Omron CX-Programmer project 新工程 (CX-Programmer 9.62)

# PLC 新PLC1: CJ2M CPU34
I/O table (CPU CJ2M-CPU34): rack 0 slot 0 CJ1W-ETN21(ETN21Mode); rack 0 slot 1 CJ1W-ID261; rack 0 slot 2 CJ1W-ID261; rack 0 slot 3 CJ1W-OD261; rack 0 slot 4 CJ1W-OD231; rack 0 slot 5 CJ1W-NC433; rack 0 slot 6 CJ1W-AD081-V1; rack 0 slot 7 CJ1W-DA08V; rack 0 slot 8 CJ1W-SCU21-V1; rack 0 slot 11 CJ2M-EIP21

## Global symbols (name address type ; comment)
0.00 BOOL  ; 手/自动选择
0.01 BOOL  ; 启动按钮
0.02 BOOL  ; 停止按钮
0.03 BOOL  ; 复位按钮
0.04 BOOL  ; 前门磁
0.05 BOOL  ; 后门磁
0.06 BOOL  ; 左门磁
0.07 BOOL  ; 右门磁
0.08 BOOL  ; 气源压力开关
0.09 BOOL  ; 主急停按钮
0.10 BOOL  ; 移动屏急停
0.11 BOOL  ; 移动屏使用中
0.12 BOOL  ; 备用1
0.13 BOOL  ; 备用2
0.14 BOOL  ; 备用3
0.15 BOOL  ; 备用4
100.00 BOOL  ; 进料定位上层前后松开输出
100.01 BOOL  ; 进料定位上层前后夹紧输出
100.02 BOOL  ; 进料定位下层前后松开输出
100.03 BOOL  ; 进料定位下层前后夹紧输出
100.04 BOOL  ; 进料定位上层左右松开输出
100.05 BOOL  ; 进料定位上层左右夹紧输出
100.06 BOOL  ; 进料定位下层左右松开输出
100.07 BOOL  ; 进料定位下层左右夹紧输出
100.08 BOOL  ; 进料定位上层平台待料输出
100.09 BOOL  ; 进料定位上层平台出料输出
100.10 BOOL  ; 进料定位下层平台待料输出
100.11 BOOL  ; 进料定位下层平台出料输出
100.12 BOOL  ; 输出
100.13 BOOL  ; 输出
100.14 BOOL  ; 输出
100.15 BOOL  ; 输出
101.00 BOOL  ; 输出
101.01 BOOL  ; 输出
101.02 BOOL  ; 输出
101.03 BOOL  ; 输出
101.04 BOOL  ; 输出
101.05 BOOL  ; 输出
101.06 BOOL  ; 输出
101.07 BOOL  ; 输出
101.08 BOOL  ; 输出
101.09 BOOL  ; 输出
101.10 BOOL  ; 输出
101.11 BOOL  ; 输出
101.12 BOOL  ; 输出
101.13 BOOL  ; 输出
101.14 BOOL  ; 输出
101.15 BOOL  ; 输出
102.00 BOOL  ; 输出
102.14 BOOL  ; 输出
102.15 BOOL  ; 输出
103.00 BOOL  ; 出料定位上层前后松开输出
103.01 BOOL  ; 出料定位上层前后夹紧输出
103.02 BOOL  ; 出料定位下层前后松开输出
103.03 BOOL  ; 出料定位下层前后夹紧输出
103.04 BOOL  ; 出料定位上层左右松开输出
103.05 BOOL  ; 出料定位上层左右夹紧输出
103.06 BOOL  ; 出料定位下层左右松开输出
103.07 BOOL  ; 出料定位下层左右夹紧输出
103.08 BOOL  ; 出料定位上层平台接料输出
103.09 BOOL  ; 出料定位上层平台出料输出
103.10 BOOL  ; 出料定位下层平台接料输出
103.11 BOOL  ; 出料定位下层平台出料输出
103.12 BOOL  ; 上下层吹气输出
103.13 BOOL  ; 输出
103.14 BOOL  ; 输出
103.15 BOOL  ; 输出
104.00 BOOL  ; 输出
104.01 BOOL  ; 输出
104.02 BOOL  ; 输出
104.03 BOOL  ; 输出
104.04 BOOL  ; 输出
104.05 BOOL  ; 输出
104.06 BOOL  ; 输出
104.07 BOOL  ; 输出
104.08 BOOL  ; 输出
104.09 BOOL  ; 输出
104.10 BOOL  ; 输出
105.14 BOOL  ; 输出
105.15 BOOL  ; 输出
106.00 BOOL  ; 进料夹爪张开输出
106.01 BOOL  ; 进料夹爪夹紧输出
106.02 BOOL  ; 进料爪上下层左右压紧上升输出
106.03 BOOL  ; 进料爪上下层左右压紧下降输出
106.04 BOOL  ; 进料爪上下层中间压紧上升输出
106.05 BOOL  ; 进料爪上下层中间压紧下降输出
106.06 BOOL  ; 进料夹爪上升输出
106.07 BOOL  ; 进料夹爪下降输出
106.08 BOOL  ; 输出
106.09 BOOL  ; 输出
106.10 BOOL  ; 输出
106.11 BOOL  ; 输出
106.12 BOOL  ; 输出
107.00 BOOL  ; 出料夹爪张开输出
107.01 BOOL  ; 出料夹爪夹紧输出
107.02 BOOL  ; 出料爪上下层左右压紧上升输出
107.03 BOOL  ; 出料爪上下层左右压紧下降输出
107.04 BOOL  ; 出料夹爪上升输出
107.05 BOOL  ; 出料夹爪下降输出
108.04 BOOL  ; 输出
108.05 BOOL  ; 输出
108.06 BOOL  ; 输出
108.07 BOOL  ; 输出
108.08 BOOL  ; 输出
108.09 BOOL  ; 输出
108.10 BOOL  ; 输出
108.11 BOOL  ; 输出
108.12 BOOL  ; 输出
108.13 BOOL  ; 输出
108.14 BOOL  ; 输出
108.15 BOOL  ; 输出
109.00 BOOL  ; 输出
109.01 BOOL  ; 输出
109.02 BOOL  ; 输出
109.03 BOOL  ; 输出
109.04 BOOL  ; 输出
109.05 BOOL  ; 输出
109.06 BOOL  ; 输出
109.07 BOOL  ; 输出
109.08 BOOL  ; 输出
109.09 BOOL  ; 输出
109.10 BOOL  ; 输出
109.11 BOOL  ; 输出
109.12 BOOL  ; 输出
109.13 BOOL  ; 输出
109.14 BOOL  ; 输出
109.15 BOOL  ; 输出
10.00 BOOL  ; 进料定位上层前后松开
10.01 BOOL  ; 进料定位上层前后夹紧
10.02 BOOL  ; 进料定位下层前后松开
10.03 BOOL  ; 进料定位下层前后夹紧
10.04 BOOL  ; 进料定位上层左右松开
10.05 BOOL  ; 进料定位上层左右夹紧
10.06 BOOL  ; 进料定位下层左右松开
10.07 BOOL  ; 进料定位下层左右夹紧
10.08 BOOL  ; 进料定位上层平台待料
10.09 BOOL  ; 进料定位上层平台出料
10.10 BOOL  ; 进料定位下层平台待料
10.11 BOOL  ; 进料定位下层平台出料
10.12 BOOL  ; 出料定位上层前后松开
10.13 BOOL  ; 出料定位上层前后夹紧
10.14 BOOL  ; 出料定位下层前后松开
10.15 BOOL  ; 出料定位下层前后夹紧
110.00 BOOL  ; 热压A增压缸上升输出
110.01 BOOL  ; 热压A增压缸下降输出
110.02 BOOL  ; 热压A上层顶升气缸上升输出
110.03 BOOL  ; 热压A上层顶升气缸下降输出
110.04 BOOL  ; 热压A下层顶升气缸上升输出
110.05 BOOL  ; 热压A下层顶升气缸下降输出
110.06 BOOL  ; 热压A垫高气缸移出输出
110.07 BOOL  ; 热压A垫高气缸热压输出
110.08 BOOL  ; 热压AHip测试气缸上升输出
110.09 BOOL  ; 热压AHip测试气缸下降输出
110.10 BOOL  ; 热压A上下层吹气输出
110.11 BOOL  ; 热压A上层HIP测试选择输出
110.12 BOOL  ; 热压A下层HIP测试选择输出
110.13 BOOL  ; 热压A极耳测试输出
110.14 BOOL  ; 热压A压力清零输出
110.15 BOOL  ; 热压B极耳测试输出
111.00 BOOL  ; 热压B压力清零输出
111.01 BOOL  ; 输出
111.02 BOOL  ; 输出
111.03 BOOL  ; 输出
111.04 BOOL  ; 输出
111.05 BOOL  ; 输出
111.06 BOOL  ; 输出
111.07 BOOL  ; 输出
111.08 BOOL  ; 输出
111.09 BOOL  ; 输出
111.10 BOOL  ; 输出
111.11 BOOL  ; 输出
111.12 BOOL  ; 输出
111.13 BOOL  ; 输出
111.14 BOOL  ; 输出
112 CHANNEL  ; 顶升伸出状态
112.14 BOOL  ; 输出
112.15 BOOL  ; 输出
113.00 BOOL  ; 热压B增压缸上升输出
113.01 BOOL  ; 热压B增压缸下降输出
113.02 BOOL  ; 热压B上层顶升气缸上升输出
113.03 BOOL  ; 热压B上层顶升气缸下降输出
113.04 BOOL  ; 热压B下层顶升气缸上升输出
113.05 BOOL  ; 热压B下层顶升气缸下降输出
113.06 BOOL  ; 热压B垫高气缸移出输出
113.07 BOOL  ; 热压B垫高气缸热压输出
113.08 BOOL  ; 热压BHip测试气缸上升输出
113.09 BOOL  ; 热压BHip测试气缸下降输出
113.10 BOOL  ; 热压B上下层吹气输出
113.11 BOOL  ; 热压B上层HIP测试选择输出
113.12 BOOL  ; 热压B下层HIP测试选择输出
113.13 BOOL  ; 热压B极耳测试输出
113.14 BOOL  ; 热压B压力清零输出
113.15 BOOL  ; 输出
114.00 BOOL  ; 输出
114.01 BOOL  ; 输出
114.02 BOOL  ; 输出
114.03 BOOL  ; 输出
114.04 BOOL  ; 输出
114.05 BOOL  ; 输出
114.06 BOOL  ; 输出
114.07 BOOL  ; 输出
114.08 BOOL  ; 输出
114.09 BOOL  ; 输出
114.10 BOOL  ; 输出
114.11 BOOL  ; 输出
114.12 BOOL  ; 输出
114.13 BOOL  ; 输出
114.14 BOOL  ; 输出
114.15 BOOL  ; 输出
115.00 BOOL  ; 输出
115.01 BOOL  ; 输出
116.00 BOOL  ; 热压C增压缸上升输出
116.01 BOOL  ; 热压C增压缸下降输出
116.02 BOOL  ; 热压C上层顶升气缸上升输出
116.03 BOOL  ; 热压C上层顶升气缸下降输出
116.04 BOOL  ; 热压C下层顶升气缸上升输出
116.05 BOOL  ; 热压C下层顶升气缸下降输出
116.06 BOOL  ; 热压C垫高气缸移出输出
116.07 BOOL  ; 热压C垫高气缸热压输出
116.08 BOOL  ; 热压CHip测试气缸上升输出
116.09 BOOL  ; 热压CHip测试气缸下降输出
116.10 BOOL  ; 热压C上下层吹气输出
116.11 BOOL  ; 热压C上层HIP测试选择输出
116.12 BOOL  ; 热压C下层HIP测试选择输出
116.13 BOOL  ; 热压C极耳测试输出
116.14 BOOL  ; 热压C压力清零输出
119.01 BOOL  ; 热压A正压伺服转矩模式输出
119.02 BOOL  ; 热压A1左右伺服转矩模式输出
119.07 BOOL  ; 热压B正压伺服转矩模式输出
119.08 BOOL  ; 热压B1左右伺服转矩模式输出
11.00 BOOL  ; 出料定位上层左右松开
11.01 BOOL  ; 出料定位上层左右夹紧
11.02 BOOL  ; 出料定位下层左右松开
11.03 BOOL  ; 出料定位下层左右夹紧
11.04 BOOL  ; 出料定位上层平台接料
11.05 BOOL  ; 出料定位上层平台出料
11.06 BOOL  ; 出料定位下层平台接料
11.07 BOOL  ; 出料定位下层平台出料
11.08 BOOL  ; 上下层吹气
11.09 BOOL  ; 进料夹爪张开
11.10 BOOL  ; 进料夹爪夹紧
11.11 BOOL  ; 进料爪上下层左右压紧上升
11.12 BOOL  ; 进料爪上下层左右压紧下降
11.13 BOOL  ; 进料爪上下层中间压紧上升
11.14 BOOL  ; 进料爪上下层中间压紧下降
11.15 BOOL  ; 进料夹爪上升
12.00 BOOL  ; 进料夹爪下降
12.01 BOOL  ; 出料夹爪张开
12.02 BOOL  ; 出料夹爪夹紧
12.03 BOOL  ; 进料爪上下层左右压紧上升
12.04 BOOL  ; 进料爪上下层左右压紧下降
12.05 BOOL  ; 进料爪上下层中间压紧上升
12.06 BOOL  ; 进料爪上下层中间压紧下降
12.07 BOOL  ; 进料夹爪上升
12.08 BOOL  ; 进料夹爪下降
12.09 BOOL  ; 热压A增压缸上升
12.10 BOOL  ; 热压A增压缸下降
12.11 BOOL  ; 热压A上层顶升气缸上升
12.12 BOOL  ; 热压A上层顶升气缸下降
12.13 BOOL  ; 热压A下层顶升气缸上升
12.14 BOOL  ; 热压A下层顶升气缸下降
12.15 BOOL  ; 热压A垫高气缸移出
13.00 BOOL  ; 热压A垫高气缸热压
13.01 BOOL  ; 热压AHip测试气缸上升
13.02 BOOL  ; 热压AHip测试气缸下降
13.03 BOOL  ; 热压A上下层吹气
13.04 BOOL  ; 热压A上层HIP测试选择继电器
13.05 BOOL  ; 热压A下层HIP测试选择继电器
13.06 BOOL  ; 热压A上下极耳有无检测继电器
13.07 BOOL  ; A工位压力清零
13.08 BOOL  ; 热压B增压缸上升
13.09 BOOL  ; 热压B增压缸下降
13.10 BOOL  ; 热压B上层顶升气缸上升
13.11 BOOL  ; 热压B上层顶升气缸下降
13.12 BOOL  ; 热压B下层顶升气缸上升
13.13 BOOL  ; 热压B下层顶升气缸下降
13.14 BOOL  ; 热压B垫高气缸移出
13.15 BOOL  ; 热压B垫高气缸热压
14.00 BOOL  ; 热压BHip测试气缸上升
14.01 BOOL  ; 热压BHip测试气缸下降
14.02 BOOL  ; 热压B上下层吹气
14.03 BOOL  ; 热压B上层HIP测试选择继电器
14.04 BOOL  ; 热压B下层HIP测试选择继电器
14.05 BOOL  ; 热压B上下极耳有无检测继电器
14.06 BOOL  ; B工位清零
14.07 BOOL  ; 热压C增压缸上升
14.08 BOOL  ; 热压C增压缸下降
14.09 BOOL  ; 热压C上层顶升气缸上升
14.10 BOOL  ; 热压C上层顶升气缸下降
14.11 BOOL  ; 热压C下层顶升气缸上升
14.12 BOOL  ; 热压C下层顶升气缸下降
14.13 BOOL  ; 热压C垫高气缸移出
14.14 BOOL  ; 热压C垫高气缸热压
14.15 BOOL  ; 热压CHip测试气缸上升
1550.03 BOOL  ; #2_1端口停止
1550.11 BOOL  ; #2_2端口停止
1559.15 BOOL  ; 单元2-端口1忙标志
1569.15 BOOL  ; 单元2-端口2忙标志
1575.03 BOOL  ; #3_1端口停止
1575.11 BOOL  ; #3_2端口停止
1584.15 BOOL  ; 单元3-端口1忙标志
1594.15 BOOL  ; 单元3-端口2忙标志
15.00 BOOL  ; 热压CHip测试气缸下降
15.01 BOOL  ; 热压C上下层吹气
15.02 BOOL  ; 热压C上层HIP测试选择继电器
15.03 BOOL  ; 热压C下层HIP测试选择继电器
15.04 BOOL  ; 热压C上下极耳有无检测继电器
15.05 BOOL  ; C工位压力清零
15.07 BOOL  ; 横移|伸缩伺服ON
15.08 BOOL  ; 横移|伸缩伺服报警解除
15.09 BOOL  ; 三个灯 红
15.10 BOOL  ; 三个灯 黄
15.11 BOOL  ; 三个灯 绿
15.12 BOOL  ; 三色灯蜂鸣器
15.13 BOOL  ; 运行指示（面板）
15.14 BOOL  ; 复位指示（面板）
15.15 BOOL  ; 停止指示（面板）
16 CHANNEL  ; 副PLC输出点映射开始地址
1600.03 BOOL  ; #4_1端口停止
1600.11 BOOL  ; #4_2端口停止
1609.15 BOOL  ; 单元4-端口1忙标志
1619.15 BOOL  ; 单元4-端口2忙标志
1625.03 BOOL  ; #5_1端口停止
1625.11 BOOL  ; #5_2端口停止
1634.15 BOOL  ; 单元5-端口1忙标志
1644.15 BOOL  ; 单元5-端口2忙标志
1659.15 BOOL  ; 单元6-端口1忙标志
1669.15 BOOL  ; 单元6-端口1忙标志
16.00 BOOL  ; 热压A上层上板左加热启动 上料侧为左
16.01 BOOL  ; 热压A上层上板中加热启动
16.02 BOOL  ; 热压A上层上板右加热启动
16.03 BOOL  ; 热压A上层下板左加热启动
16.04 BOOL  ; 热压A上层下板中加热启动
16.05 BOOL  ; 热压A上层下板右加热启动
17.00 BOOL  ; 热压A下层上板左加热启动
17.01 BOOL  ; 热压A下层上板中加热启动
17.02 BOOL  ; 热压A下层上板右加热启动
17.03 BOOL  ; 热压A下层下板左加热启动
17.04 BOOL  ; 热压A下层下板中加热启动
17.05 BOOL  ; 热压A下层下板右加热启动
18.00 BOOL  ; 热压B上层上板左加热启动
18.01 BOOL  ; 热压B上层上板中加热启动
18.02 BOOL  ; 热压B上层上板右加热启动
18.03 BOOL  ; 热压B上层下板左加热启动
18.04 BOOL  ; 热压B上层下板中加热启动
18.05 BOOL  ; 热压B上层下板右加热启动
19.00 BOOL  ; 热压B下层上板左加热启动
19.01 BOOL  ; 热压B下层上板中加热启动
19.02 BOOL  ; 热压B下层上板右加热启动
19.03 BOOL  ; 热压B下层下板左加热启动
19.04 BOOL  ; 热压B下层下板中加热启动
19.05 BOOL  ; 热压B下层下板右加热启动
1.00 BOOL  ; 启动按钮1
1.01 BOOL  ; 启动按钮2
1.02 BOOL  ; 进出料安全光栅
1.03 BOOL  ; 进料定位上层前后松开位
1.04 BOOL  ; 进料定位上层前后夹紧位
1.05 BOOL  ; 进料定位下层前后松开位
1.06 BOOL  ; 进料定位下层前后夹紧位
1.07 BOOL  ; 进料定位上层左右松开位
1.08 BOOL  ; 进料定位上层左右夹紧位
1.09 BOOL  ; 进料定位下层左右松开位
1.10 BOOL  ; 进料定位下层左右夹紧位
1.11 BOOL  ; 进料定位平台上层待料位
1.12 BOOL  ; 进料定位平台上层出料位
1.13 BOOL  ; 进料定位平台下层待料位
1.14 BOOL  ; 进料定位平台下层出料位
1.15 BOOL  ; 进料定位上层有料感应
2000.00 BOOL  ; NC433_0_X 3ST-A进出料横移伺服A存储器操作命令激活序列数
2000.01 BOOL  ; NC433_0_X 3ST-A进出料横移伺服A存储器操作命令起动
2000.02 BOOL  ; NC433_0_X 3ST-A进出料横移伺服A存储器操作命令独立起动
2000.03 BOOL  ; NC433_0_X 3ST-A进出料横移伺服A直接操作命令绝对移动
2000.04 BOOL  ; NC433_0_X 3ST-A进出料横移伺服A直接操作命令相对移动
2000.05 BOOL  ; NC433_0_X 3ST-A进出料横移伺服A直接操作命令中断进给
2000.06 BOOL  ; NC433_0_X 3ST-A进出料横移伺服A原点定位命令原点搜索
2000.07 BOOL  ; NC433_0_X 3ST-A进出料横移伺服A原点定位命令原点返回
2000.08 BOOL  ; NC433_0_X 3ST-A进出料横移伺服A原点定位命令当前位置预置
2000.09 BOOL  ; NC433_0_X 3ST-A进出料横移伺服A点动
2000.10 BOOL  ; NC433_0_X 3ST-A进出料横移伺服A点动方向(0=CW,1=CCW)
2000.11 BOOL  ; NC433_0_X 3ST-A进出料横移伺服A示教
2000.12 BOOL  ; NC433_0_X 3ST-A进出料横移伺服A错误清除
2000.13 BOOL  ; NC433_0_X 3ST-A进出料横移伺服A偏差计数器复位输出/ 原点调整命令输出
2000.14 BOOL  ; NC433_0_X 3ST-A进出料横移伺服A激活Override
2000.15 BOOL  ; NC433_0_X 3ST-A进出料横移伺服A停止
2001.00 BOOL  ; NC433_0_X 3ST-A进出料横移伺服A预留
2001.01 BOOL  ; NC433_0_X 3ST-A进出料横移伺服A预留
2001.02 BOOL  ; NC433_0_X 3ST-A进出料横移伺服A预留
2001.03 BOOL  ; NC433_0_X 3ST-A进出料横移伺服A预留
2001.04 BOOL  ; NC433_0_X 3ST-A进出料横移伺服A预留
2001.05 BOOL  ; NC433_0_X 3ST-A进出料横移伺服A预留
2001.06 BOOL  ; NC433_0_X 3ST-A进出料横移伺服A预留
2001.07 BOOL  ; NC433_0_X 3ST-A进出料横移伺服A预留
2001.08 BOOL  ; NC433_0_X 3ST-A进出料横移伺服A强制中断
2001.09 BOOL  ; NC433_0_X 3ST-A进出料横移伺服A预留
2001.10 BOOL  ; NC433_0_X 3ST-A进出料横移伺服A预留
2001.11 BOOL  ; NC433_0_X 3ST-A进出料横移伺服A预留
2001.12 BOOL  ; NC433_0_X 3ST-A进出料横移伺服A数据写入
2001.13 BOOL  ; NC433_0_X 3ST-A进出料横移伺服A数据读出
2001.14 BOOL  ; NC433_0_X 3ST-A进出料横移伺服A数据保存
2001.15 BOOL  ; NC433_0_X 3ST-A进出料横移伺服A预留
2002.00 BOOL  ; NC433_0_Y 3ST-A进出料伸缩伺服A存储器操作命令激活序列数
2002.01 BOOL  ; NC433_0_Y 3ST-A进出料伸缩伺服A存储器操作命令起动
2002.02 BOOL  ; NC433_0_Y 3ST-A进出料伸缩伺服A存储器操作命令独立起动
2002.03 BOOL  ; NC433_0_Y 3ST-A进出料伸缩伺服A直接操作命令绝对移动
2002.04 BOOL  ; NC433_0_Y 3ST-A进出料伸缩伺服A直接操作命令相对移动
2002.05 BOOL  ; NC433_0_Y 3ST-A进出料伸缩伺服A直接操作命令中断进给
2002.06 BOOL  ; NC433_0_Y 3ST-A进出料伸缩伺服A原点定位命令原点搜索
2002.07 BOOL  ; NC433_0_Y 3ST-A进出料伸缩伺服A原点定位命令原点返回
2002.08 BOOL  ; NC433_0_Y 3ST-A进出料伸缩伺服A原点定位命令当前位置预置
2002.09 BOOL  ; NC433_0_Y 3ST-A进出料伸缩伺服A点动
2002.10 BOOL  ; NC433_0_Y 3ST-A进出料伸缩伺服A点动方向(0=CW,1=CCW)
2002.11 BOOL  ; NC433_0_Y 3ST-A进出料伸缩伺服A示教
2002.12 BOOL  ; NC433_0_Y 3ST-A进出料伸缩伺服A错误清除
2002.13 BOOL  ; NC433_0_Y 3ST-A进出料伸缩伺服A偏差计数器复位输出/ 原点调整命令输出
2002.14 BOOL  ; NC433_0_Y 3ST-A进出料伸缩伺服A激活Override
2002.15 BOOL  ; NC433_0_Y 3ST-A进出料伸缩伺服A停止
2003.00 BOOL  ; NC433_0_Y 3ST-A进出料伸缩伺服A预留
2003.01 BOOL  ; NC433_0_Y 3ST-A进出料伸缩伺服A预留
2003.02 BOOL  ; NC433_0_Y 3ST-A进出料伸缩伺服A预留
2003.03 BOOL  ; NC433_0_Y 3ST-A进出料伸缩伺服A预留
2003.04 BOOL  ; NC433_0_Y 3ST-A进出料伸缩伺服A预留
2003.05 BOOL  ; NC433_0_Y 3ST-A进出料伸缩伺服A预留
2003.06 BOOL  ; NC433_0_Y 3ST-A进出料伸缩伺服A预留
2003.07 BOOL  ; NC433_0_Y 3ST-A进出料伸缩伺服A预留
2003.08 BOOL  ; NC433_0_Y 3ST-A进出料伸缩伺服A强制中断
2003.09 BOOL  ; NC433_0_Y 3ST-A进出料伸缩伺服A预留
2003.10 BOOL  ; NC433_0_Y 3ST-A进出料伸缩伺服A预留
2003.11 BOOL  ; NC433_0_Y 3ST-A进出料伸缩伺服A预留
2003.12 BOOL  ; NC433_0_Y 3ST-A进出料伸缩伺服A数据写入
2003.13 BOOL  ; NC433_0_Y 3ST-A进出料伸缩伺服A数据读出
2003.14 BOOL  ; NC433_0_Y 3ST-A进出料伸缩伺服A数据保存
2003.15 BOOL  ; NC433_0_Y 3ST-A进出料伸缩伺服A预留
2004.00 BOOL  ; NC433_0_ Z 3ST-B进出料横移伺服B存储器操作命令激活序列数
2004.01 BOOL  ; NC433_0_ Z 3ST-B进出料横移伺服B存储器操作命令起动
2004.02 BOOL  ; NC433_0_ Z 3ST-B进出料横移伺服B存储器操作命令独立起动
2004.03 BOOL  ; NC433_0_ Z 3ST-B进出料横移伺服B直接操作命令绝对移动
2004.04 BOOL  ; NC433_0_ Z 3ST-B进出料横移伺服B直接操作命令相对移动
2004.05 BOOL  ; NC433_0_ Z 3ST-B进出料横移伺服B直接操作命令中断进给
2004.06 BOOL  ; NC433_0_ Z 3ST-B进出料横移伺服B原点定位命令原点搜索
2004.07 BOOL  ; NC433_0_ Z 3ST-B进出料横移伺服B原点定位命令原点返回
2004.08 BOOL  ; NC433_0_ Z 3ST-B进出料横移伺服B原点定位命令当前位置预置
2004.09 BOOL  ; NC433_0_ Z 3ST-B进出料横移伺服B点动
2004.10 BOOL  ; NC433_0_ Z 3ST-B进出料横移伺服B点动方向(0=CW,1=CCW)
2004.11 BOOL  ; NC433_0_ Z 3ST-B进出料横移伺服B示教
2004.12 BOOL  ; NC433_0_ Z 3ST-B进出料横移伺服B错误清除
2004.13 BOOL  ; NC433_0_ Z 3ST-B进出料横移伺服B偏差计数器复位输出/ 原点调整命令输出
2004.14 BOOL  ; NC433_0_ Z 3ST-B进出料横移伺服B激活Override
2004.15 BOOL  ; NC433_0_ Z 3ST-B进出料横移伺服B停止
2005.00 BOOL  ; NC433_0_ Z 3ST-B进出料横移伺服B预留
2005.01 BOOL  ; NC433_0_ Z 3ST-B进出料横移伺服B预留
2005.02 BOOL  ; NC433_0_ Z 3ST-B进出料横移伺服B预留
2005.03 BOOL  ; NC433_0_ Z 3ST-B进出料横移伺服B预留
2005.04 BOOL  ; NC433_0_ Z 3ST-B进出料横移伺服B预留
2005.05 BOOL  ; NC433_0_ Z 3ST-B进出料横移伺服B预留
2005.06 BOOL  ; NC433_0_ Z 3ST-B进出料横移伺服B预留
2005.07 BOOL  ; NC433_0_ Z 3ST-B进出料横移伺服B预留
2005.08 BOOL  ; NC433_0_ Z 3ST-B进出料横移伺服B强制中断
2005.09 BOOL  ; NC433_0_ Z 3ST-B进出料横移伺服B预留
2005.10 BOOL  ; NC433_0_ Z 3ST-B进出料横移伺服B预留
2005.11 BOOL  ; NC433_0_ Z 3ST-B进出料横移伺服B预留
2005.12 BOOL  ; NC433_0_ Z 3ST-B进出料横移伺服B数据写入
2005.13 BOOL  ; NC433_0_ Z 3ST-B进出料横移伺服B数据读出
2005.14 BOOL  ; NC433_0_ Z 3ST-B进出料横移伺服B数据保存
2005.15 BOOL  ; NC433_0_ Z 3ST-B进出料横移伺服B预留
2006.00 BOOL  ; NC433_0_U 3ST-B进出料伸缩伺服存储器操作命令激活序列数
2006.01 BOOL  ; NC433_0_U 3ST-B进出料伸缩伺服存储器操作命令起动
2006.02 BOOL  ; NC433_0_U 3ST-B进出料伸缩伺服存储器操作命令独立起动
2006.03 BOOL  ; NC433_0_U 3ST-B进出料伸缩伺服直接操作命令绝对移动
2006.04 BOOL  ; NC433_0_U 3ST-B进出料伸缩伺服直接操作命令相对移动
2006.05 BOOL  ; NC433_0_U 3ST-B进出料伸缩伺服直接操作命令中断进给
2006.06 BOOL  ; NC433_0_U 3ST-B进出料伸缩伺服原点定位命令原点搜索
2006.07 BOOL  ; NC433_0_U 3ST-B进出料伸缩伺服原点定位命令原点返回
2006.08 BOOL  ; NC433_0_U 3ST-B进出料伸缩伺服原点定位命令当前位置预置
2006.09 BOOL  ; NC433_0_U 3ST-B进出料伸缩伺服点动
2006.10 BOOL  ; NC433_0_U 3ST-B进出料伸缩伺服点动方向(0=CW,1=CCW)
2006.11 BOOL  ; NC433_0_U 3ST-B进出料伸缩伺服示教
2006.12 BOOL  ; NC433_0_U 3ST-B进出料伸缩伺服错误清除
2006.13 BOOL  ; NC433_0_U 3ST-B进出料伸缩伺服偏差计数器复位输出/ 原点调整命令输出
2006.14 BOOL  ; NC433_0_U 3ST-B进出料伸缩伺服激活Override
2006.15 BOOL  ; NC433_0_U 3ST-B进出料伸缩伺服停止
2007.00 BOOL  ; NC433_0_U 3ST-B进出料伸缩伺服预留
2007.01 BOOL  ; NC433_0_U 3ST-B进出料伸缩伺服预留
2007.02 BOOL  ; NC433_0_U 3ST-B进出料伸缩伺服预留
2007.03 BOOL  ; NC433_0_U 3ST-B进出料伸缩伺服预留
2007.04 BOOL  ; NC433_0_U 3ST-B进出料伸缩伺服预留
2007.05 BOOL  ; NC433_0_U 3ST-B进出料伸缩伺服预留
2007.06 BOOL  ; NC433_0_U 3ST-B进出料伸缩伺服预留
2007.07 BOOL  ; NC433_0_U 3ST-B进出料伸缩伺服预留
2007.08 BOOL  ; NC433_0_U 3ST-B进出料伸缩伺服强制中断
2007.09 BOOL  ; NC433_0_U 3ST-B进出料伸缩伺服预留
2007.10 BOOL  ; NC433_0_U 3ST-B进出料伸缩伺服预留
2007.11 BOOL  ; NC433_0_U 3ST-B进出料伸缩伺服预留
2007.12 BOOL  ; NC433_0_U 3ST-B进出料伸缩伺服数据写入
2007.13 BOOL  ; NC433_0_U 3ST-B进出料伸缩伺服数据读出
2007.14 BOOL  ; NC433_0_U 3ST-B进出料伸缩伺服数据保存
2007.15 BOOL  ; NC433_0_U 3ST-B进出料伸缩伺服预留
2008.00 BOOL  ; NC433_0_X 3ST-A进出料横移伺服A预留
2008.01 BOOL  ; NC433_0_X 3ST-A进出料横移伺服A预留
2008.02 BOOL  ; NC433_0_X 3ST-A进出料横移伺服A预留
2008.03 BOOL  ; NC433_0_X 3ST-A进出料横移伺服A预留
2008.04 BOOL  ; NC433_0_X 3ST-A进出料横移伺服A等待存储器操作
2008.05 BOOL  ; NC433_0_X 3ST-A进出料横移伺服A定位完成标志位
2008.06 BOOL  ; NC433_0_X 3ST-A进出料横移伺服A无原点标志位
2008.07 BOOL  ; NC433_0_X 3ST-A进出料横移伺服A原点停止标志位
2008.08 BOOL  ; NC433_0_X 3ST-A进出料横移伺服A0 区监测标志位
2008.09 BOOL  ; NC433_0_X 3ST-A进出料横移伺服A1 区监测标志位
2008.10 BOOL  ; NC433_0_X 3ST-A进出料横移伺服A2 区监测标志位
2008.11 BOOL  ; NC433_0_X 3ST-A进出料横移伺服A示教完成
2008.12 BOOL  ; NC433_0_X 3ST-A进出料横移伺服A错误标志
2008.13 BOOL  ; NC433_0_X 3ST-A进出料横移伺服A忙标志
2008.14 BOOL  ; NC433_0_X 3ST-A进出料横移伺服A数据传送标志位
2008.15 BOOL  ; NC433_0_X 3ST-A进出料横移伺服A减速停止执行标志位
2009.00 BOOL  ; NC433_0_X 3ST-A进出料横移伺服A预留
2009.01 BOOL  ; NC433_0_X 3ST-A进出料横移伺服A预留
2009.02 BOOL  ; NC433_0_X 3ST-A进出料横移伺服A预留
2009.03 BOOL  ; NC433_0_X 3ST-A进出料横移伺服A预留
2009.04 BOOL  ; NC433_0_X 3ST-A进出料横移伺服A预留
2009.05 BOOL  ; NC433_0_X 3ST-A进出料横移伺服A预留
2009.06 BOOL  ; NC433_0_X 3ST-A进出料横移伺服A预留
2009.07 BOOL  ; NC433_0_X 3ST-A进出料横移伺服A预留
2009.08 BOOL  ; NC433_0_X 3ST-A进出料横移伺服ACW极限输入信号
2009.09 BOOL  ; NC433_0_X 3ST-A进出料横移伺服ACCW极限输入信号
2009.10 BOOL  ; NC433_0_X 3ST-A进出料横移伺服A原点接近输入信号
2009.11 BOOL  ; NC433_0_X 3ST-A进出料横移伺服A原点输入信号
2009.12 BOOL  ; NC433_0_X 3ST-A进出料横移伺服A中断输入信号
2009.13 BOOL  ; NC433_0_X 3ST-A进出料横移伺服A紧急输入信号
2009.14 BOOL  ; NC433_0_X 3ST-A进出料横移伺服A定位完成输入信号
2009.15 BOOL  ; NC433_0_X 3ST-A进出料横移伺服A偏差计数器复位输出/ 原点调整命令输出
2010.00 BOOL  ; NC433_0_X 3ST-A进出料横移伺服A错误代码
2010.01 BOOL  ; NC433_0_X 3ST-A进出料横移伺服A错误代码
2010.02 BOOL  ; NC433_0_X 3ST-A进出料横移伺服A错误代码
2010.03 BOOL  ; NC433_0_X 3ST-A进出料横移伺服A错误代码
2010.04 BOOL  ; NC433_0_X 3ST-A进出料横移伺服A错误代码
2010.05 BOOL  ; NC433_0_X 3ST-A进出料横移伺服A错误代码
2010.06 BOOL  ; NC433_0_X 3ST-A进出料横移伺服A错误代码
2010.07 BOOL  ; NC433_0_X 3ST-A进出料横移伺服A错误代码
2010.08 BOOL  ; NC433_0_X 3ST-A进出料横移伺服A错误代码
2010.09 BOOL  ; NC433_0_X 3ST-A进出料横移伺服A错误代码
2010.10 BOOL  ; NC433_0_X 3ST-A进出料横移伺服A错误代码
2010.11 BOOL  ; NC433_0_X 3ST-A进出料横移伺服A错误代码
2010.12 BOOL  ; NC433_0_X 3ST-A进出料横移伺服A错误代码
2010.13 BOOL  ; NC433_0_X 3ST-A进出料横移伺服A错误代码
2010.14 BOOL  ; NC433_0_X 3ST-A进出料横移伺服A错误代码
2010.15 BOOL  ; NC433_0_X 3ST-A进出料横移伺服A错误代码
2011.00 BOOL  ; NC433_0_Y 3ST-A进出料伸缩伺服A预留
2011.01 BOOL  ; NC433_0_Y 3ST-A进出料伸缩伺服A预留
2011.02 BOOL  ; NC433_0_Y 3ST-A进出料伸缩伺服A预留
2011.03 BOOL  ; NC433_0_Y 3ST-A进出料伸缩伺服A预留
2011.04 BOOL  ; NC433_0_Y 3ST-A进出料伸缩伺服A等待存储器操作
2011.05 BOOL  ; NC433_0_Y 3ST-A进出料伸缩伺服A定位完成标志位
2011.06 BOOL  ; NC433_0_Y 3ST-A进出料伸缩伺服A无原点标志位
2011.07 BOOL  ; NC433_0_Y 3ST-A进出料伸缩伺服A原点停止标志位
2011.08 BOOL  ; NC433_0_Y 3ST-A进出料伸缩伺服A0 区监测标志位
2011.09 BOOL  ; NC433_0_Y 3ST-A进出料伸缩伺服A1 区监测标志位
2011.10 BOOL  ; NC433_0_Y 3ST-A进出料伸缩伺服A2 区监测标志位
2011.11 BOOL  ; NC433_0_Y 3ST-A进出料伸缩伺服A示教完成
2011.12 BOOL  ; NC433_0_Y 3ST-A进出料伸缩伺服A错误标志
2011.13 BOOL  ; NC433_0_Y 3ST-A进出料伸缩伺服A忙标志
2011.14 BOOL  ; NC433_0_Y 3ST-A进出料伸缩伺服A数据传送标志位
2011.15 BOOL  ; NC433_0_Y 3ST-A进出料伸缩伺服A减速停止执行标志位
2012.00 BOOL  ; NC433_0_Y 3ST-A进出料伸缩伺服A预留
2012.01 BOOL  ; NC433_0_Y 3ST-A进出料伸缩伺服A预留
2012.02 BOOL  ; NC433_0_Y 3ST-A进出料伸缩伺服A预留
2012.03 BOOL  ; NC433_0_Y 3ST-A进出料伸缩伺服A预留
2012.04 BOOL  ; NC433_0_Y 3ST-A进出料伸缩伺服A预留
2012.05 BOOL  ; NC433_0_Y 3ST-A进出料伸缩伺服A预留
2012.06 BOOL  ; NC433_0_Y 3ST-A进出料伸缩伺服A预留
2012.07 BOOL  ; NC433_0_Y 3ST-A进出料伸缩伺服A预留
2012.08 BOOL  ; NC433_0_Y 3ST-A进出料伸缩伺服ACW极限输入信号
2012.09 BOOL  ; NC433_0_Y 3ST-A进出料伸缩伺服ACCW极限输入信号
2012.10 BOOL  ; NC433_0_Y 3ST-A进出料伸缩伺服A原点接近输入信号
2012.11 BOOL  ; NC433_0_Y 3ST-A进出料伸缩伺服A原点输入信号
2012.12 BOOL  ; NC433_0_Y 3ST-A进出料伸缩伺服A中断输入信号
2012.13 BOOL  ; NC433_0_Y 3ST-A进出料伸缩伺服A紧急输入信号
2012.14 BOOL  ; NC433_0_Y 3ST-A进出料伸缩伺服A定位完成输入信号
2012.15 BOOL  ; NC433_0_Y 3ST-A进出料伸缩伺服A偏差计数器复位输出/ 原点调整命令输出
2013.00 BOOL  ; NC433_0_Y 3ST-A进出料伸缩伺服A错误代码
2013.01 BOOL  ; NC433_0_Y 3ST-A进出料伸缩伺服A错误代码
2013.02 BOOL  ; NC433_0_Y 3ST-A进出料伸缩伺服A错误代码
2013.03 BOOL  ; NC433_0_Y 3ST-A进出料伸缩伺服A错误代码
2013.04 BOOL  ; NC433_0_Y 3ST-A进出料伸缩伺服A错误代码
2013.05 BOOL  ; NC433_0_Y 3ST-A进出料伸缩伺服A错误代码
2013.06 BOOL  ; NC433_0_Y 3ST-A进出料伸缩伺服A错误代码
2013.07 BOOL  ; NC433_0_Y 3ST-A进出料伸缩伺服A错误代码
2013.08 BOOL  ; NC433_0_Y 3ST-A进出料伸缩伺服A错误代码
2013.09 BOOL  ; NC433_0_Y 3ST-A进出料伸缩伺服A错误代码
2013.10 BOOL  ; NC433_0_Y 3ST-A进出料伸缩伺服A错误代码
2013.11 BOOL  ; NC433_0_Y 3ST-A进出料伸缩伺服A错误代码
2013.12 BOOL  ; NC433_0_Y 3ST-A进出料伸缩伺服A错误代码
2013.13 BOOL  ; NC433_0_Y 3ST-A进出料伸缩伺服A错误代码
2013.14 BOOL  ; NC433_0_Y 3ST-A进出料伸缩伺服A错误代码
2013.15 BOOL  ; NC433_0_Y 3ST-A进出料伸缩伺服A错误代码
2014.00 BOOL  ; NC433_0_ Z 3ST-B进出料横移伺服B预留
2014.01 BOOL  ; NC433_0_ Z 3ST-B进出料横移伺服B预留
2014.02 BOOL  ; NC433_0_ Z 3ST-B进出料横移伺服B预留
2014.03 BOOL  ; NC433_0_ Z 3ST-B进出料横移伺服B预留
2014.04 BOOL  ; NC433_0_ Z 3ST-B进出料横移伺服B等待存储器操作
2014.05 BOOL  ; NC433_0_ Z 3ST-B进出料横移伺服B定位完成标志位
2014.06 BOOL  ; NC433_0_ Z 3ST-B进出料横移伺服B无原点标志位
2014.07 BOOL  ; NC433_0_ Z 3ST-B进出料横移伺服B原点停止标志位
2014.08 BOOL  ; NC433_0_ Z 3ST-B进出料横移伺服B0 区监测标志位
2014.09 BOOL  ; NC433_0_ Z 3ST-B进出料横移伺服B1 区监测标志位
2014.10 BOOL  ; NC433_0_ Z 3ST-B进出料横移伺服B2 区监测标志位
2014.11 BOOL  ; NC433_0_ Z 3ST-B进出料横移伺服B示教完成
2014.12 BOOL  ; NC433_0_ Z 3ST-B进出料横移伺服B错误标志
2014.13 BOOL  ; NC433_0_ Z 3ST-B进出料横移伺服B忙标志
2014.14 BOOL  ; NC433_0_ Z 3ST-B进出料横移伺服B数据传送标志位
2014.15 BOOL  ; NC433_0_ Z 3ST-B进出料横移伺服B减速停止执行标志位
2015.00 BOOL  ; NC433_0_ Z 3ST-B进出料横移伺服B预留
2015.01 BOOL  ; NC433_0_ Z 3ST-B进出料横移伺服B预留
2015.02 BOOL  ; NC433_0_ Z 3ST-B进出料横移伺服B预留
2015.03 BOOL  ; NC433_0_ Z 3ST-B进出料横移伺服B预留
2015.04 BOOL  ; NC433_0_ Z 3ST-B进出料横移伺服B预留
2015.05 BOOL  ; NC433_0_ Z 3ST-B进出料横移伺服B预留
2015.06 BOOL  ; NC433_0_ Z 3ST-B进出料横移伺服B预留
2015.07 BOOL  ; NC433_0_ Z 3ST-B进出料横移伺服B预留
2015.08 BOOL  ; NC433_0_ Z 3ST-B进出料横移伺服BCW极限输入信号
2015.09 BOOL  ; NC433_0_ Z 3ST-B进出料横移伺服BCCW极限输入信号
2015.10 BOOL  ; NC433_0_ Z 3ST-B进出料横移伺服B原点接近输入信号
2015.11 BOOL  ; NC433_0_ Z 3ST-B进出料横移伺服B原点输入信号
2015.12 BOOL  ; NC433_0_ Z 3ST-B进出料横移伺服B中断输入信号
2015.13 BOOL  ; NC433_0_ Z 3ST-B进出料横移伺服B紧急输入信号
2015.14 BOOL  ; NC433_0_ Z 3ST-B进出料横移伺服B定位完成输入信号
2015.15 BOOL  ; NC433_0_ Z 3ST-B进出料横移伺服B偏差计数器复位输出/ 原点调整命令输出
2016.00 BOOL  ; NC433_0_ Z 3ST-B进出料横移伺服B错误代码
2016.01 BOOL  ; NC433_0_ Z 3ST-B进出料横移伺服B错误代码
2016.02 BOOL  ; NC433_0_ Z 3ST-B进出料横移伺服B错误代码
2016.03 BOOL  ; NC433_0_ Z 3ST-B进出料横移伺服B错误代码
2016.04 BOOL  ; NC433_0_ Z 3ST-B进出料横移伺服B错误代码
2016.05 BOOL  ; NC433_0_ Z 3ST-B进出料横移伺服B错误代码
2016.06 BOOL  ; NC433_0_ Z 3ST-B进出料横移伺服B错误代码
2016.07 BOOL  ; NC433_0_ Z 3ST-B进出料横移伺服B错误代码
2016.08 BOOL  ; NC433_0_ Z 3ST-B进出料横移伺服B错误代码
2016.09 BOOL  ; NC433_0_ Z 3ST-B进出料横移伺服B错误代码
2016.10 BOOL  ; NC433_0_ Z 3ST-B进出料横移伺服B错误代码
2016.11 BOOL  ; NC433_0_ Z 3ST-B进出料横移伺服B错误代码
2016.12 BOOL  ; NC433_0_ Z 3ST-B进出料横移伺服B错误代码
2016.13 BOOL  ; NC433_0_ Z 3ST-B进出料横移伺服B错误代码
2016.14 BOOL  ; NC433_0_ Z 3ST-B进出料横移伺服B错误代码
2016.15 BOOL  ; NC433_0_ Z 3ST-B进出料横移伺服B错误代码
2017.00 BOOL  ; NC433_0_U 3ST-B进出料伸缩伺服预留
2017.01 BOOL  ; NC433_0_U 3ST-B进出料伸缩伺服预留
2017.02 BOOL  ; NC433_0_U 3ST-B进出料伸缩伺服预留
2017.03 BOOL  ; NC433_0_U 3ST-B进出料伸缩伺服预留
2017.04 BOOL  ; NC433_0_U 3ST-B进出料伸缩伺服等待存储器操作
2017.05 BOOL  ; NC433_0_U 3ST-B进出料伸缩伺服定位完成标志位
2017.06 BOOL  ; NC433_0_U 3ST-B进出料伸缩伺服无原点标志位
2017.07 BOOL  ; NC433_0_U 3ST-B进出料伸缩伺服原点停止标志位
2017.08 BOOL  ; NC433_0_U 3ST-B进出料伸缩伺服0 区监测标志位
2017.09 BOOL  ; NC433_0_U 3ST-B进出料伸缩伺服1 区监测标志位
2017.10 BOOL  ; NC433_0_U 3ST-B进出料伸缩伺服2 区监测标志位
2017.11 BOOL  ; NC433_0_U 3ST-B进出料伸缩伺服示教完成
2017.12 BOOL  ; NC433_0_U 3ST-B进出料伸缩伺服错误标志
2017.13 BOOL  ; NC433_0_U 3ST-B进出料伸缩伺服忙标志
2017.14 BOOL  ; NC433_0_U 3ST-B进出料伸缩伺服数据传送标志位
2017.15 BOOL  ; NC433_0_U 3ST-B进出料伸缩伺服减速停止执行标志位
2018.00 BOOL  ; NC433_0_U 3ST-B进出料伸缩伺服预留
2018.01 BOOL  ; NC433_0_U 3ST-B进出料伸缩伺服预留
2018.02 BOOL  ; NC433_0_U 3ST-B进出料伸缩伺服预留
2018.03 BOOL  ; NC433_0_U 3ST-B进出料伸缩伺服预留
2018.04 BOOL  ; NC433_0_U 3ST-B进出料伸缩伺服预留
2018.05 BOOL  ; NC433_0_U 3ST-B进出料伸缩伺服预留
2018.06 BOOL  ; NC433_0_U 3ST-B进出料伸缩伺服预留
2018.07 BOOL  ; NC433_0_U 3ST-B进出料伸缩伺服预留
2018.08 BOOL  ; NC433_0_U 3ST-B进出料伸缩伺服CW极限输入信号
2018.09 BOOL  ; NC433_0_U 3ST-B进出料伸缩伺服CCW极限输入信号
2018.10 BOOL  ; NC433_0_U 3ST-B进出料伸缩伺服原点接近输入信号
2018.11 BOOL  ; NC433_0_U 3ST-B进出料伸缩伺服原点输入信号
2018.12 BOOL  ; NC433_0_U 3ST-B进出料伸缩伺服中断输入信号
2018.13 BOOL  ; NC433_0_U 3ST-B进出料伸缩伺服紧急输入信号
2018.14 BOOL  ; NC433_0_U 3ST-B进出料伸缩伺服定位完成输入信号
2018.15 BOOL  ; NC433_0_U 3ST-B进出料伸缩伺服偏差计数器复位输出/ 原点调整命令输出
2019.00 BOOL  ; NC433_0_U 3ST-B进出料伸缩伺服错误代码
2019.01 BOOL  ; NC433_0_U 3ST-B进出料伸缩伺服错误代码
2019.02 BOOL  ; NC433_0_U 3ST-B进出料伸缩伺服错误代码
2019.03 BOOL  ; NC433_0_U 3ST-B进出料伸缩伺服错误代码
2019.04 BOOL  ; NC433_0_U 3ST-B进出料伸缩伺服错误代码
2019.05 BOOL  ; NC433_0_U 3ST-B进出料伸缩伺服错误代码
2019.06 BOOL  ; NC433_0_U 3ST-B进出料伸缩伺服错误代码
2019.07 BOOL  ; NC433_0_U 3ST-B进出料伸缩伺服错误代码
2019.08 BOOL  ; NC433_0_U 3ST-B进出料伸缩伺服错误代码
2019.09 BOOL  ; NC433_0_U 3ST-B进出料伸缩伺服错误代码
2019.10 BOOL  ; NC433_0_U 3ST-B进出料伸缩伺服错误代码
2019.11 BOOL  ; NC433_0_U 3ST-B进出料伸缩伺服错误代码
2019.12 BOOL  ; NC433_0_U 3ST-B进出料伸缩伺服错误代码
2019.13 BOOL  ; NC433_0_U 3ST-B进出料伸缩伺服错误代码
2019.14 BOOL  ; NC433_0_U 3ST-B进出料伸缩伺服错误代码
2019.15 BOOL  ; NC433_0_U 3ST-B进出料伸缩伺服错误代码
2020.00 BOOL  ; NC433_1_X 4ST_A正压伺服A存储器操作命令激活序列数
2020.01 BOOL  ; NC433_1_X 4ST_A正压伺服A存储器操作命令起动
2020.02 BOOL  ; NC433_1_X 4ST_A正压伺服A存储器操作命令独立起动
2020.03 BOOL  ; NC433_1_X 4ST_A正压伺服A直接操作命令绝对移动
2020.04 BOOL  ; NC433_1_X 4ST_A正压伺服A直接操作命令相对移动
2020.05 BOOL  ; NC433_1_X 4ST_A正压伺服A直接操作命令中断进给
2020.06 BOOL  ; NC433_1_X 4ST_A正压伺服A原点定位命令原点搜索
2020.07 BOOL  ; NC433_1_X 4ST_A正压伺服A原点定位命令原点返回
2020.08 BOOL  ; NC433_1_X 4ST_A正压伺服A原点定位命令当前位置预置
2020.09 BOOL  ; NC433_1_X 4ST_A正压伺服A点动
2020.10 BOOL  ; NC433_1_X 4ST_A正压伺服A点动方向(0=CW,1=CCW)
2020.11 BOOL  ; NC433_1_X 4ST_A正压伺服A示教
2020.12 BOOL  ; NC433_1_X 4ST_A正压伺服A错误清除
2020.13 BOOL  ; NC433_1_X 4ST_A正压伺服A偏差计数器复位输出/ 原点调整命令输出
2020.14 BOOL  ; NC433_1_X 4ST_A正压伺服A激活Override
2020.15 BOOL  ; NC433_1_X 4ST_A正压伺服A停止
2021.00 BOOL  ; NC433_1_X 4ST_A正压伺服A预留
2021.01 BOOL  ; NC433_1_X 4ST_A正压伺服A预留
2021.02 BOOL  ; NC433_1_X 4ST_A正压伺服A预留
2021.03 BOOL  ; NC433_1_X 4ST_A正压伺服A预留
2021.04 BOOL  ; NC433_1_X 4ST_A正压伺服A预留
2021.05 BOOL  ; NC433_1_X 4ST_A正压伺服A预留
2021.06 BOOL  ; NC433_1_X 4ST_A正压伺服A预留
2021.07 BOOL  ; NC433_1_X 4ST_A正压伺服A预留
2021.08 BOOL  ; NC433_1_X 4ST_A正压伺服A强制中断
2021.09 BOOL  ; NC433_1_X 4ST_A正压伺服A预留
2021.10 BOOL  ; NC433_1_X 4ST_A正压伺服A预留
2021.11 BOOL  ; NC433_1_X 4ST_A正压伺服A预留
2021.12 BOOL  ; NC433_1_X 4ST_A正压伺服A数据写入
2021.13 BOOL  ; NC433_1_X 4ST_A正压伺服A数据读出
2021.14 BOOL  ; NC433_1_X 4ST_A正压伺服A数据保存
2021.15 BOOL  ; NC433_1_X 4ST_A正压伺服A预留
2022.00 BOOL  ; NC433_1_Y 4ST_A压板平移伺服存储器操作命令激活序列数
2022.01 BOOL  ; NC433_1_Y 4ST_A压板平移伺服存储器操作命令起动
2022.02 BOOL  ; NC433_1_Y 4ST_A压板平移伺服存储器操作命令独立起动
2022.03 BOOL  ; NC433_1_Y 4ST_A压板平移伺服直接操作命令绝对移动
2022.04 BOOL  ; NC433_1_Y 4ST_A压板平移伺服直接操作命令相对移动
2022.05 BOOL  ; NC433_1_Y 4ST_A压板平移伺服直接操作命令中断进给
2022.06 BOOL  ; NC433_1_Y 4ST_A压板平移伺服原点定位命令原点搜索
2022.07 BOOL  ; NC433_1_Y 4ST_A压板平移伺服原点定位命令原点返回
2022.08 BOOL  ; NC433_1_Y 4ST_A压板平移伺服原点定位命令当前位置预置
2022.09 BOOL  ; NC433_1_Y 4ST_A压板平移伺服点动
2022.10 BOOL  ; NC433_1_Y 4ST_A压板平移伺服点动方向(0=CW,1=CCW)
2022.11 BOOL  ; NC433_1_Y 4ST_A压板平移伺服示教
2022.12 BOOL  ; NC433_1_Y 4ST_A压板平移伺服错误清除
2022.13 BOOL  ; NC433_1_Y 4ST_A压板平移伺服偏差计数器复位输出/ 原点调整命令输出
2022.14 BOOL  ; NC433_1_Y 4ST_A压板平移伺服激活Override
2022.15 BOOL  ; NC433_1_Y 4ST_A压板平移伺服停止
2023.00 BOOL  ; NC433_1_Y 4ST_A压板平移伺服预留
2023.01 BOOL  ; NC433_1_Y 4ST_A压板平移伺服预留
2023.02 BOOL  ; NC433_1_Y 4ST_A压板平移伺服预留
2023.03 BOOL  ; NC433_1_Y 4ST_A压板平移伺服预留
2023.04 BOOL  ; NC433_1_Y 4ST_A压板平移伺服预留
2023.05 BOOL  ; NC433_1_Y 4ST_A压板平移伺服预留
2023.06 BOOL  ; NC433_1_Y 4ST_A压板平移伺服预留
2023.07 BOOL  ; NC433_1_Y 4ST_A压板平移伺服预留
2023.08 BOOL  ; NC433_1_Y 4ST_A压板平移伺服强制中断
2023.09 BOOL  ; NC433_1_Y 4ST_A压板平移伺服预留
2023.10 BOOL  ; NC433_1_Y 4ST_A压板平移伺服预留
2023.11 BOOL  ; NC433_1_Y 4ST_A压板平移伺服预留
2023.12 BOOL  ; NC433_1_Y 4ST_A压板平移伺服数据写入
2023.13 BOOL  ; NC433_1_Y 4ST_A压板平移伺服数据读出
2023.14 BOOL  ; NC433_1_Y 4ST_A压板平移伺服数据保存
2023.15 BOOL  ; NC433_1_Y 4ST_A压板平移伺服预留
2024.00 BOOL  ; NC433_1_Z 4ST_A侧压A1左伺服存储器操作命令激活序列数
2024.01 BOOL  ; NC433_1_Z 4ST_A侧压A1左伺服存储器操作命令起动
2024.02 BOOL  ; NC433_1_Z 4ST_A侧压A1左伺服存储器操作命令独立起动
2024.03 BOOL  ; NC433_1_Z 4ST_A侧压A1左伺服直接操作命令绝对移动
2024.04 BOOL  ; NC433_1_Z 4ST_A侧压A1左伺服直接操作命令相对移动
2024.05 BOOL  ; NC433_1_Z 4ST_A侧压A1左伺服直接操作命令中断进给
2024.06 BOOL  ; NC433_1_Z 4ST_A侧压A1左伺服原点定位命令原点搜索
2024.07 BOOL  ; NC433_1_Z 4ST_A侧压A1左伺服原点定位命令原点返回
2024.08 BOOL  ; NC433_1_Z 4ST_A侧压A1左伺服原点定位命令当前位置预置
2024.09 BOOL  ; NC433_1_Z 4ST_A侧压A1左伺服点动
2024.10 BOOL  ; NC433_1_Z 4ST_A侧压A1左伺服点动方向(0=CW,1=CCW)
2024.11 BOOL  ; NC433_1_Z 4ST_A侧压A1左伺服示教
2024.12 BOOL  ; NC433_1_Z 4ST_A侧压A1左伺服错误清除
2024.13 BOOL  ; NC433_1_Z 4ST_A侧压A1左伺服偏差计数器复位输出/ 原点调整命令输出
2024.14 BOOL  ; NC433_1_Z 4ST_A侧压A1左伺服激活Override
2024.15 BOOL  ; NC433_1_Z 4ST_A侧压A1左伺服停止
2025.00 BOOL  ; NC433_1_Z 4ST_A侧压A1左伺服预留
2025.01 BOOL  ; NC433_1_Z 4ST_A侧压A1左伺服预留
2025.02 BOOL  ; NC433_1_Z 4ST_A侧压A1左伺服预留
2025.03 BOOL  ; NC433_1_Z 4ST_A侧压A1左伺服预留
2025.04 BOOL  ; NC433_1_Z 4ST_A侧压A1左伺服预留
2025.05 BOOL  ; NC433_1_Z 4ST_A侧压A1左伺服预留
2025.06 BOOL  ; NC433_1_Z 4ST_A侧压A1左伺服预留
2025.07 BOOL  ; NC433_1_Z 4ST_A侧压A1左伺服预留
2025.08 BOOL  ; NC433_1_Z 4ST_A侧压A1左伺服强制中断
2025.09 BOOL  ; NC433_1_Z 4ST_A侧压A1左伺服预留
2025.10 BOOL  ; NC433_1_Z 4ST_A侧压A1左伺服预留
2025.11 BOOL  ; NC433_1_Z 4ST_A侧压A1左伺服预留
2025.12 BOOL  ; NC433_1_Z 4ST_A侧压A1左伺服数据写入
2025.13 BOOL  ; NC433_1_Z 4ST_A侧压A1左伺服数据读出
2025.14 BOOL  ; NC433_1_Z 4ST_A侧压A1左伺服数据保存
2025.15 BOOL  ; NC433_1_Z 4ST_A侧压A1左伺服预留
2026.00 BOOL  ; NC433_1 4ST_A侧压A1右伺服存储器操作命令激活序列数
2026.01 BOOL  ; NC433_1 4ST_A侧压A1右伺服存储器操作命令起动
2026.02 BOOL  ; NC433_1 4ST_A侧压A1右伺服存储器操作命令独立起动
2026.03 BOOL  ; NC433_1 4ST_A侧压A1右伺服直接操作命令绝对移动
2026.04 BOOL  ; NC433_1 4ST_A侧压A1右伺服直接操作命令相对移动
2026.05 BOOL  ; NC433_1 4ST_A侧压A1右伺服直接操作命令中断进给
2026.06 BOOL  ; NC433_1 4ST_A侧压A1右伺服原点定位命令原点搜索
2026.07 BOOL  ; NC433_1 4ST_A侧压A1右伺服原点定位命令原点返回
2026.08 BOOL  ; NC433_1 4ST_A侧压A1右伺服原点定位命令当前位置预置
2026.09 BOOL  ; NC433_1 4ST_A侧压A1右伺服点动
2026.10 BOOL  ; NC433_1 4ST_A侧压A1右伺服点动方向(0=CW,1=CCW)
2026.11 BOOL  ; NC433_1 4ST_A侧压A1右伺服示教
2026.12 BOOL  ; NC433_1 4ST_A侧压A1右伺服错误清除
2026.13 BOOL  ; NC433_1 4ST_A侧压A1右伺服偏差计数器复位输出/ 原点调整命令输出
2026.14 BOOL  ; NC433_1 4ST_A侧压A1右伺服激活Override
2026.15 BOOL  ; NC433_1 4ST_A侧压A1右伺服停止
2027.00 BOOL  ; NC433_1 4ST_A侧压A1右伺服预留
2027.01 BOOL  ; NC433_1 4ST_A侧压A1右伺服预留
2027.02 BOOL  ; NC433_1 4ST_A侧压A1右伺服预留
2027.03 BOOL  ; NC433_1 4ST_A侧压A1右伺服预留
2027.04 BOOL  ; NC433_1 4ST_A侧压A1右伺服预留
2027.05 BOOL  ; NC433_1 4ST_A侧压A1右伺服预留
2027.06 BOOL  ; NC433_1 4ST_A侧压A1右伺服预留
2027.07 BOOL  ; NC433_1 4ST_A侧压A1右伺服预留
2027.08 BOOL  ; NC433_1 4ST_A侧压A1右伺服强制中断
2027.09 BOOL  ; NC433_1 4ST_A侧压A1右伺服预留
2027.10 BOOL  ; NC433_1 4ST_A侧压A1右伺服预留
2027.11 BOOL  ; NC433_1 4ST_A侧压A1右伺服预留
2027.12 BOOL  ; NC433_1 4ST_A侧压A1右伺服数据写入
2027.13 BOOL  ; NC433_1 4ST_A侧压A1右伺服数据读出
2027.14 BOOL  ; NC433_1 4ST_A侧压A1右伺服数据保存
2027.15 BOOL  ; NC433_1 4ST_A侧压A1右伺服预留
2028.00 BOOL  ; NC433_1_X 4ST_A正压伺服A预留
2028.01 BOOL  ; NC433_1_X 4ST_A正压伺服A预留
2028.02 BOOL  ; NC433_1_X 4ST_A正压伺服A预留
2028.03 BOOL  ; NC433_1_X 4ST_A正压伺服A预留
2028.04 BOOL  ; NC433_1_X 4ST_A正压伺服A等待存储器操作
2028.05 BOOL  ; NC433_1_X 4ST_A正压伺服A定位完成标志位
2028.06 BOOL  ; NC433_1_X 4ST_A正压伺服A无原点标志位
2028.07 BOOL  ; NC433_1_X 4ST_A正压伺服A原点停止标志位
2028.08 BOOL  ; NC433_1_X 4ST_A正压伺服A0 区监测标志位
2028.09 BOOL  ; NC433_1_X 4ST_A正压伺服A1 区监测标志位
2028.10 BOOL  ; NC433_1_X 4ST_A正压伺服A2 区监测标志位
2028.11 BOOL  ; NC433_1_X 4ST_A正压伺服A示教完成
2028.12 BOOL  ; NC433_1_X 4ST_A正压伺服A错误标志
2028.13 BOOL  ; NC433_1_X 4ST_A正压伺服A忙标志
2028.14 BOOL  ; NC433_1_X 4ST_A正压伺服A数据传送标志位
2028.15 BOOL  ; NC433_1_X 4ST_A正压伺服A减速停止执行标志位
2029.00 BOOL  ; NC433_1_X 4ST_A正压伺服A预留
2029.01 BOOL  ; NC433_1_X 4ST_A正压伺服A预留
2029.02 BOOL  ; NC433_1_X 4ST_A正压伺服A预留
2029.03 BOOL  ; NC433_1_X 4ST_A正压伺服A预留
2029.04 BOOL  ; NC433_1_X 4ST_A正压伺服A预留
2029.05 BOOL  ; NC433_1_X 4ST_A正压伺服A预留
2029.06 BOOL  ; NC433_1_X 4ST_A正压伺服A预留
2029.07 BOOL  ; NC433_1_X 4ST_A正压伺服A预留
2029.08 BOOL  ; NC433_1_X 4ST_A正压伺服ACW极限输入信号
2029.09 BOOL  ; NC433_1_X 4ST_A正压伺服ACCW极限输入信号
2029.10 BOOL  ; NC433_1_X 4ST_A正压伺服A原点接近输入信号
2029.11 BOOL  ; NC433_1_X 4ST_A正压伺服A原点输入信号
2029.12 BOOL  ; NC433_1_X 4ST_A正压伺服A中断输入信号
2029.13 BOOL  ; NC433_1_X 4ST_A正压伺服A紧急输入信号
2029.14 BOOL  ; NC433_1_X 4ST_A正压伺服A定位完成输入信号
2029.15 BOOL  ; NC433_1_X 4ST_A正压伺服A偏差计数器复位输出/ 原点调整命令输出
2030.00 BOOL  ; NC433_1_X 4ST_A正压伺服A错误代码
2030.01 BOOL  ; NC433_1_X 4ST_A正压伺服A错误代码
2030.02 BOOL  ; NC433_1_X 4ST_A正压伺服A错误代码
2030.03 BOOL  ; NC433_1_X 4ST_A正压伺服A错误代码
2030.04 BOOL  ; NC433_1_X 4ST_A正压伺服A错误代码
2030.05 BOOL  ; NC433_1_X 4ST_A正压伺服A错误代码
2030.06 BOOL  ; NC433_1_X 4ST_A正压伺服A错误代码
2030.07 BOOL  ; NC433_1_X 4ST_A正压伺服A错误代码
2030.08 BOOL  ; NC433_1_X 4ST_A正压伺服A错误代码
2030.09 BOOL  ; NC433_1_X 4ST_A正压伺服A错误代码
2030.10 BOOL  ; NC433_1_X 4ST_A正压伺服A错误代码
2030.11 BOOL  ; NC433_1_X 4ST_A正压伺服A错误代码
2030.12 BOOL  ; NC433_1_X 4ST_A正压伺服A错误代码
2030.13 BOOL  ; NC433_1_X 4ST_A正压伺服A错误代码
2030.14 BOOL  ; NC433_1_X 4ST_A正压伺服A错误代码
2030.15 BOOL  ; NC433_1_X 4ST_A正压伺服A错误代码
2031.00 BOOL  ; NC433_1_Y 4ST_A压板平移伺服预留
2031.01 BOOL  ; NC433_1_Y 4ST_A压板平移伺服预留
2031.02 BOOL  ; NC433_1_Y 4ST_A压板平移伺服预留
2031.03 BOOL  ; NC433_1_Y 4ST_A压板平移伺服预留
2031.04 BOOL  ; NC433_1_Y 4ST_A压板平移伺服等待存储器操作
2031.05 BOOL  ; NC433_1_Y 4ST_A压板平移伺服定位完成标志位
2031.06 BOOL  ; NC433_1_Y 4ST_A压板平移伺服无原点标志位
2031.07 BOOL  ; NC433_1_Y 4ST_A压板平移伺服原点停止标志位
2031.08 BOOL  ; NC433_1_Y 4ST_A压板平移伺服0 区监测标志位
2031.09 BOOL  ; NC433_1_Y 4ST_A压板平移伺服1 区监测标志位
2031.10 BOOL  ; NC433_1_Y 4ST_A压板平移伺服2 区监测标志位
2031.11 BOOL  ; NC433_1_Y 4ST_A压板平移伺服示教完成
2031.12 BOOL  ; NC433_1_Y 4ST_A压板平移伺服错误标志
2031.13 BOOL  ; NC433_1_Y 4ST_A压板平移伺服忙标志
2031.14 BOOL  ; NC433_1_Y 4ST_A压板平移伺服数据传送标志位
2031.15 BOOL  ; NC433_1_Y 4ST_A压板平移伺服减速停止执行标志位
2032.00 BOOL  ; NC433_1_Y 4ST_A压板平移伺服预留
2032.01 BOOL  ; NC433_1_Y 4ST_A压板平移伺服预留
2032.02 BOOL  ; NC433_1_Y 4ST_A压板平移伺服预留
2032.03 BOOL  ; NC433_1_Y 4ST_A压板平移伺服预留
2032.04 BOOL  ; NC433_1_Y 4ST_A压板平移伺服预留
2032.05 BOOL  ; NC433_1_Y 4ST_A压板平移伺服预留
2032.06 BOOL  ; NC433_1_Y 4ST_A压板平移伺服预留
2032.07 BOOL  ; NC433_1_Y 4ST_A压板平移伺服预留
2032.08 BOOL  ; NC433_1_Y 4ST_A压板平移伺服CW极限输入信号
2032.09 BOOL  ; NC433_1_Y 4ST_A压板平移伺服CCW极限输入信号
2032.10 BOOL  ; NC433_1_Y 4ST_A压板平移伺服原点接近输入信号
2032.11 BOOL  ; NC433_1_Y 4ST_A压板平移伺服原点输入信号
2032.12 BOOL  ; NC433_1_Y 4ST_A压板平移伺服中断输入信号
2032.13 BOOL  ; NC433_1_Y 4ST_A压板平移伺服紧急输入信号
2032.14 BOOL  ; NC433_1_Y 4ST_A压板平移伺服定位完成输入信号
2032.15 BOOL  ; NC433_1_Y 4ST_A压板平移伺服偏差计数器复位输出/ 原点调整命令输出
2033.00 BOOL  ; NC433_1_Y 4ST_A压板平移伺服错误代码
2033.01 BOOL  ; NC433_1_Y 4ST_A压板平移伺服错误代码
2033.02 BOOL  ; NC433_1_Y 4ST_A压板平移伺服错误代码
2033.03 BOOL  ; NC433_1_Y 4ST_A压板平移伺服错误代码
2033.04 BOOL  ; NC433_1_Y 4ST_A压板平移伺服错误代码
2033.05 BOOL  ; NC433_1_Y 4ST_A压板平移伺服错误代码
2033.06 BOOL  ; NC433_1_Y 4ST_A压板平移伺服错误代码
2033.07 BOOL  ; NC433_1_Y 4ST_A压板平移伺服错误代码
2033.08 BOOL  ; NC433_1_Y 4ST_A压板平移伺服错误代码
2033.09 BOOL  ; NC433_1_Y 4ST_A压板平移伺服错误代码
2033.10 BOOL  ; NC433_1_Y 4ST_A压板平移伺服错误代码
2033.11 BOOL  ; NC433_1_Y 4ST_A压板平移伺服错误代码
2033.12 BOOL  ; NC433_1_Y 4ST_A压板平移伺服错误代码
2033.13 BOOL  ; NC433_1_Y 4ST_A压板平移伺服错误代码
2033.14 BOOL  ; NC433_1_Y 4ST_A压板平移伺服错误代码
2033.15 BOOL  ; NC433_1_Y 4ST_A压板平移伺服错误代码
2034.00 BOOL  ; NC433_1_Z 4ST_A侧压A1左伺服预留
2034.01 BOOL  ; NC433_1_Z 4ST_A侧压A1左伺服预留
2034.02 BOOL  ; NC433_1_Z 4ST_A侧压A1左伺服预留
2034.03 BOOL  ; NC433_1_Z 4ST_A侧压A1左伺服预留
2034.04 BOOL  ; NC433_1_Z 4ST_A侧压A1左伺服等待存储器操作
2034.05 BOOL  ; NC433_1_Z 4ST_A侧压A1左伺服定位完成标志位
2034.06 BOOL  ; NC433_1_Z 4ST_A侧压A1左伺服无原点标志位
2034.07 BOOL  ; NC433_1_Z 4ST_A侧压A1左伺服原点停止标志位
2034.08 BOOL  ; NC433_1_Z 4ST_A侧压A1左伺服0 区监测标志位
2034.09 BOOL  ; NC433_1_Z 4ST_A侧压A1左伺服1 区监测标志位
2034.10 BOOL  ; NC433_1_Z 4ST_A侧压A1左伺服2 区监测标志位
2034.11 BOOL  ; NC433_1_Z 4ST_A侧压A1左伺服示教完成
2034.12 BOOL  ; NC433_1_Z 4ST_A侧压A1左伺服错误标志
2034.13 BOOL  ; NC433_1_Z 4ST_A侧压A1左伺服忙标志
2034.14 BOOL  ; NC433_1_Z 4ST_A侧压A1左伺服数据传送标志位
2034.15 BOOL  ; NC433_1_Z 4ST_A侧压A1左伺服减速停止执行标志位
2035.00 BOOL  ; NC433_1_Z 4ST_A侧压A1左伺服预留
2035.01 BOOL  ; NC433_1_Z 4ST_A侧压A1左伺服预留
2035.02 BOOL  ; NC433_1_Z 4ST_A侧压A1左伺服预留
2035.03 BOOL  ; NC433_1_Z 4ST_A侧压A1左伺服预留
2035.04 BOOL  ; NC433_1_Z 4ST_A侧压A1左伺服预留
2035.05 BOOL  ; NC433_1_Z 4ST_A侧压A1左伺服预留
2035.06 BOOL  ; NC433_1_Z 4ST_A侧压A1左伺服预留
2035.07 BOOL  ; NC433_1_Z 4ST_A侧压A1左伺服预留
2035.08 BOOL  ; NC433_1_Z 4ST_A侧压A1左伺服CW极限输入信号
2035.09 BOOL  ; NC433_1_Z 4ST_A侧压A1左伺服CCW极限输入信号
2035.10 BOOL  ; NC433_1_Z 4ST_A侧压A1左伺服原点接近输入信号
2035.11 BOOL  ; NC433_1_Z 4ST_A侧压A1左伺服原点输入信号
2035.12 BOOL  ; NC433_1_Z 4ST_A侧压A1左伺服中断输入信号
2035.13 BOOL  ; NC433_1_Z 4ST_A侧压A1左伺服紧急输入信号
2035.14 BOOL  ; NC433_1_Z 4ST_A侧压A1左伺服定位完成输入信号
2035.15 BOOL  ; NC433_1_Z 4ST_A侧压A1左伺服偏差计数器复位输出/ 原点调整命令输出
2036.00 BOOL  ; NC433_1_Z 4ST_A侧压A1左伺服错误代码
2036.01 BOOL  ; NC433_1_Z 4ST_A侧压A1左伺服错误代码
2036.02 BOOL  ; NC433_1_Z 4ST_A侧压A1左伺服错误代码
2036.03 BOOL  ; NC433_1_Z 4ST_A侧压A1左伺服错误代码
2036.04 BOOL  ; NC433_1_Z 4ST_A侧压A1左伺服错误代码
2036.05 BOOL  ; NC433_1_Z 4ST_A侧压A1左伺服错误代码
2036.06 BOOL  ; NC433_1_Z 4ST_A侧压A1左伺服错误代码
2036.07 BOOL  ; NC433_1_Z 4ST_A侧压A1左伺服错误代码
2036.08 BOOL  ; NC433_1_Z 4ST_A侧压A1左伺服错误代码
2036.09 BOOL  ; NC433_1_Z 4ST_A侧压A1左伺服错误代码
2036.10 BOOL  ; NC433_1_Z 4ST_A侧压A1左伺服错误代码
2036.11 BOOL  ; NC433_1_Z 4ST_A侧压A1左伺服错误代码
2036.12 BOOL  ; NC433_1_Z 4ST_A侧压A1左伺服错误代码
2036.13 BOOL  ; NC433_1_Z 4ST_A侧压A1左伺服错误代码
2036.14 BOOL  ; NC433_1_Z 4ST_A侧压A1左伺服错误代码
2036.15 BOOL  ; NC433_1_Z 4ST_A侧压A1左伺服错误代码
2037.00 BOOL  ; NC433_1 4ST_A侧压A1右伺服预留
2037.01 BOOL  ; NC433_1 4ST_A侧压A1右伺服预留
2037.02 BOOL  ; NC433_1 4ST_A侧压A1右伺服预留
2037.03 BOOL  ; NC433_1 4ST_A侧压A1右伺服预留
2037.04 BOOL  ; NC433_1 4ST_A侧压A1右伺服等待存储器操作
2037.05 BOOL  ; NC433_1 4ST_A侧压A1右伺服定位完成标志位
2037.06 BOOL  ; NC433_1 4ST_A侧压A1右伺服无原点标志位
2037.07 BOOL  ; NC433_1 4ST_A侧压A1右伺服原点停止标志位
2037.08 BOOL  ; NC433_1 4ST_A侧压A1右伺服0 区监测标志位
2037.09 BOOL  ; NC433_1 4ST_A侧压A1右伺服1 区监测标志位
2037.10 BOOL  ; NC433_1 4ST_A侧压A1右伺服2 区监测标志位
2037.11 BOOL  ; NC433_1 4ST_A侧压A1右伺服示教完成
2037.12 BOOL  ; NC433_1 4ST_A侧压A1右伺服错误标志
2037.13 BOOL  ; NC433_1 4ST_A侧压A1右伺服忙标志
2037.14 BOOL  ; NC433_1 4ST_A侧压A1右伺服数据传送标志位
2037.15 BOOL  ; NC433_1 4ST_A侧压A1右伺服减速停止执行标志位
2038.00 BOOL  ; NC433_1 4ST_A侧压A1右伺服预留
2038.01 BOOL  ; NC433_1 4ST_A侧压A1右伺服预留
2038.02 BOOL  ; NC433_1 4ST_A侧压A1右伺服预留
2038.03 BOOL  ; NC433_1 4ST_A侧压A1右伺服预留
2038.04 BOOL  ; NC433_1 4ST_A侧压A1右伺服预留
2038.05 BOOL  ; NC433_1 4ST_A侧压A1右伺服预留
2038.06 BOOL  ; NC433_1 4ST_A侧压A1右伺服预留
2038.07 BOOL  ; NC433_1 4ST_A侧压A1右伺服预留
2038.08 BOOL  ; NC433_1 4ST_A侧压A1右伺服CW极限输入信号
2038.09 BOOL  ; NC433_1 4ST_A侧压A1右伺服CCW极限输入信号
2038.10 BOOL  ; NC433_1 4ST_A侧压A1右伺服原点接近输入信号
2038.11 BOOL  ; NC433_1 4ST_A侧压A1右伺服原点输入信号
2038.12 BOOL  ; NC433_1 4ST_A侧压A1右伺服中断输入信号
2038.13 BOOL  ; NC433_1 4ST_A侧压A1右伺服紧急输入信号
2038.14 BOOL  ; NC433_1 4ST_A侧压A1右伺服定位完成输入信号
2038.15 BOOL  ; NC433_1 4ST_A侧压A1右伺服偏差计数器复位输出/ 原点调整命令输出
2039.00 BOOL  ; NC433_1 4ST_A侧压A1右伺服错误代码
2039.01 BOOL  ; NC433_1 4ST_A侧压A1右伺服错误代码
2039.02 BOOL  ; NC433_1 4ST_A侧压A1右伺服错误代码
2039.03 BOOL  ; NC433_1 4ST_A侧压A1右伺服错误代码
2039.04 BOOL  ; NC433_1 4ST_A侧压A1右伺服错误代码
2039.05 BOOL  ; NC433_1 4ST_A侧压A1右伺服错误代码
2039.06 BOOL  ; NC433_1 4ST_A侧压A1右伺服错误代码
2039.07 BOOL  ; NC433_1 4ST_A侧压A1右伺服错误代码
2039.08 BOOL  ; NC433_1 4ST_A侧压A1右伺服错误代码
2039.09 BOOL  ; NC433_1 4ST_A侧压A1右伺服错误代码
2039.10 BOOL  ; NC433_1 4ST_A侧压A1右伺服错误代码
2039.11 BOOL  ; NC433_1 4ST_A侧压A1右伺服错误代码
2039.12 BOOL  ; NC433_1 4ST_A侧压A1右伺服错误代码
2039.13 BOOL  ; NC433_1 4ST_A侧压A1右伺服错误代码
2039.14 BOOL  ; NC433_1 4ST_A侧压A1右伺服错误代码
2039.15 BOOL  ; NC433_1 4ST_A侧压A1右伺服错误代码
2040.00 BOOL  ; NC433_2_X 4ST_A侧压A2左伺服存储器操作命令激活序列数
2040.01 BOOL  ; NC433_2_X 4ST_A侧压A2左伺服存储器操作命令起动
2040.02 BOOL  ; NC433_2_X 4ST_A侧压A2左伺服存储器操作命令独立起动
2040.03 BOOL  ; NC433_2_X 4ST_A侧压A2左伺服直接操作命令绝对移动
2040.04 BOOL  ; NC433_2_X 4ST_A侧压A2左伺服直接操作命令相对移动
2040.05 BOOL  ; NC433_2_X 4ST_A侧压A2左伺服直接操作命令中断进给
2040.06 BOOL  ; NC433_2_X 4ST_A侧压A2左伺服原点定位命令原点搜索
2040.07 BOOL  ; NC433_2_X 4ST_A侧压A2左伺服原点定位命令原点返回
2040.08 BOOL  ; NC433_2_X 4ST_A侧压A2左伺服原点定位命令当前位置预置
2040.09 BOOL  ; NC433_2_X 4ST_A侧压A2左伺服点动
2040.10 BOOL  ; NC433_2_X 4ST_A侧压A2左伺服点动方向(0=CW,1=CCW)
2040.11 BOOL  ; NC433_2_X 4ST_A侧压A2左伺服示教
2040.12 BOOL  ; NC433_2_X 4ST_A侧压A2左伺服错误清除
2040.13 BOOL  ; NC433_2_X 4ST_A侧压A2左伺服偏差计数器复位输出/ 原点调整命令输出
2040.14 BOOL  ; NC433_2_X 4ST_A侧压A2左伺服激活Override
2040.15 BOOL  ; NC433_2_X 4ST_A侧压A2左伺服停止
2041.00 BOOL  ; NC433_2_X 4ST_A侧压A2左伺服预留
2041.01 BOOL  ; NC433_2_X 4ST_A侧压A2左伺服预留
2041.02 BOOL  ; NC433_2_X 4ST_A侧压A2左伺服预留
2041.03 BOOL  ; NC433_2_X 4ST_A侧压A2左伺服预留
2041.04 BOOL  ; NC433_2_X 4ST_A侧压A2左伺服预留
2041.05 BOOL  ; NC433_2_X 4ST_A侧压A2左伺服预留
2041.06 BOOL  ; NC433_2_X 4ST_A侧压A2左伺服预留
2041.07 BOOL  ; NC433_2_X 4ST_A侧压A2左伺服预留
2041.08 BOOL  ; NC433_2_X 4ST_A侧压A2左伺服强制中断
2041.09 BOOL  ; NC433_2_X 4ST_A侧压A2左伺服预留
2041.10 BOOL  ; NC433_2_X 4ST_A侧压A2左伺服预留
2041.11 BOOL  ; NC433_2_X 4ST_A侧压A2左伺服预留
2041.12 BOOL  ; NC433_2_X 4ST_A侧压A2左伺服数据写入
2041.13 BOOL  ; NC433_2_X 4ST_A侧压A2左伺服数据读出
2041.14 BOOL  ; NC433_2_X 4ST_A侧压A2左伺服数据保存
2041.15 BOOL  ; NC433_2_X 4ST_A侧压A2左伺服预留
2042.00 BOOL  ; NC433_2_Y 4ST_A侧压A2右伺服存储器操作命令激活序列数
2042.01 BOOL  ; NC433_2_Y 4ST_A侧压A2右伺服存储器操作命令起动
2042.02 BOOL  ; NC433_2_Y 4ST_A侧压A2右伺服存储器操作命令独立起动
2042.03 BOOL  ; NC433_2_Y 4ST_A侧压A2右伺服直接操作命令绝对移动
2042.04 BOOL  ; NC433_2_Y 4ST_A侧压A2右伺服直接操作命令相对移动
2042.05 BOOL  ; NC433_2_Y 4ST_A侧压A2右伺服直接操作命令中断进给
2042.06 BOOL  ; NC433_2_Y 4ST_A侧压A2右伺服原点定位命令原点搜索
2042.07 BOOL  ; NC433_2_Y 4ST_A侧压A2右伺服原点定位命令原点返回
2042.08 BOOL  ; NC433_2_Y 4ST_A侧压A2右伺服原点定位命令当前位置预置
2042.09 BOOL  ; NC433_2_Y 4ST_A侧压A2右伺服点动
2042.10 BOOL  ; NC433_2_Y 4ST_A侧压A2右伺服点动方向(0=CW,1=CCW)
2042.11 BOOL  ; NC433_2_Y 4ST_A侧压A2右伺服示教
2042.12 BOOL  ; NC433_2_Y 4ST_A侧压A2右伺服错误清除
2042.13 BOOL  ; NC433_2_Y 4ST_A侧压A2右伺服偏差计数器复位输出/ 原点调整命令输出
2042.14 BOOL  ; NC433_2_Y 4ST_A侧压A2右伺服激活Override
2042.15 BOOL  ; NC433_2_Y 4ST_A侧压A2右伺服停止
2043.00 BOOL  ; NC433_2_Y 4ST_A侧压A2右伺服预留
2043.01 BOOL  ; NC433_2_Y 4ST_A侧压A2右伺服预留
2043.02 BOOL  ; NC433_2_Y 4ST_A侧压A2右伺服预留
2043.03 BOOL  ; NC433_2_Y 4ST_A侧压A2右伺服预留
2043.04 BOOL  ; NC433_2_Y 4ST_A侧压A2右伺服预留
2043.05 BOOL  ; NC433_2_Y 4ST_A侧压A2右伺服预留
2043.06 BOOL  ; NC433_2_Y 4ST_A侧压A2右伺服预留
2043.07 BOOL  ; NC433_2_Y 4ST_A侧压A2右伺服预留
2043.08 BOOL  ; NC433_2_Y 4ST_A侧压A2右伺服强制中断
2043.09 BOOL  ; NC433_2_Y 4ST_A侧压A2右伺服预留
2043.10 BOOL  ; NC433_2_Y 4ST_A侧压A2右伺服预留
2043.11 BOOL  ; NC433_2_Y 4ST_A侧压A2右伺服预留
2043.12 BOOL  ; NC433_2_Y 4ST_A侧压A2右伺服数据写入
2043.13 BOOL  ; NC433_2_Y 4ST_A侧压A2右伺服数据读出
2043.14 BOOL  ; NC433_2_Y 4ST_A侧压A2右伺服数据保存
2043.15 BOOL  ; NC433_2_Y 4ST_A侧压A2右伺服预留
2044.00 BOOL  ; NC433_2_Z 4ST_A侧压A3左伺服存储器操作命令激活序列数
2044.01 BOOL  ; NC433_2_Z 4ST_A侧压A3左伺服存储器操作命令起动
2044.02 BOOL  ; NC433_2_Z 4ST_A侧压A3左伺服存储器操作命令独立起动
2044.03 BOOL  ; NC433_2_Z 4ST_A侧压A3左伺服直接操作命令绝对移动
2044.04 BOOL  ; NC433_2_Z 4ST_A侧压A3左伺服直接操作命令相对移动
2044.05 BOOL  ; NC433_2_Z 4ST_A侧压A3左伺服直接操作命令中断进给
2044.06 BOOL  ; NC433_2_Z 4ST_A侧压A3左伺服原点定位命令原点搜索
2044.07 BOOL  ; NC433_2_Z 4ST_A侧压A3左伺服原点定位命令原点返回
2044.08 BOOL  ; NC433_2_Z 4ST_A侧压A3左伺服原点定位命令当前位置预置
2044.09 BOOL  ; NC433_2_Z 4ST_A侧压A3左伺服点动
2044.10 BOOL  ; NC433_2_Z 4ST_A侧压A3左伺服点动方向(0=CW,1=CCW)
2044.11 BOOL  ; NC433_2_Z 4ST_A侧压A3左伺服示教
2044.12 BOOL  ; NC433_2_Z 4ST_A侧压A3左伺服错误清除
2044.13 BOOL  ; NC433_2_Z 4ST_A侧压A3左伺服偏差计数器复位输出/ 原点调整命令输出
2044.14 BOOL  ; NC433_2_Z 4ST_A侧压A3左伺服激活Override
2044.15 BOOL  ; NC433_2_Z 4ST_A侧压A3左伺服停止
2045.00 BOOL  ; NC433_2_Z 4ST_A侧压A3左伺服预留
2045.01 BOOL  ; NC433_2_Z 4ST_A侧压A3左伺服预留
2045.02 BOOL  ; NC433_2_Z 4ST_A侧压A3左伺服预留
2045.03 BOOL  ; NC433_2_Z 4ST_A侧压A3左伺服预留
2045.04 BOOL  ; NC433_2_Z 4ST_A侧压A3左伺服预留
2045.05 BOOL  ; NC433_2_Z 4ST_A侧压A3左伺服预留
2045.06 BOOL  ; NC433_2_Z 4ST_A侧压A3左伺服预留
2045.07 BOOL  ; NC433_2_Z 4ST_A侧压A3左伺服预留
2045.08 BOOL  ; NC433_2_Z 4ST_A侧压A3左伺服强制中断
2045.09 BOOL  ; NC433_2_Z 4ST_A侧压A3左伺服预留
2045.10 BOOL  ; NC433_2_Z 4ST_A侧压A3左伺服预留
2045.11 BOOL  ; NC433_2_Z 4ST_A侧压A3左伺服预留
2045.12 BOOL  ; NC433_2_Z 4ST_A侧压A3左伺服数据写入
2045.13 BOOL  ; NC433_2_Z 4ST_A侧压A3左伺服数据读出
2045.14 BOOL  ; NC433_2_Z 4ST_A侧压A3左伺服数据保存
2045.15 BOOL  ; NC433_2_Z 4ST_A侧压A3左伺服预留
2046.00 BOOL  ; NC433_2_U 4ST_A侧压A3右伺服存储器操作命令激活序列数
2046.01 BOOL  ; NC433_2_U 4ST_A侧压A3右伺服存储器操作命令起动
2046.02 BOOL  ; NC433_2_U 4ST_A侧压A3右伺服存储器操作命令独立起动
2046.03 BOOL  ; NC433_2_U 4ST_A侧压A3右伺服直接操作命令绝对移动
2046.04 BOOL  ; NC433_2_U 4ST_A侧压A3右伺服直接操作命令相对移动
2046.05 BOOL  ; NC433_2_U 4ST_A侧压A3右伺服直接操作命令中断进给
2046.06 BOOL  ; NC433_2_U 4ST_A侧压A3右伺服原点定位命令原点搜索
2046.07 BOOL  ; NC433_2_U 4ST_A侧压A3右伺服原点定位命令原点返回
2046.08 BOOL  ; NC433_2_U 4ST_A侧压A3右伺服原点定位命令当前位置预置
2046.09 BOOL  ; NC433_2_U 4ST_A侧压A3右伺服点动
2046.10 BOOL  ; NC433_2_U 4ST_A侧压A3右伺服点动方向(0=CW,1=CCW)
2046.11 BOOL  ; NC433_2_U 4ST_A侧压A3右伺服示教
2046.12 BOOL  ; NC433_2_U 4ST_A侧压A3右伺服错误清除
2046.13 BOOL  ; NC433_2_U 4ST_A侧压A3右伺服偏差计数器复位输出/ 原点调整命令输出
2046.14 BOOL  ; NC433_2_U 4ST_A侧压A3右伺服激活Override
2046.15 BOOL  ; NC433_2_U 4ST_A侧压A3右伺服停止
2047.00 BOOL  ; NC433_2_U 4ST_A侧压A3右伺服预留
2047.01 BOOL  ; NC433_2_U 4ST_A侧压A3右伺服预留
2047.02 BOOL  ; NC433_2_U 4ST_A侧压A3右伺服预留
2047.03 BOOL  ; NC433_2_U 4ST_A侧压A3右伺服预留
2047.04 BOOL  ; NC433_2_U 4ST_A侧压A3右伺服预留
2047.05 BOOL  ; NC433_2_U 4ST_A侧压A3右伺服预留
2047.06 BOOL  ; NC433_2_U 4ST_A侧压A3右伺服预留
2047.07 BOOL  ; NC433_2_U 4ST_A侧压A3右伺服预留
2047.08 BOOL  ; NC433_2_U 4ST_A侧压A3右伺服强制中断
2047.09 BOOL  ; NC433_2_U 4ST_A侧压A3右伺服预留
2047.10 BOOL  ; NC433_2_U 4ST_A侧压A3右伺服预留
2047.11 BOOL  ; NC433_2_U 4ST_A侧压A3右伺服预留
2047.12 BOOL  ; NC433_2_U 4ST_A侧压A3右伺服数据写入
2047.13 BOOL  ; NC433_2_U 4ST_A侧压A3右伺服数据读出
2047.14 BOOL  ; NC433_2_U 4ST_A侧压A3右伺服数据保存
2047.15 BOOL  ; NC433_2_U 4ST_A侧压A3右伺服预留
2048.00 BOOL  ; NC433_2_X 4ST_A侧压A2左伺服预留
2048.01 BOOL  ; NC433_2_X 4ST_A侧压A2左伺服预留
2048.02 BOOL  ; NC433_2_X 4ST_A侧压A2左伺服预留
2048.03 BOOL  ; NC433_2_X 4ST_A侧压A2左伺服预留
2048.04 BOOL  ; NC433_2_X 4ST_A侧压A2左伺服等待存储器操作
2048.05 BOOL  ; NC433_2_X 4ST_A侧压A2左伺服定位完成标志位
2048.06 BOOL  ; NC433_2_X 4ST_A侧压A2左伺服无原点标志位
2048.07 BOOL  ; NC433_2_X 4ST_A侧压A2左伺服原点停止标志位
2048.08 BOOL  ; NC433_2_X 4ST_A侧压A2左伺服0 区监测标志位
2048.09 BOOL  ; NC433_2_X 4ST_A侧压A2左伺服1 区监测标志位
2048.10 BOOL  ; NC433_2_X 4ST_A侧压A2左伺服2 区监测标志位
2048.11 BOOL  ; NC433_2_X 4ST_A侧压A2左伺服示教完成
2048.12 BOOL  ; NC433_2_X 4ST_A侧压A2左伺服错误标志
2048.13 BOOL  ; NC433_2_X 4ST_A侧压A2左伺服忙标志
2048.14 BOOL  ; NC433_2_X 4ST_A侧压A2左伺服数据传送标志位
2048.15 BOOL  ; NC433_2_X 4ST_A侧压A2左伺服减速停止执行标志位
2049.00 BOOL  ; NC433_2_X 4ST_A侧压A2左伺服预留
2049.01 BOOL  ; NC433_2_X 4ST_A侧压A2左伺服预留
2049.02 BOOL  ; NC433_2_X 4ST_A侧压A2左伺服预留
2049.03 BOOL  ; NC433_2_X 4ST_A侧压A2左伺服预留
2049.04 BOOL  ; NC433_2_X 4ST_A侧压A2左伺服预留
2049.05 BOOL  ; NC433_2_X 4ST_A侧压A2左伺服预留
2049.06 BOOL  ; NC433_2_X 4ST_A侧压A2左伺服预留
2049.07 BOOL  ; NC433_2_X 4ST_A侧压A2左伺服预留
2049.08 BOOL  ; NC433_2_X 4ST_A侧压A2左伺服CW极限输入信号
2049.09 BOOL  ; NC433_2_X 4ST_A侧压A2左伺服CCW极限输入信号
2049.10 BOOL  ; NC433_2_X 4ST_A侧压A2左伺服原点接近输入信号
2049.11 BOOL  ; NC433_2_X 4ST_A侧压A2左伺服原点输入信号
2049.12 BOOL  ; NC433_2_X 4ST_A侧压A2左伺服中断输入信号
2049.13 BOOL  ; NC433_2_X 4ST_A侧压A2左伺服紧急输入信号
2049.14 BOOL  ; NC433_2_X 4ST_A侧压A2左伺服定位完成输入信号
2049.15 BOOL  ; NC433_2_X 4ST_A侧压A2左伺服偏差计数器复位输出/ 原点调整命令输出
2050.00 BOOL  ; NC433_2_X 4ST_A侧压A2左伺服错误代码
2050.01 BOOL  ; NC433_2_X 4ST_A侧压A2左伺服错误代码
2050.02 BOOL  ; NC433_2_X 4ST_A侧压A2左伺服错误代码
2050.03 BOOL  ; NC433_2_X 4ST_A侧压A2左伺服错误代码
2050.04 BOOL  ; NC433_2_X 4ST_A侧压A2左伺服错误代码
2050.05 BOOL  ; NC433_2_X 4ST_A侧压A2左伺服错误代码
2050.06 BOOL  ; NC433_2_X 4ST_A侧压A2左伺服错误代码
2050.07 BOOL  ; NC433_2_X 4ST_A侧压A2左伺服错误代码
2050.08 BOOL  ; NC433_2_X 4ST_A侧压A2左伺服错误代码
2050.09 BOOL  ; NC433_2_X 4ST_A侧压A2左伺服错误代码
2050.10 BOOL  ; NC433_2_X 4ST_A侧压A2左伺服错误代码
2050.11 BOOL  ; NC433_2_X 4ST_A侧压A2左伺服错误代码
2050.12 BOOL  ; NC433_2_X 4ST_A侧压A2左伺服错误代码
2050.13 BOOL  ; NC433_2_X 4ST_A侧压A2左伺服错误代码
2050.14 BOOL  ; NC433_2_X 4ST_A侧压A2左伺服错误代码
2050.15 BOOL  ; NC433_2_X 4ST_A侧压A2左伺服错误代码
2051.00 BOOL  ; NC433_2_Y 4ST_A侧压A2右伺服预留
2051.01 BOOL  ; NC433_2_Y 4ST_A侧压A2右伺服预留
2051.02 BOOL  ; NC433_2_Y 4ST_A侧压A2右伺服预留
2051.03 BOOL  ; NC433_2_Y 4ST_A侧压A2右伺服预留
2051.04 BOOL  ; NC433_2_Y 4ST_A侧压A2右伺服等待存储器操作
2051.05 BOOL  ; NC433_2_Y 4ST_A侧压A2右伺服定位完成标志位
2051.06 BOOL  ; NC433_2_Y 4ST_A侧压A2右伺服无原点标志位
2051.07 BOOL  ; NC433_2_Y 4ST_A侧压A2右伺服原点停止标志位
2051.08 BOOL  ; NC433_2_Y 4ST_A侧压A2右伺服0 区监测标志位
2051.09 BOOL  ; NC433_2_Y 4ST_A侧压A2右伺服1 区监测标志位
2051.10 BOOL  ; NC433_2_Y 4ST_A侧压A2右伺服2 区监测标志位
2051.11 BOOL  ; NC433_2_Y 4ST_A侧压A2右伺服示教完成
2051.12 BOOL  ; NC433_2_Y 4ST_A侧压A2右伺服错误标志
2051.13 BOOL  ; NC433_2_Y 4ST_A侧压A2右伺服忙标志
2051.14 BOOL  ; NC433_2_Y 4ST_A侧压A2右伺服数据传送标志位
2051.15 BOOL  ; NC433_2_Y 4ST_A侧压A2右伺服减速停止执行标志位
2052.00 BOOL  ; NC433_2_Y 4ST_A侧压A2右伺服预留
2052.01 BOOL  ; NC433_2_Y 4ST_A侧压A2右伺服预留
2052.02 BOOL  ; NC433_2_Y 4ST_A侧压A2右伺服预留
2052.03 BOOL  ; NC433_2_Y 4ST_A侧压A2右伺服预留
2052.04 BOOL  ; NC433_2_Y 4ST_A侧压A2右伺服预留
2052.05 BOOL  ; NC433_2_Y 4ST_A侧压A2右伺服预留
2052.06 BOOL  ; NC433_2_Y 4ST_A侧压A2右伺服预留
2052.07 BOOL  ; NC433_2_Y 4ST_A侧压A2右伺服预留
2052.08 BOOL  ; NC433_2_Y 4ST_A侧压A2右伺服CW极限输入信号
2052.09 BOOL  ; NC433_2_Y 4ST_A侧压A2右伺服CCW极限输入信号
2052.10 BOOL  ; NC433_2_Y 4ST_A侧压A2右伺服原点接近输入信号
2052.11 BOOL  ; NC433_2_Y 4ST_A侧压A2右伺服原点输入信号
2052.12 BOOL  ; NC433_2_Y 4ST_A侧压A2右伺服中断输入信号
2052.13 BOOL  ; NC433_2_Y 4ST_A侧压A2右伺服紧急输入信号
2052.14 BOOL  ; NC433_2_Y 4ST_A侧压A2右伺服定位完成输入信号
2052.15 BOOL  ; NC433_2_Y 4ST_A侧压A2右伺服偏差计数器复位输出/ 原点调整命令输出
2053.00 BOOL  ; NC433_2_Y 4ST_A侧压A2右伺服错误代码
2053.01 BOOL  ; NC433_2_Y 4ST_A侧压A2右伺服错误代码
2053.02 BOOL  ; NC433_2_Y 4ST_A侧压A2右伺服错误代码
2053.03 BOOL  ; NC433_2_Y 4ST_A侧压A2右伺服错误代码
2053.04 BOOL  ; NC433_2_Y 4ST_A侧压A2右伺服错误代码
2053.05 BOOL  ; NC433_2_Y 4ST_A侧压A2右伺服错误代码
2053.06 BOOL  ; NC433_2_Y 4ST_A侧压A2右伺服错误代码
2053.07 BOOL  ; NC433_2_Y 4ST_A侧压A2右伺服错误代码
2053.08 BOOL  ; NC433_2_Y 4ST_A侧压A2右伺服错误代码
2053.09 BOOL  ; NC433_2_Y 4ST_A侧压A2右伺服错误代码
2053.10 BOOL  ; NC433_2_Y 4ST_A侧压A2右伺服错误代码
2053.11 BOOL  ; NC433_2_Y 4ST_A侧压A2右伺服错误代码
2053.12 BOOL  ; NC433_2_Y 4ST_A侧压A2右伺服错误代码
2053.13 BOOL  ; NC433_2_Y 4ST_A侧压A2右伺服错误代码
2053.14 BOOL  ; NC433_2_Y 4ST_A侧压A2右伺服错误代码
2053.15 BOOL  ; NC433_2_Y 4ST_A侧压A2右伺服错误代码
2054.00 BOOL  ; NC433_2_Z 4ST_A侧压A3左伺服预留
2054.01 BOOL  ; NC433_2_Z 4ST_A侧压A3左伺服预留
2054.02 BOOL  ; NC433_2_Z 4ST_A侧压A3左伺服预留
2054.03 BOOL  ; NC433_2_Z 4ST_A侧压A3左伺服预留
2054.04 BOOL  ; NC433_2_Z 4ST_A侧压A3左伺服等待存储器操作
2054.05 BOOL  ; NC433_2_Z 4ST_A侧压A3左伺服定位完成标志位
2054.06 BOOL  ; NC433_2_Z 4ST_A侧压A3左伺服无原点标志位
2054.07 BOOL  ; NC433_2_Z 4ST_A侧压A3左伺服原点停止标志位
2054.08 BOOL  ; NC433_2_Z 4ST_A侧压A3左伺服0 区监测标志位
2054.09 BOOL  ; NC433_2_Z 4ST_A侧压A3左伺服1 区监测标志位
2054.10 BOOL  ; NC433_2_Z 4ST_A侧压A3左伺服2 区监测标志位
2054.11 BOOL  ; NC433_2_Z 4ST_A侧压A3左伺服示教完成
2054.12 BOOL  ; NC433_2_Z 4ST_A侧压A3左伺服错误标志
2054.13 BOOL  ; NC433_2_Z 4ST_A侧压A3左伺服忙标志
2054.14 BOOL  ; NC433_2_Z 4ST_A侧压A3左伺服数据传送标志位
2054.15 BOOL  ; NC433_2_Z 4ST_A侧压A3左伺服减速停止执行标志位
2055.00 BOOL  ; NC433_2_Z 4ST_A侧压A3左伺服预留
2055.01 BOOL  ; NC433_2_Z 4ST_A侧压A3左伺服预留
2055.02 BOOL  ; NC433_2_Z 4ST_A侧压A3左伺服预留
2055.03 BOOL  ; NC433_2_Z 4ST_A侧压A3左伺服预留
2055.04 BOOL  ; NC433_2_Z 4ST_A侧压A3左伺服预留
2055.05 BOOL  ; NC433_2_Z 4ST_A侧压A3左伺服预留
2055.06 BOOL  ; NC433_2_Z 4ST_A侧压A3左伺服预留
2055.07 BOOL  ; NC433_2_Z 4ST_A侧压A3左伺服预留
2055.08 BOOL  ; NC433_2_Z 4ST_A侧压A3左伺服CW极限输入信号
2055.09 BOOL  ; NC433_2_Z 4ST_A侧压A3左伺服CCW极限输入信号
2055.10 BOOL  ; NC433_2_Z 4ST_A侧压A3左伺服原点接近输入信号
2055.11 BOOL  ; NC433_2_Z 4ST_A侧压A3左伺服原点输入信号
2055.12 BOOL  ; NC433_2_Z 4ST_A侧压A3左伺服中断输入信号
2055.13 BOOL  ; NC433_2_Z 4ST_A侧压A3左伺服紧急输入信号
2055.14 BOOL  ; NC433_2_Z 4ST_A侧压A3左伺服定位完成输入信号
2055.15 BOOL  ; NC433_2_Z 4ST_A侧压A3左伺服偏差计数器复位输出/ 原点调整命令输出
2056.00 BOOL  ; NC433_2_Z 4ST_A侧压A3左伺服错误代码
2056.01 BOOL  ; NC433_2_Z 4ST_A侧压A3左伺服错误代码
2056.02 BOOL  ; NC433_2_Z 4ST_A侧压A3左伺服错误代码
2056.03 BOOL  ; NC433_2_Z 4ST_A侧压A3左伺服错误代码
2056.04 BOOL  ; NC433_2_Z 4ST_A侧压A3左伺服错误代码
2056.05 BOOL  ; NC433_2_Z 4ST_A侧压A3左伺服错误代码
2056.06 BOOL  ; NC433_2_Z 4ST_A侧压A3左伺服错误代码
2056.07 BOOL  ; NC433_2_Z 4ST_A侧压A3左伺服错误代码
2056.08 BOOL  ; NC433_2_Z 4ST_A侧压A3左伺服错误代码
2056.09 BOOL  ; NC433_2_Z 4ST_A侧压A3左伺服错误代码
2056.10 BOOL  ; NC433_2_Z 4ST_A侧压A3左伺服错误代码
2056.11 BOOL  ; NC433_2_Z 4ST_A侧压A3左伺服错误代码
2056.12 BOOL  ; NC433_2_Z 4ST_A侧压A3左伺服错误代码
2056.13 BOOL  ; NC433_2_Z 4ST_A侧压A3左伺服错误代码
2056.14 BOOL  ; NC433_2_Z 4ST_A侧压A3左伺服错误代码
2056.15 BOOL  ; NC433_2_Z 4ST_A侧压A3左伺服错误代码
2057.00 BOOL  ; NC433_2_U 4ST_A侧压A3右伺服预留
2057.01 BOOL  ; NC433_2_U 4ST_A侧压A3右伺服预留
2057.02 BOOL  ; NC433_2_U 4ST_A侧压A3右伺服预留
2057.03 BOOL  ; NC433_2_U 4ST_A侧压A3右伺服预留
2057.04 BOOL  ; NC433_2_U 4ST_A侧压A3右伺服等待存储器操作
2057.05 BOOL  ; NC433_2_U 4ST_A侧压A3右伺服定位完成标志位
2057.06 BOOL  ; NC433_2_U 4ST_A侧压A3右伺服无原点标志位
2057.07 BOOL  ; NC433_2_U 4ST_A侧压A3右伺服原点停止标志位
2057.08 BOOL  ; NC433_2_U 4ST_A侧压A3右伺服0 区监测标志位
2057.09 BOOL  ; NC433_2_U 4ST_A侧压A3右伺服1 区监测标志位
2057.10 BOOL  ; NC433_2_U 4ST_A侧压A3右伺服2 区监测标志位
2057.11 BOOL  ; NC433_2_U 4ST_A侧压A3右伺服示教完成
2057.12 BOOL  ; NC433_2_U 4ST_A侧压A3右伺服错误标志
2057.13 BOOL  ; NC433_2_U 4ST_A侧压A3右伺服忙标志
2057.14 BOOL  ; NC433_2_U 4ST_A侧压A3右伺服数据传送标志位
2057.15 BOOL  ; NC433_2_U 4ST_A侧压A3右伺服减速停止执行标志位
2058.00 BOOL  ; NC433_2_U 4ST_A侧压A3右伺服预留
2058.01 BOOL  ; NC433_2_U 4ST_A侧压A3右伺服预留
2058.02 BOOL  ; NC433_2_U 4ST_A侧压A3右伺服预留
2058.03 BOOL  ; NC433_2_U 4ST_A侧压A3右伺服预留
2058.04 BOOL  ; NC433_2_U 4ST_A侧压A3右伺服预留
2058.05 BOOL  ; NC433_2_U 4ST_A侧压A3右伺服预留
2058.06 BOOL  ; NC433_2_U 4ST_A侧压A3右伺服预留
2058.07 BOOL  ; NC433_2_U 4ST_A侧压A3右伺服预留
2058.08 BOOL  ; NC433_2_U 4ST_A侧压A3右伺服CW极限输入信号
2058.09 BOOL  ; NC433_2_U 4ST_A侧压A3右伺服CCW极限输入信号
2058.10 BOOL  ; NC433_2_U 4ST_A侧压A3右伺服原点接近输入信号
2058.11 BOOL  ; NC433_2_U 4ST_A侧压A3右伺服原点输入信号
2058.12 BOOL  ; NC433_2_U 4ST_A侧压A3右伺服中断输入信号
2058.13 BOOL  ; NC433_2_U 4ST_A侧压A3右伺服紧急输入信号
2058.14 BOOL  ; NC433_2_U 4ST_A侧压A3右伺服定位完成输入信号
2058.15 BOOL  ; NC433_2_U 4ST_A侧压A3右伺服偏差计数器复位输出/ 原点调整命令输出
2059.00 BOOL  ; NC433_2_U 4ST_A侧压A3右伺服错误代码
2059.01 BOOL  ; NC433_2_U 4ST_A侧压A3右伺服错误代码
2059.02 BOOL  ; NC433_2_U 4ST_A侧压A3右伺服错误代码
2059.03 BOOL  ; NC433_2_U 4ST_A侧压A3右伺服错误代码
2059.04 BOOL  ; NC433_2_U 4ST_A侧压A3右伺服错误代码
2059.05 BOOL  ; NC433_2_U 4ST_A侧压A3右伺服错误代码
2059.06 BOOL  ; NC433_2_U 4ST_A侧压A3右伺服错误代码
2059.07 BOOL  ; NC433_2_U 4ST_A侧压A3右伺服错误代码
2059.08 BOOL  ; NC433_2_U 4ST_A侧压A3右伺服错误代码
2059.09 BOOL  ; NC433_2_U 4ST_A侧压A3右伺服错误代码
2059.10 BOOL  ; NC433_2_U 4ST_A侧压A3右伺服错误代码
2059.11 BOOL  ; NC433_2_U 4ST_A侧压A3右伺服错误代码
2059.12 BOOL  ; NC433_2_U 4ST_A侧压A3右伺服错误代码
2059.13 BOOL  ; NC433_2_U 4ST_A侧压A3右伺服错误代码
2059.14 BOOL  ; NC433_2_U 4ST_A侧压A3右伺服错误代码
2059.15 BOOL  ; NC433_2_U 4ST_A侧压A3右伺服错误代码
2060.00 BOOL  ; NC433_3_X 4ST_A侧压A4左伺服存储器操作命令激活序列数
2060.01 BOOL  ; NC433_3_X 4ST_A侧压A4左伺服存储器操作命令起动
2060.02 BOOL  ; NC433_3_X 4ST_A侧压A4左伺服存储器操作命令独立起动
2060.03 BOOL  ; NC433_3_X 4ST_A侧压A4左伺服直接操作命令绝对移动
2060.04 BOOL  ; NC433_3_X 4ST_A侧压A4左伺服直接操作命令相对移动
2060.05 BOOL  ; NC433_3_X 4ST_A侧压A4左伺服直接操作命令中断进给
2060.06 BOOL  ; NC433_3_X 4ST_A侧压A4左伺服原点定位命令原点搜索
2060.07 BOOL  ; NC433_3_X 4ST_A侧压A4左伺服原点定位命令原点返回
2060.08 BOOL  ; NC433_3_X 4ST_A侧压A4左伺服原点定位命令当前位置预置
2060.09 BOOL  ; NC433_3_X 4ST_A侧压A4左伺服点动
2060.10 BOOL  ; NC433_3_X 4ST_A侧压A4左伺服点动方向(0=CW,1=CCW)
2060.11 BOOL  ; NC433_3_X 4ST_A侧压A4左伺服示教
2060.12 BOOL  ; NC433_3_X 4ST_A侧压A4左伺服错误清除
2060.13 BOOL  ; NC433_3_X 4ST_A侧压A4左伺服偏差计数器复位输出/ 原点调整命令输出
2060.14 BOOL  ; NC433_3_X 4ST_A侧压A4左伺服激活Override
2060.15 BOOL  ; NC433_3_X 4ST_A侧压A4左伺服停止
2061.00 BOOL  ; NC433_3_X 4ST_A侧压A4左伺服预留
2061.01 BOOL  ; NC433_3_X 4ST_A侧压A4左伺服预留
2061.02 BOOL  ; NC433_3_X 4ST_A侧压A4左伺服预留
2061.03 BOOL  ; NC433_3_X 4ST_A侧压A4左伺服预留
2061.04 BOOL  ; NC433_3_X 4ST_A侧压A4左伺服预留
2061.05 BOOL  ; NC433_3_X 4ST_A侧压A4左伺服预留
2061.06 BOOL  ; NC433_3_X 4ST_A侧压A4左伺服预留
2061.07 BOOL  ; NC433_3_X 4ST_A侧压A4左伺服预留
2061.08 BOOL  ; NC433_3_X 4ST_A侧压A4左伺服强制中断
2061.09 BOOL  ; NC433_3_X 4ST_A侧压A4左伺服预留
2061.10 BOOL  ; NC433_3_X 4ST_A侧压A4左伺服预留
2061.11 BOOL  ; NC433_3_X 4ST_A侧压A4左伺服预留
2061.12 BOOL  ; NC433_3_X 4ST_A侧压A4左伺服数据写入
2061.13 BOOL  ; NC433_3_X 4ST_A侧压A4左伺服数据读出
2061.14 BOOL  ; NC433_3_X 4ST_A侧压A4左伺服数据保存
2061.15 BOOL  ; NC433_3_X 4ST_A侧压A4左伺服预留
2062.00 BOOL  ; NC433_3_Y 4ST_A侧压A4右伺服存储器操作命令激活序列数
2062.01 BOOL  ; NC433_3_Y 4ST_A侧压A4右伺服存储器操作命令起动
2062.02 BOOL  ; NC433_3_Y 4ST_A侧压A4右伺服存储器操作命令独立起动
2062.03 BOOL  ; NC433_3_Y 4ST_A侧压A4右伺服直接操作命令绝对移动
2062.04 BOOL  ; NC433_3_Y 4ST_A侧压A4右伺服直接操作命令相对移动
2062.05 BOOL  ; NC433_3_Y 4ST_A侧压A4右伺服直接操作命令中断进给
2062.06 BOOL  ; NC433_3_Y 4ST_A侧压A4右伺服原点定位命令原点搜索
2062.07 BOOL  ; NC433_3_Y 4ST_A侧压A4右伺服原点定位命令原点返回
2062.08 BOOL  ; NC433_3_Y 4ST_A侧压A4右伺服原点定位命令当前位置预置
2062.09 BOOL  ; NC433_3_Y 4ST_A侧压A4右伺服点动
2062.10 BOOL  ; NC433_3_Y 4ST_A侧压A4右伺服点动方向(0=CW,1=CCW)
2062.11 BOOL  ; NC433_3_Y 4ST_A侧压A4右伺服示教
2062.12 BOOL  ; NC433_3_Y 4ST_A侧压A4右伺服错误清除
2062.13 BOOL  ; NC433_3_Y 4ST_A侧压A4右伺服偏差计数器复位输出/ 原点调整命令输出
2062.14 BOOL  ; NC433_3_Y 4ST_A侧压A4右伺服激活Override
2062.15 BOOL  ; NC433_3_Y 4ST_A侧压A4右伺服停止
2063.00 BOOL  ; NC433_3_Y 4ST_A侧压A4右伺服预留
2063.01 BOOL  ; NC433_3_Y 4ST_A侧压A4右伺服预留
2063.02 BOOL  ; NC433_3_Y 4ST_A侧压A4右伺服预留
2063.03 BOOL  ; NC433_3_Y 4ST_A侧压A4右伺服预留
2063.04 BOOL  ; NC433_3_Y 4ST_A侧压A4右伺服预留
2063.05 BOOL  ; NC433_3_Y 4ST_A侧压A4右伺服预留
2063.06 BOOL  ; NC433_3_Y 4ST_A侧压A4右伺服预留
2063.07 BOOL  ; NC433_3_Y 4ST_A侧压A4右伺服预留
2063.08 BOOL  ; NC433_3_Y 4ST_A侧压A4右伺服强制中断
2063.09 BOOL  ; NC433_3_Y 4ST_A侧压A4右伺服预留
2063.10 BOOL  ; NC433_3_Y 4ST_A侧压A4右伺服预留
2063.11 BOOL  ; NC433_3_Y 4ST_A侧压A4右伺服预留
2063.12 BOOL  ; NC433_3_Y 4ST_A侧压A4右伺服数据写入
2063.13 BOOL  ; NC433_3_Y 4ST_A侧压A4右伺服数据读出
2063.14 BOOL  ; NC433_3_Y 4ST_A侧压A4右伺服数据保存
2063.15 BOOL  ; NC433_3_Y 4ST_A侧压A4右伺服预留
2064.00 BOOL  ; NC433_3_Z 4ST_B 正压伺服B存储器操作命令激活序列数
2064.01 BOOL  ; NC433_3_Z 4ST_B 正压伺服B存储器操作命令起动
2064.02 BOOL  ; NC433_3_Z 4ST_B 正压伺服B存储器操作命令独立起动
2064.03 BOOL  ; NC433_3_Z 4ST_B 正压伺服B直接操作命令绝对移动
2064.04 BOOL  ; NC433_3_Z 4ST_B 正压伺服B直接操作命令相对移动
2064.05 BOOL  ; NC433_3_Z 4ST_B 正压伺服B直接操作命令中断进给
2064.06 BOOL  ; NC433_3_Z 4ST_B 正压伺服B原点定位命令原点搜索
2064.07 BOOL  ; NC433_3_Z 4ST_B 正压伺服B原点定位命令原点返回
2064.08 BOOL  ; NC433_3_Z 4ST_B 正压伺服B原点定位命令当前位置预置
2064.09 BOOL  ; NC433_3_Z 4ST_B 正压伺服B点动
2064.10 BOOL  ; NC433_3_Z 4ST_B 正压伺服B点动方向(0=CW,1=CCW)
2064.11 BOOL  ; NC433_3_Z 4ST_B 正压伺服B示教
2064.12 BOOL  ; NC433_3_Z 4ST_B 正压伺服B错误清除
2064.13 BOOL  ; NC433_3_Z 4ST_B 正压伺服B偏差计数器复位输出/ 原点调整命令输出
2064.14 BOOL  ; NC433_3_Z 4ST_B 正压伺服B激活Override
2064.15 BOOL  ; NC433_3_Z 4ST_B 正压伺服B停止
2065.00 BOOL  ; NC433_3_Z 4ST_B 正压伺服B预留
2065.01 BOOL  ; NC433_3_Z 4ST_B 正压伺服B预留
2065.02 BOOL  ; NC433_3_Z 4ST_B 正压伺服B预留
2065.03 BOOL  ; NC433_3_Z 4ST_B 正压伺服B预留
2065.04 BOOL  ; NC433_3_Z 4ST_B 正压伺服B预留
2065.05 BOOL  ; NC433_3_Z 4ST_B 正压伺服B预留
2065.06 BOOL  ; NC433_3_Z 4ST_B 正压伺服B预留
2065.07 BOOL  ; NC433_3_Z 4ST_B 正压伺服B预留
2065.08 BOOL  ; NC433_3_Z 4ST_B 正压伺服B强制中断
2065.09 BOOL  ; NC433_3_Z 4ST_B 正压伺服B预留
2065.10 BOOL  ; NC433_3_Z 4ST_B 正压伺服B预留
2065.11 BOOL  ; NC433_3_Z 4ST_B 正压伺服B预留
2065.12 BOOL  ; NC433_3_Z 4ST_B 正压伺服B数据写入
2065.13 BOOL  ; NC433_3_Z 4ST_B 正压伺服B数据读出
2065.14 BOOL  ; NC433_3_Z 4ST_B 正压伺服B数据保存
2065.15 BOOL  ; NC433_3_Z 4ST_B 正压伺服B预留
2066.00 BOOL  ; NC433_3_U 4ST_B 压板平移伺服B存储器操作命令激活序列数
2066.01 BOOL  ; NC433_3_U 4ST_B 压板平移伺服B存储器操作命令起动
2066.02 BOOL  ; NC433_3_U 4ST_B 压板平移伺服B存储器操作命令独立起动
2066.03 BOOL  ; NC433_3_U 4ST_B 压板平移伺服B直接操作命令绝对移动
2066.04 BOOL  ; NC433_3_U 4ST_B 压板平移伺服B直接操作命令相对移动
2066.05 BOOL  ; NC433_3_U 4ST_B 压板平移伺服B直接操作命令中断进给
2066.06 BOOL  ; NC433_3_U 4ST_B 压板平移伺服B原点定位命令原点搜索
2066.07 BOOL  ; NC433_3_U 4ST_B 压板平移伺服B原点定位命令原点返回
2066.08 BOOL  ; NC433_3_U 4ST_B 压板平移伺服B原点定位命令当前位置预置
2066.09 BOOL  ; NC433_3_U 4ST_B 压板平移伺服B点动
2066.10 BOOL  ; NC433_3_U 4ST_B 压板平移伺服B点动方向(0=CW,1=CCW)
2066.11 BOOL  ; NC433_3_U 4ST_B 压板平移伺服B示教
2066.12 BOOL  ; NC433_3_U 4ST_B 压板平移伺服B错误清除
2066.13 BOOL  ; NC433_3_U 4ST_B 压板平移伺服B偏差计数器复位输出/ 原点调整命令输出
2066.14 BOOL  ; NC433_3_U 4ST_B 压板平移伺服B激活Override
2066.15 BOOL  ; NC433_3_U 4ST_B 压板平移伺服B停止
2067.00 BOOL  ; NC433_3_U 4ST_B 压板平移伺服B预留
2067.01 BOOL  ; NC433_3_U 4ST_B 压板平移伺服B预留
2067.02 BOOL  ; NC433_3_U 4ST_B 压板平移伺服B预留
2067.03 BOOL  ; NC433_3_U 4ST_B 压板平移伺服B预留
2067.04 BOOL  ; NC433_3_U 4ST_B 压板平移伺服B预留
2067.05 BOOL  ; NC433_3_U 4ST_B 压板平移伺服B预留
2067.06 BOOL  ; NC433_3_U 4ST_B 压板平移伺服B预留
2067.07 BOOL  ; NC433_3_U 4ST_B 压板平移伺服B预留
2067.08 BOOL  ; NC433_3_U 4ST_B 压板平移伺服B强制中断
2067.09 BOOL  ; NC433_3_U 4ST_B 压板平移伺服B预留
2067.10 BOOL  ; NC433_3_U 4ST_B 压板平移伺服B预留
2067.11 BOOL  ; NC433_3_U 4ST_B 压板平移伺服B预留
2067.12 BOOL  ; NC433_3_U 4ST_B 压板平移伺服B数据写入
2067.13 BOOL  ; NC433_3_U 4ST_B 压板平移伺服B数据读出
2067.14 BOOL  ; NC433_3_U 4ST_B 压板平移伺服B数据保存
2067.15 BOOL  ; NC433_3_U 4ST_B 压板平移伺服B预留
2068.00 BOOL  ; NC433_3_X 4ST_A侧压A4左伺服预留
2068.01 BOOL  ; NC433_3_X 4ST_A侧压A4左伺服预留
2068.02 BOOL  ; NC433_3_X 4ST_A侧压A4左伺服预留
2068.03 BOOL  ; NC433_3_X 4ST_A侧压A4左伺服预留
2068.04 BOOL  ; NC433_3_X 4ST_A侧压A4左伺服等待存储器操作
2068.05 BOOL  ; NC433_3_X 4ST_A侧压A4左伺服定位完成标志位
2068.06 BOOL  ; NC433_3_X 4ST_A侧压A4左伺服无原点标志位
2068.07 BOOL  ; NC433_3_X 4ST_A侧压A4左伺服原点停止标志位
2068.08 BOOL  ; NC433_3_X 4ST_A侧压A4左伺服0 区监测标志位
2068.09 BOOL  ; NC433_3_X 4ST_A侧压A4左伺服1 区监测标志位
2068.10 BOOL  ; NC433_3_X 4ST_A侧压A4左伺服2 区监测标志位
2068.11 BOOL  ; NC433_3_X 4ST_A侧压A4左伺服示教完成
2068.12 BOOL  ; NC433_3_X 4ST_A侧压A4左伺服错误标志
2068.13 BOOL  ; NC433_3_X 4ST_A侧压A4左伺服忙标志
2068.14 BOOL  ; NC433_3_X 4ST_A侧压A4左伺服数据传送标志位
2068.15 BOOL  ; NC433_3_X 4ST_A侧压A4左伺服减速停止执行标志位
2069.00 BOOL  ; NC433_3_X 4ST_A侧压A4左伺服预留
2069.01 BOOL  ; NC433_3_X 4ST_A侧压A4左伺服预留
2069.02 BOOL  ; NC433_3_X 4ST_A侧压A4左伺服预留
2069.03 BOOL  ; NC433_3_X 4ST_A侧压A4左伺服预留
2069.04 BOOL  ; NC433_3_X 4ST_A侧压A4左伺服预留
2069.05 BOOL  ; NC433_3_X 4ST_A侧压A4左伺服预留
2069.06 BOOL  ; NC433_3_X 4ST_A侧压A4左伺服预留
2069.07 BOOL  ; NC433_3_X 4ST_A侧压A4左伺服预留
2069.08 BOOL  ; NC433_3_X 4ST_A侧压A4左伺服CW极限输入信号
2069.09 BOOL  ; NC433_3_X 4ST_A侧压A4左伺服CCW极限输入信号
2069.10 BOOL  ; NC433_3_X 4ST_A侧压A4左伺服原点接近输入信号
2069.11 BOOL  ; NC433_3_X 4ST_A侧压A4左伺服原点输入信号
2069.12 BOOL  ; NC433_3_X 4ST_A侧压A4左伺服中断输入信号
2069.13 BOOL  ; NC433_3_X 4ST_A侧压A4左伺服紧急输入信号
2069.14 BOOL  ; NC433_3_X 4ST_A侧压A4左伺服定位完成输入信号
2069.15 BOOL  ; NC433_3_X 4ST_A侧压A4左伺服偏差计数器复位输出/ 原点调整命令输出
2070 CHANNEL  ; DA08V_1 通道使能
2070.00 BOOL  ; NC433_3_X 4ST_A侧压A4左伺服错误代码
2070.01 BOOL  ; NC433_3_X 4ST_A侧压A4左伺服错误代码
2070.02 BOOL  ; NC433_3_X 4ST_A侧压A4左伺服错误代码
2070.03 BOOL  ; NC433_3_X 4ST_A侧压A4左伺服错误代码
2070.04 BOOL  ; NC433_3_X 4ST_A侧压A4左伺服错误代码
2070.05 BOOL  ; NC433_3_X 4ST_A侧压A4左伺服错误代码
2070.06 BOOL  ; NC433_3_X 4ST_A侧压A4左伺服错误代码
2070.07 BOOL  ; NC433_3_X 4ST_A侧压A4左伺服错误代码
2070.08 BOOL  ; NC433_3_X 4ST_A侧压A4左伺服错误代码
2070.09 BOOL  ; NC433_3_X 4ST_A侧压A4左伺服错误代码
2070.10 BOOL  ; NC433_3_X 4ST_A侧压A4左伺服错误代码
2070.11 BOOL  ; NC433_3_X 4ST_A侧压A4左伺服错误代码
2070.12 BOOL  ; NC433_3_X 4ST_A侧压A4左伺服错误代码
2070.13 BOOL  ; NC433_3_X 4ST_A侧压A4左伺服错误代码
2070.14 BOOL  ; NC433_3_X 4ST_A侧压A4左伺服错误代码
2070.15 BOOL  ; NC433_3_X 4ST_A侧压A4左伺服错误代码
2071 CHANNEL  ; DA08V_1 通道1 A1比例阀 转换值
2071.00 BOOL  ; NC433_3_Y 4ST_A侧压A4右伺服预留
2071.01 BOOL  ; NC433_3_Y 4ST_A侧压A4右伺服预留
2071.02 BOOL  ; NC433_3_Y 4ST_A侧压A4右伺服预留
2071.03 BOOL  ; NC433_3_Y 4ST_A侧压A4右伺服预留
2071.04 BOOL  ; NC433_3_Y 4ST_A侧压A4右伺服等待存储器操作
2071.05 BOOL  ; NC433_3_Y 4ST_A侧压A4右伺服定位完成标志位
2071.06 BOOL  ; NC433_3_Y 4ST_A侧压A4右伺服无原点标志位
2071.07 BOOL  ; NC433_3_Y 4ST_A侧压A4右伺服原点停止标志位
2071.08 BOOL  ; NC433_3_Y 4ST_A侧压A4右伺服0 区监测标志位
2071.09 BOOL  ; NC433_3_Y 4ST_A侧压A4右伺服1 区监测标志位
2071.10 BOOL  ; NC433_3_Y 4ST_A侧压A4右伺服2 区监测标志位
2071.11 BOOL  ; NC433_3_Y 4ST_A侧压A4右伺服示教完成
2071.12 BOOL  ; NC433_3_Y 4ST_A侧压A4右伺服错误标志
2071.13 BOOL  ; NC433_3_Y 4ST_A侧压A4右伺服忙标志
2071.14 BOOL  ; NC433_3_Y 4ST_A侧压A4右伺服数据传送标志位
2071.15 BOOL  ; NC433_3_Y 4ST_A侧压A4右伺服减速停止执行标志位
2072 CHANNEL  ; DA08V_1 通道2 A2比例阀 转换值
2072.00 BOOL  ; NC433_3_Y 4ST_A侧压A4右伺服预留
2072.01 BOOL  ; NC433_3_Y 4ST_A侧压A4右伺服预留
2072.02 BOOL  ; NC433_3_Y 4ST_A侧压A4右伺服预留
2072.03 BOOL  ; NC433_3_Y 4ST_A侧压A4右伺服预留
2072.04 BOOL  ; NC433_3_Y 4ST_A侧压A4右伺服预留
2072.05 BOOL  ; NC433_3_Y 4ST_A侧压A4右伺服预留
2072.06 BOOL  ; NC433_3_Y 4ST_A侧压A4右伺服预留
2072.07 BOOL  ; NC433_3_Y 4ST_A侧压A4右伺服预留
2072.08 BOOL  ; NC433_3_Y 4ST_A侧压A4右伺服CW极限输入信号
2072.09 BOOL  ; NC433_3_Y 4ST_A侧压A4右伺服CCW极限输入信号
2072.10 BOOL  ; NC433_3_Y 4ST_A侧压A4右伺服原点接近输入信号
2072.11 BOOL  ; NC433_3_Y 4ST_A侧压A4右伺服原点输入信号
2072.12 BOOL  ; NC433_3_Y 4ST_A侧压A4右伺服中断输入信号
2072.13 BOOL  ; NC433_3_Y 4ST_A侧压A4右伺服紧急输入信号
2072.14 BOOL  ; NC433_3_Y 4ST_A侧压A4右伺服定位完成输入信号
2072.15 BOOL  ; NC433_3_Y 4ST_A侧压A4右伺服偏差计数器复位输出/ 原点调整命令输出
2073 CHANNEL  ; DA08V_1 通道3 A3比例阀 转换值
2073.00 BOOL  ; NC433_3_Y 4ST_A侧压A4右伺服错误代码
2073.01 BOOL  ; NC433_3_Y 4ST_A侧压A4右伺服错误代码
2073.02 BOOL  ; NC433_3_Y 4ST_A侧压A4右伺服错误代码
2073.03 BOOL  ; NC433_3_Y 4ST_A侧压A4右伺服错误代码
2073.04 BOOL  ; NC433_3_Y 4ST_A侧压A4右伺服错误代码
2073.05 BOOL  ; NC433_3_Y 4ST_A侧压A4右伺服错误代码
2073.06 BOOL  ; NC433_3_Y 4ST_A侧压A4右伺服错误代码
2073.07 BOOL  ; NC433_3_Y 4ST_A侧压A4右伺服错误代码
2073.08 BOOL  ; NC433_3_Y 4ST_A侧压A4右伺服错误代码
2073.09 BOOL  ; NC433_3_Y 4ST_A侧压A4右伺服错误代码
2073.10 BOOL  ; NC433_3_Y 4ST_A侧压A4右伺服错误代码
2073.11 BOOL  ; NC433_3_Y 4ST_A侧压A4右伺服错误代码
2073.12 BOOL  ; NC433_3_Y 4ST_A侧压A4右伺服错误代码
2073.13 BOOL  ; NC433_3_Y 4ST_A侧压A4右伺服错误代码
2073.14 BOOL  ; NC433_3_Y 4ST_A侧压A4右伺服错误代码
2073.15 BOOL  ; NC433_3_Y 4ST_A侧压A4右伺服错误代码
2074 CHANNEL  ; DA08V_1 通道4 A4比例阀 转换值
2074.00 BOOL  ; NC433_3_Z 4ST_B 正压伺服B预留
2074.01 BOOL  ; NC433_3_Z 4ST_B 正压伺服B预留
2074.02 BOOL  ; NC433_3_Z 4ST_B 正压伺服B预留
2074.03 BOOL  ; NC433_3_Z 4ST_B 正压伺服B预留
2074.04 BOOL  ; NC433_3_Z 4ST_B 正压伺服B等待存储器操作
2074.05 BOOL  ; NC433_3_Z 4ST_B 正压伺服B定位完成标志位
2074.06 BOOL  ; NC433_3_Z 4ST_B 正压伺服B无原点标志位
2074.07 BOOL  ; NC433_3_Z 4ST_B 正压伺服B原点停止标志位
2074.08 BOOL  ; NC433_3_Z 4ST_B 正压伺服B0 区监测标志位
2074.09 BOOL  ; NC433_3_Z 4ST_B 正压伺服B1 区监测标志位
2074.10 BOOL  ; NC433_3_Z 4ST_B 正压伺服B2 区监测标志位
2074.11 BOOL  ; NC433_3_Z 4ST_B 正压伺服B示教完成
2074.12 BOOL  ; NC433_3_Z 4ST_B 正压伺服B错误标志
2074.13 BOOL  ; NC433_3_Z 4ST_B 正压伺服B忙标志
2074.14 BOOL  ; NC433_3_Z 4ST_B 正压伺服B数据传送标志位
2074.15 BOOL  ; NC433_3_Z 4ST_B 正压伺服B减速停止执行标志位
2075 CHANNEL  ; DA08V_1 通道5 B1比例阀 转换值
2075.00 BOOL  ; NC433_3_Z 4ST_B 正压伺服B预留
2075.01 BOOL  ; NC433_3_Z 4ST_B 正压伺服B预留
2075.02 BOOL  ; NC433_3_Z 4ST_B 正压伺服B预留
2075.03 BOOL  ; NC433_3_Z 4ST_B 正压伺服B预留
2075.04 BOOL  ; NC433_3_Z 4ST_B 正压伺服B预留
2075.05 BOOL  ; NC433_3_Z 4ST_B 正压伺服B预留
2075.06 BOOL  ; NC433_3_Z 4ST_B 正压伺服B预留
2075.07 BOOL  ; NC433_3_Z 4ST_B 正压伺服B预留
2075.08 BOOL  ; NC433_3_Z 4ST_B 正压伺服BCW极限输入信号
2075.09 BOOL  ; NC433_3_Z 4ST_B 正压伺服BCCW极限输入信号
2075.10 BOOL  ; NC433_3_Z 4ST_B 正压伺服B原点接近输入信号
2075.11 BOOL  ; NC433_3_Z 4ST_B 正压伺服B原点输入信号
2075.12 BOOL  ; NC433_3_Z 4ST_B 正压伺服B中断输入信号
2075.13 BOOL  ; NC433_3_Z 4ST_B 正压伺服B紧急输入信号
2075.14 BOOL  ; NC433_3_Z 4ST_B 正压伺服B定位完成输入信号
2075.15 BOOL  ; NC433_3_Z 4ST_B 正压伺服B偏差计数器复位输出/ 原点调整命令输出
2076 CHANNEL  ; DA08V_1 通道6 B2比例阀 转换值
2076.00 BOOL  ; NC433_3_Z 4ST_B 正压伺服B错误代码
2076.01 BOOL  ; NC433_3_Z 4ST_B 正压伺服B错误代码
2076.02 BOOL  ; NC433_3_Z 4ST_B 正压伺服B错误代码
2076.03 BOOL  ; NC433_3_Z 4ST_B 正压伺服B错误代码
2076.04 BOOL  ; NC433_3_Z 4ST_B 正压伺服B错误代码
2076.05 BOOL  ; NC433_3_Z 4ST_B 正压伺服B错误代码
2076.06 BOOL  ; NC433_3_Z 4ST_B 正压伺服B错误代码
2076.07 BOOL  ; NC433_3_Z 4ST_B 正压伺服B错误代码
2076.08 BOOL  ; NC433_3_Z 4ST_B 正压伺服B错误代码
2076.09 BOOL  ; NC433_3_Z 4ST_B 正压伺服B错误代码
2076.10 BOOL  ; NC433_3_Z 4ST_B 正压伺服B错误代码
2076.11 BOOL  ; NC433_3_Z 4ST_B 正压伺服B错误代码
2076.12 BOOL  ; NC433_3_Z 4ST_B 正压伺服B错误代码
2076.13 BOOL  ; NC433_3_Z 4ST_B 正压伺服B错误代码
2076.14 BOOL  ; NC433_3_Z 4ST_B 正压伺服B错误代码
2076.15 BOOL  ; NC433_3_Z 4ST_B 正压伺服B错误代码
2077 CHANNEL  ; DA08V_1 通道7 B3比例阀 转换值
2077.00 BOOL  ; NC433_3_U 4ST_B 压板平移伺服B预留
2077.01 BOOL  ; NC433_3_U 4ST_B 压板平移伺服B预留
2077.02 BOOL  ; NC433_3_U 4ST_B 压板平移伺服B预留
2077.03 BOOL  ; NC433_3_U 4ST_B 压板平移伺服B预留
2077.04 BOOL  ; NC433_3_U 4ST_B 压板平移伺服B等待存储器操作
2077.05 BOOL  ; NC433_3_U 4ST_B 压板平移伺服B定位完成标志位
2077.06 BOOL  ; NC433_3_U 4ST_B 压板平移伺服B无原点标志位
2077.07 BOOL  ; NC433_3_U 4ST_B 压板平移伺服B原点停止标志位
2077.08 BOOL  ; NC433_3_U 4ST_B 压板平移伺服B0 区监测标志位
2077.09 BOOL  ; NC433_3_U 4ST_B 压板平移伺服B1 区监测标志位
2077.10 BOOL  ; NC433_3_U 4ST_B 压板平移伺服B2 区监测标志位
2077.11 BOOL  ; NC433_3_U 4ST_B 压板平移伺服B示教完成
2077.12 BOOL  ; NC433_3_U 4ST_B 压板平移伺服B错误标志
2077.13 BOOL  ; NC433_3_U 4ST_B 压板平移伺服B忙标志
2077.14 BOOL  ; NC433_3_U 4ST_B 压板平移伺服B数据传送标志位
2077.15 BOOL  ; NC433_3_U 4ST_B 压板平移伺服B减速停止执行标志位
2078 CHANNEL  ; DA08V_1 通道8 B4比例阀 转换值
2078.00 BOOL  ; NC433_3_U 4ST_B 压板平移伺服B预留
2078.01 BOOL  ; NC433_3_U 4ST_B 压板平移伺服B预留
2078.02 BOOL  ; NC433_3_U 4ST_B 压板平移伺服B预留
2078.03 BOOL  ; NC433_3_U 4ST_B 压板平移伺服B预留
2078.04 BOOL  ; NC433_3_U 4ST_B 压板平移伺服B预留
2078.05 BOOL  ; NC433_3_U 4ST_B 压板平移伺服B预留
2078.06 BOOL  ; NC433_3_U 4ST_B 压板平移伺服B预留
2078.07 BOOL  ; NC433_3_U 4ST_B 压板平移伺服B预留
2078.08 BOOL  ; NC433_3_U 4ST_B 压板平移伺服BCW极限输入信号
2078.09 BOOL  ; NC433_3_U 4ST_B 压板平移伺服BCCW极限输入信号
2078.10 BOOL  ; NC433_3_U 4ST_B 压板平移伺服B原点接近输入信号
2078.11 BOOL  ; NC433_3_U 4ST_B 压板平移伺服B原点输入信号
2078.12 BOOL  ; NC433_3_U 4ST_B 压板平移伺服B中断输入信号
2078.13 BOOL  ; NC433_3_U 4ST_B 压板平移伺服B紧急输入信号
2078.14 BOOL  ; NC433_3_U 4ST_B 压板平移伺服B定位完成输入信号
2078.15 BOOL  ; NC433_3_U 4ST_B 压板平移伺服B偏差计数器复位输出/ 原点调整命令输出
2079.00 BOOL  ; NC433_3_U 4ST_B 压板平移伺服B错误代码
2079.01 BOOL  ; NC433_3_U 4ST_B 压板平移伺服B错误代码
2079.02 BOOL  ; NC433_3_U 4ST_B 压板平移伺服B错误代码
2079.03 BOOL  ; NC433_3_U 4ST_B 压板平移伺服B错误代码
2079.04 BOOL  ; NC433_3_U 4ST_B 压板平移伺服B错误代码
2079.05 BOOL  ; NC433_3_U 4ST_B 压板平移伺服B错误代码
2079.06 BOOL  ; NC433_3_U 4ST_B 压板平移伺服B错误代码
2079.07 BOOL  ; NC433_3_U 4ST_B 压板平移伺服B错误代码
2079.08 BOOL  ; NC433_3_U 4ST_B 压板平移伺服B错误代码
2079.09 BOOL  ; NC433_3_U 4ST_B 压板平移伺服B错误代码
2079.10 BOOL  ; NC433_3_U 4ST_B 压板平移伺服B错误代码
2079.11 BOOL  ; NC433_3_U 4ST_B 压板平移伺服B错误代码
2079.12 BOOL  ; NC433_3_U 4ST_B 压板平移伺服B错误代码
2079.13 BOOL  ; NC433_3_U 4ST_B 压板平移伺服B错误代码
2079.14 BOOL  ; NC433_3_U 4ST_B 压板平移伺服B错误代码
2079.15 BOOL  ; NC433_3_U 4ST_B 压板平移伺服B错误代码
2080 CHANNEL  ; DA08V_2 通道使能
2080.00 BOOL  ; NC433_4_X 4ST_B 侧压B1左伺服存储器操作命令激活序列数
2080.01 BOOL  ; NC433_4_X 4ST_B 侧压B1左伺服存储器操作命令起动
2080.02 BOOL  ; NC433_4_X 4ST_B 侧压B1左伺服存储器操作命令独立起动
2080.03 BOOL  ; NC433_4_X 4ST_B 侧压B1左伺服直接操作命令绝对移动
2080.04 BOOL  ; NC433_4_X 4ST_B 侧压B1左伺服直接操作命令相对移动
2080.05 BOOL  ; NC433_4_X 4ST_B 侧压B1左伺服直接操作命令中断进给
2080.06 BOOL  ; NC433_4_X 4ST_B 侧压B1左伺服原点定位命令原点搜索
2080.07 BOOL  ; NC433_4_X 4ST_B 侧压B1左伺服原点定位命令原点返回
2080.08 BOOL  ; NC433_4_X 4ST_B 侧压B1左伺服原点定位命令当前位置预置
2080.09 BOOL  ; NC433_4_X 4ST_B 侧压B1左伺服点动
2080.10 BOOL  ; NC433_4_X 4ST_B 侧压B1左伺服点动方向(0=CW,1=CCW)
2080.11 BOOL  ; NC433_4_X 4ST_B 侧压B1左伺服示教
2080.12 BOOL  ; NC433_4_X 4ST_B 侧压B1左伺服错误清除
2080.13 BOOL  ; NC433_4_X 4ST_B 侧压B1左伺服偏差计数器复位输出/ 原点调整命令输出
2080.14 BOOL  ; NC433_4_X 4ST_B 侧压B1左伺服激活Override
2080.15 BOOL  ; NC433_4_X 4ST_B 侧压B1左伺服停止
2081 CHANNEL  ; DA08V_2 通道1DA 转换值
2081.00 BOOL  ; NC433_4_X 4ST_B 侧压B1左伺服预留
2081.01 BOOL  ; NC433_4_X 4ST_B 侧压B1左伺服预留
2081.02 BOOL  ; NC433_4_X 4ST_B 侧压B1左伺服预留
2081.03 BOOL  ; NC433_4_X 4ST_B 侧压B1左伺服预留
2081.04 BOOL  ; NC433_4_X 4ST_B 侧压B1左伺服预留
2081.05 BOOL  ; NC433_4_X 4ST_B 侧压B1左伺服预留
2081.06 BOOL  ; NC433_4_X 4ST_B 侧压B1左伺服预留
2081.07 BOOL  ; NC433_4_X 4ST_B 侧压B1左伺服预留
2081.08 BOOL  ; NC433_4_X 4ST_B 侧压B1左伺服强制中断
2081.09 BOOL  ; NC433_4_X 4ST_B 侧压B1左伺服预留
2081.10 BOOL  ; NC433_4_X 4ST_B 侧压B1左伺服预留
2081.11 BOOL  ; NC433_4_X 4ST_B 侧压B1左伺服预留
2081.12 BOOL  ; NC433_4_X 4ST_B 侧压B1左伺服数据写入
2081.13 BOOL  ; NC433_4_X 4ST_B 侧压B1左伺服数据读出
2081.14 BOOL  ; NC433_4_X 4ST_B 侧压B1左伺服数据保存
2081.15 BOOL  ; NC433_4_X 4ST_B 侧压B1左伺服预留
2082 CHANNEL  ; DA08V_2 通道2DA 转换值
2082.00 BOOL  ; NC433_4_Y 4ST_B 侧压B1右伺服存储器操作命令激活序列数
2082.01 BOOL  ; NC433_4_Y 4ST_B 侧压B1右伺服存储器操作命令起动
2082.02 BOOL  ; NC433_4_Y 4ST_B 侧压B1右伺服存储器操作命令独立起动
2082.03 BOOL  ; NC433_4_Y 4ST_B 侧压B1右伺服直接操作命令绝对移动
2082.04 BOOL  ; NC433_4_Y 4ST_B 侧压B1右伺服直接操作命令相对移动
2082.05 BOOL  ; NC433_4_Y 4ST_B 侧压B1右伺服直接操作命令中断进给
2082.06 BOOL  ; NC433_4_Y 4ST_B 侧压B1右伺服原点定位命令原点搜索
2082.07 BOOL  ; NC433_4_Y 4ST_B 侧压B1右伺服原点定位命令原点返回
2082.08 BOOL  ; NC433_4_Y 4ST_B 侧压B1右伺服原点定位命令当前位置预置
2082.09 BOOL  ; NC433_4_Y 4ST_B 侧压B1右伺服点动
2082.10 BOOL  ; NC433_4_Y 4ST_B 侧压B1右伺服点动方向(0=CW,1=CCW)
2082.11 BOOL  ; NC433_4_Y 4ST_B 侧压B1右伺服示教
2082.12 BOOL  ; NC433_4_Y 4ST_B 侧压B1右伺服错误清除
2082.13 BOOL  ; NC433_4_Y 4ST_B 侧压B1右伺服偏差计数器复位输出/ 原点调整命令输出
2082.14 BOOL  ; NC433_4_Y 4ST_B 侧压B1右伺服激活Override
2082.15 BOOL  ; NC433_4_Y 4ST_B 侧压B1右伺服停止
2083 CHANNEL  ; DA08V_2 通道3DA 转换值
2083.00 BOOL  ; NC433_4_Y 4ST_B 侧压B1右伺服预留
2083.01 BOOL  ; NC433_4_Y 4ST_B 侧压B1右伺服预留
2083.02 BOOL  ; NC433_4_Y 4ST_B 侧压B1右伺服预留
2083.03 BOOL  ; NC433_4_Y 4ST_B 侧压B1右伺服预留
2083.04 BOOL  ; NC433_4_Y 4ST_B 侧压B1右伺服预留
2083.05 BOOL  ; NC433_4_Y 4ST_B 侧压B1右伺服预留
2083.06 BOOL  ; NC433_4_Y 4ST_B 侧压B1右伺服预留
2083.07 BOOL  ; NC433_4_Y 4ST_B 侧压B1右伺服预留
2083.08 BOOL  ; NC433_4_Y 4ST_B 侧压B1右伺服强制中断
2083.09 BOOL  ; NC433_4_Y 4ST_B 侧压B1右伺服预留
2083.10 BOOL  ; NC433_4_Y 4ST_B 侧压B1右伺服预留
2083.11 BOOL  ; NC433_4_Y 4ST_B 侧压B1右伺服预留
2083.12 BOOL  ; NC433_4_Y 4ST_B 侧压B1右伺服数据写入
2083.13 BOOL  ; NC433_4_Y 4ST_B 侧压B1右伺服数据读出
2083.14 BOOL  ; NC433_4_Y 4ST_B 侧压B1右伺服数据保存
2083.15 BOOL  ; NC433_4_Y 4ST_B 侧压B1右伺服预留
2084 CHANNEL  ; DA08V_2 通道4DA 转换值
2084.00 BOOL  ; NC433_4_Z 4ST_B 侧压B2左伺服存储器操作命令激活序列数
2084.01 BOOL  ; NC433_4_Z 4ST_B 侧压B2左伺服存储器操作命令起动
2084.02 BOOL  ; NC433_4_Z 4ST_B 侧压B2左伺服存储器操作命令独立起动
2084.03 BOOL  ; NC433_4_Z 4ST_B 侧压B2左伺服直接操作命令绝对移动
2084.04 BOOL  ; NC433_4_Z 4ST_B 侧压B2左伺服直接操作命令相对移动
2084.05 BOOL  ; NC433_4_Z 4ST_B 侧压B2左伺服直接操作命令中断进给
2084.06 BOOL  ; NC433_4_Z 4ST_B 侧压B2左伺服原点定位命令原点搜索
2084.07 BOOL  ; NC433_4_Z 4ST_B 侧压B2左伺服原点定位命令原点返回
2084.08 BOOL  ; NC433_4_Z 4ST_B 侧压B2左伺服原点定位命令当前位置预置
2084.09 BOOL  ; NC433_4_Z 4ST_B 侧压B2左伺服点动
2084.10 BOOL  ; NC433_4_Z 4ST_B 侧压B2左伺服点动方向(0=CW,1=CCW)
2084.11 BOOL  ; NC433_4_Z 4ST_B 侧压B2左伺服示教
2084.12 BOOL  ; NC433_4_Z 4ST_B 侧压B2左伺服错误清除
2084.13 BOOL  ; NC433_4_Z 4ST_B 侧压B2左伺服偏差计数器复位输出/ 原点调整命令输出
2084.14 BOOL  ; NC433_4_Z 4ST_B 侧压B2左伺服激活Override
2084.15 BOOL  ; NC433_4_Z 4ST_B 侧压B2左伺服停止
2085 CHANNEL  ; DA08V_2 通道5DA 转换值
2085.00 BOOL  ; NC433_4_Z 4ST_B 侧压B2左伺服预留
2085.01 BOOL  ; NC433_4_Z 4ST_B 侧压B2左伺服预留
2085.02 BOOL  ; NC433_4_Z 4ST_B 侧压B2左伺服预留
2085.03 BOOL  ; NC433_4_Z 4ST_B 侧压B2左伺服预留
2085.04 BOOL  ; NC433_4_Z 4ST_B 侧压B2左伺服预留
2085.05 BOOL  ; NC433_4_Z 4ST_B 侧压B2左伺服预留
2085.06 BOOL  ; NC433_4_Z 4ST_B 侧压B2左伺服预留
2085.07 BOOL  ; NC433_4_Z 4ST_B 侧压B2左伺服预留
2085.08 BOOL  ; NC433_4_Z 4ST_B 侧压B2左伺服强制中断
2085.09 BOOL  ; NC433_4_Z 4ST_B 侧压B2左伺服预留
2085.10 BOOL  ; NC433_4_Z 4ST_B 侧压B2左伺服预留
2085.11 BOOL  ; NC433_4_Z 4ST_B 侧压B2左伺服预留
2085.12 BOOL  ; NC433_4_Z 4ST_B 侧压B2左伺服数据写入
2085.13 BOOL  ; NC433_4_Z 4ST_B 侧压B2左伺服数据读出
2085.14 BOOL  ; NC433_4_Z 4ST_B 侧压B2左伺服数据保存
2085.15 BOOL  ; NC433_4_Z 4ST_B 侧压B2左伺服预留
2086 CHANNEL  ; DA08V_2 通道6DA 转换值
2086.00 BOOL  ; NC433_4_U 4ST_B 侧压B2右伺服存储器操作命令激活序列数
2086.01 BOOL  ; NC433_4_U 4ST_B 侧压B2右伺服存储器操作命令起动
2086.02 BOOL  ; NC433_4_U 4ST_B 侧压B2右伺服存储器操作命令独立起动
2086.03 BOOL  ; NC433_4_U 4ST_B 侧压B2右伺服直接操作命令绝对移动
2086.04 BOOL  ; NC433_4_U 4ST_B 侧压B2右伺服直接操作命令相对移动
2086.05 BOOL  ; NC433_4_U 4ST_B 侧压B2右伺服直接操作命令中断进给
2086.06 BOOL  ; NC433_4_U 4ST_B 侧压B2右伺服原点定位命令原点搜索
2086.07 BOOL  ; NC433_4_U 4ST_B 侧压B2右伺服原点定位命令原点返回
2086.08 BOOL  ; NC433_4_U 4ST_B 侧压B2右伺服原点定位命令当前位置预置
2086.09 BOOL  ; NC433_4_U 4ST_B 侧压B2右伺服点动
2086.10 BOOL  ; NC433_4_U 4ST_B 侧压B2右伺服点动方向(0=CW,1=CCW)
2086.11 BOOL  ; NC433_4_U 4ST_B 侧压B2右伺服示教
2086.12 BOOL  ; NC433_4_U 4ST_B 侧压B2右伺服错误清除
2086.13 BOOL  ; NC433_4_U 4ST_B 侧压B2右伺服偏差计数器复位输出/ 原点调整命令输出
2086.14 BOOL  ; NC433_4_U 4ST_B 侧压B2右伺服激活Override
2086.15 BOOL  ; NC433_4_U 4ST_B 侧压B2右伺服停止
2087 CHANNEL  ; DA08V_2 通道7DA 转换值
2087.00 BOOL  ; NC433_4_U 4ST_B 侧压B2右伺服预留
2087.01 BOOL  ; NC433_4_U 4ST_B 侧压B2右伺服预留
2087.02 BOOL  ; NC433_4_U 4ST_B 侧压B2右伺服预留
2087.03 BOOL  ; NC433_4_U 4ST_B 侧压B2右伺服预留
2087.04 BOOL  ; NC433_4_U 4ST_B 侧压B2右伺服预留
2087.05 BOOL  ; NC433_4_U 4ST_B 侧压B2右伺服预留
2087.06 BOOL  ; NC433_4_U 4ST_B 侧压B2右伺服预留
2087.07 BOOL  ; NC433_4_U 4ST_B 侧压B2右伺服预留
2087.08 BOOL  ; NC433_4_U 4ST_B 侧压B2右伺服强制中断
2087.09 BOOL  ; NC433_4_U 4ST_B 侧压B2右伺服预留
2087.10 BOOL  ; NC433_4_U 4ST_B 侧压B2右伺服预留
2087.11 BOOL  ; NC433_4_U 4ST_B 侧压B2右伺服预留
2087.12 BOOL  ; NC433_4_U 4ST_B 侧压B2右伺服数据写入
2087.13 BOOL  ; NC433_4_U 4ST_B 侧压B2右伺服数据读出
2087.14 BOOL  ; NC433_4_U 4ST_B 侧压B2右伺服数据保存
2087.15 BOOL  ; NC433_4_U 4ST_B 侧压B2右伺服预留
2088 CHANNEL  ; DA08V_2 通道8DA 转换值
2088.00 BOOL  ; NC433_4_X 4ST_B 侧压B1左伺服预留
2088.01 BOOL  ; NC433_4_X 4ST_B 侧压B1左伺服预留
2088.02 BOOL  ; NC433_4_X 4ST_B 侧压B1左伺服预留
2088.03 BOOL  ; NC433_4_X 4ST_B 侧压B1左伺服预留
2088.04 BOOL  ; NC433_4_X 4ST_B 侧压B1左伺服等待存储器操作
2088.05 BOOL  ; NC433_4_X 4ST_B 侧压B1左伺服定位完成标志位
2088.06 BOOL  ; NC433_4_X 4ST_B 侧压B1左伺服无原点标志位
2088.07 BOOL  ; NC433_4_X 4ST_B 侧压B1左伺服原点停止标志位
2088.08 BOOL  ; NC433_4_X 4ST_B 侧压B1左伺服0 区监测标志位
2088.09 BOOL  ; NC433_4_X 4ST_B 侧压B1左伺服1 区监测标志位
2088.10 BOOL  ; NC433_4_X 4ST_B 侧压B1左伺服2 区监测标志位
2088.11 BOOL  ; NC433_4_X 4ST_B 侧压B1左伺服示教完成
2088.12 BOOL  ; NC433_4_X 4ST_B 侧压B1左伺服错误标志
2088.13 BOOL  ; NC433_4_X 4ST_B 侧压B1左伺服忙标志
2088.14 BOOL  ; NC433_4_X 4ST_B 侧压B1左伺服数据传送标志位
2088.15 BOOL  ; NC433_4_X 4ST_B 侧压B1左伺服减速停止执行标志位
2089.00 BOOL  ; NC433_4_X 4ST_B 侧压B1左伺服预留
2089.01 BOOL  ; NC433_4_X 4ST_B 侧压B1左伺服预留
2089.02 BOOL  ; NC433_4_X 4ST_B 侧压B1左伺服预留
2089.03 BOOL  ; NC433_4_X 4ST_B 侧压B1左伺服预留
2089.04 BOOL  ; NC433_4_X 4ST_B 侧压B1左伺服预留
2089.05 BOOL  ; NC433_4_X 4ST_B 侧压B1左伺服预留
2089.06 BOOL  ; NC433_4_X 4ST_B 侧压B1左伺服预留
2089.07 BOOL  ; NC433_4_X 4ST_B 侧压B1左伺服预留
2089.08 BOOL  ; NC433_4_X 4ST_B 侧压B1左伺服CW极限输入信号
2089.09 BOOL  ; NC433_4_X 4ST_B 侧压B1左伺服CCW极限输入信号
2089.10 BOOL  ; NC433_4_X 4ST_B 侧压B1左伺服原点接近输入信号
2089.11 BOOL  ; NC433_4_X 4ST_B 侧压B1左伺服原点输入信号
2089.12 BOOL  ; NC433_4_X 4ST_B 侧压B1左伺服中断输入信号
2089.13 BOOL  ; NC433_4_X 4ST_B 侧压B1左伺服紧急输入信号
2089.14 BOOL  ; NC433_4_X 4ST_B 侧压B1左伺服定位完成输入信号
2089.15 BOOL  ; NC433_4_X 4ST_B 侧压B1左伺服偏差计数器复位输出/ 原点调整命令输出
2090 CHANNEL  ; DA08V_3 通道使能
2090.00 BOOL  ; NC433_4_X 4ST_B 侧压B1左伺服错误代码
2090.01 BOOL  ; NC433_4_X 4ST_B 侧压B1左伺服错误代码
2090.02 BOOL  ; NC433_4_X 4ST_B 侧压B1左伺服错误代码
2090.03 BOOL  ; NC433_4_X 4ST_B 侧压B1左伺服错误代码
2090.04 BOOL  ; NC433_4_X 4ST_B 侧压B1左伺服错误代码
2090.05 BOOL  ; NC433_4_X 4ST_B 侧压B1左伺服错误代码
2090.06 BOOL  ; NC433_4_X 4ST_B 侧压B1左伺服错误代码
2090.07 BOOL  ; NC433_4_X 4ST_B 侧压B1左伺服错误代码
2090.08 BOOL  ; NC433_4_X 4ST_B 侧压B1左伺服错误代码
2090.09 BOOL  ; NC433_4_X 4ST_B 侧压B1左伺服错误代码
2090.10 BOOL  ; NC433_4_X 4ST_B 侧压B1左伺服错误代码
2090.11 BOOL  ; NC433_4_X 4ST_B 侧压B1左伺服错误代码
2090.12 BOOL  ; NC433_4_X 4ST_B 侧压B1左伺服错误代码
2090.13 BOOL  ; NC433_4_X 4ST_B 侧压B1左伺服错误代码
2090.14 BOOL  ; NC433_4_X 4ST_B 侧压B1左伺服错误代码
2090.15 BOOL  ; NC433_4_X 4ST_B 侧压B1左伺服错误代码
2091 CHANNEL  ; DA08V_3 通道1DA 转换值
2091.00 BOOL  ; NC433_4_Y 4ST_B 侧压B1右伺服预留
2091.01 BOOL  ; NC433_4_Y 4ST_B 侧压B1右伺服预留
2091.02 BOOL  ; NC433_4_Y 4ST_B 侧压B1右伺服预留
2091.03 BOOL  ; NC433_4_Y 4ST_B 侧压B1右伺服预留
2091.04 BOOL  ; NC433_4_Y 4ST_B 侧压B1右伺服等待存储器操作
2091.05 BOOL  ; NC433_4_Y 4ST_B 侧压B1右伺服定位完成标志位
2091.06 BOOL  ; NC433_4_Y 4ST_B 侧压B1右伺服无原点标志位
2091.07 BOOL  ; NC433_4_Y 4ST_B 侧压B1右伺服原点停止标志位
2091.08 BOOL  ; NC433_4_Y 4ST_B 侧压B1右伺服0 区监测标志位
2091.09 BOOL  ; NC433_4_Y 4ST_B 侧压B1右伺服1 区监测标志位
2091.10 BOOL  ; NC433_4_Y 4ST_B 侧压B1右伺服2 区监测标志位
2091.11 BOOL  ; NC433_4_Y 4ST_B 侧压B1右伺服示教完成
2091.12 BOOL  ; NC433_4_Y 4ST_B 侧压B1右伺服错误标志
2091.13 BOOL  ; NC433_4_Y 4ST_B 侧压B1右伺服忙标志
2091.14 BOOL  ; NC433_4_Y 4ST_B 侧压B1右伺服数据传送标志位
2091.15 BOOL  ; NC433_4_Y 4ST_B 侧压B1右伺服减速停止执行标志位
2092 CHANNEL  ; DA08V_3 通道2DA 转换值
2092.00 BOOL  ; NC433_4_Y 4ST_B 侧压B1右伺服预留
2092.01 BOOL  ; NC433_4_Y 4ST_B 侧压B1右伺服预留
2092.02 BOOL  ; NC433_4_Y 4ST_B 侧压B1右伺服预留
2092.03 BOOL  ; NC433_4_Y 4ST_B 侧压B1右伺服预留
2092.04 BOOL  ; NC433_4_Y 4ST_B 侧压B1右伺服预留
2092.05 BOOL  ; NC433_4_Y 4ST_B 侧压B1右伺服预留
2092.06 BOOL  ; NC433_4_Y 4ST_B 侧压B1右伺服预留
2092.07 BOOL  ; NC433_4_Y 4ST_B 侧压B1右伺服预留
2092.08 BOOL  ; NC433_4_Y 4ST_B 侧压B1右伺服CW极限输入信号
2092.09 BOOL  ; NC433_4_Y 4ST_B 侧压B1右伺服CCW极限输入信号
2092.10 BOOL  ; NC433_4_Y 4ST_B 侧压B1右伺服原点接近输入信号
2092.11 BOOL  ; NC433_4_Y 4ST_B 侧压B1右伺服原点输入信号
2092.12 BOOL  ; NC433_4_Y 4ST_B 侧压B1右伺服中断输入信号
2092.13 BOOL  ; NC433_4_Y 4ST_B 侧压B1右伺服紧急输入信号
2092.14 BOOL  ; NC433_4_Y 4ST_B 侧压B1右伺服定位完成输入信号
2092.15 BOOL  ; NC433_4_Y 4ST_B 侧压B1右伺服偏差计数器复位输出/ 原点调整命令输出
2093 CHANNEL  ; DA08V_3 通道3DA 转换值
2093.00 BOOL  ; NC433_4_Y 4ST_B 侧压B1右伺服错误代码
2093.01 BOOL  ; NC433_4_Y 4ST_B 侧压B1右伺服错误代码
2093.02 BOOL  ; NC433_4_Y 4ST_B 侧压B1右伺服错误代码
2093.03 BOOL  ; NC433_4_Y 4ST_B 侧压B1右伺服错误代码
2093.04 BOOL  ; NC433_4_Y 4ST_B 侧压B1右伺服错误代码
2093.05 BOOL  ; NC433_4_Y 4ST_B 侧压B1右伺服错误代码
2093.06 BOOL  ; NC433_4_Y 4ST_B 侧压B1右伺服错误代码
2093.07 BOOL  ; NC433_4_Y 4ST_B 侧压B1右伺服错误代码
2093.08 BOOL  ; NC433_4_Y 4ST_B 侧压B1右伺服错误代码
2093.09 BOOL  ; NC433_4_Y 4ST_B 侧压B1右伺服错误代码
2093.10 BOOL  ; NC433_4_Y 4ST_B 侧压B1右伺服错误代码
2093.11 BOOL  ; NC433_4_Y 4ST_B 侧压B1右伺服错误代码
2093.12 BOOL  ; NC433_4_Y 4ST_B 侧压B1右伺服错误代码
2093.13 BOOL  ; NC433_4_Y 4ST_B 侧压B1右伺服错误代码
2093.14 BOOL  ; NC433_4_Y 4ST_B 侧压B1右伺服错误代码
2093.15 BOOL  ; NC433_4_Y 4ST_B 侧压B1右伺服错误代码
2094 CHANNEL  ; DA08V_3 通道4DA 转换值
2094.00 BOOL  ; NC433_4_Z 4ST_B 侧压B2左伺服预留
2094.01 BOOL  ; NC433_4_Z 4ST_B 侧压B2左伺服预留
2094.02 BOOL  ; NC433_4_Z 4ST_B 侧压B2左伺服预留
2094.03 BOOL  ; NC433_4_Z 4ST_B 侧压B2左伺服预留
2094.04 BOOL  ; NC433_4_Z 4ST_B 侧压B2左伺服等待存储器操作
2094.05 BOOL  ; NC433_4_Z 4ST_B 侧压B2左伺服定位完成标志位
2094.06 BOOL  ; NC433_4_Z 4ST_B 侧压B2左伺服无原点标志位
2094.07 BOOL  ; NC433_4_Z 4ST_B 侧压B2左伺服原点停止标志位
2094.08 BOOL  ; NC433_4_Z 4ST_B 侧压B2左伺服0 区监测标志位
2094.09 BOOL  ; NC433_4_Z 4ST_B 侧压B2左伺服1 区监测标志位
2094.10 BOOL  ; NC433_4_Z 4ST_B 侧压B2左伺服2 区监测标志位
2094.11 BOOL  ; NC433_4_Z 4ST_B 侧压B2左伺服示教完成
2094.12 BOOL  ; NC433_4_Z 4ST_B 侧压B2左伺服错误标志
2094.13 BOOL  ; NC433_4_Z 4ST_B 侧压B2左伺服忙标志
2094.14 BOOL  ; NC433_4_Z 4ST_B 侧压B2左伺服数据传送标志位
2094.15 BOOL  ; NC433_4_Z 4ST_B 侧压B2左伺服减速停止执行标志位
2095 CHANNEL  ; DA08V_3 通道5DA 转换值
2095.00 BOOL  ; NC433_4_Z 4ST_B 侧压B2左伺服预留
2095.01 BOOL  ; NC433_4_Z 4ST_B 侧压B2左伺服预留
2095.02 BOOL  ; NC433_4_Z 4ST_B 侧压B2左伺服预留
2095.03 BOOL  ; NC433_4_Z 4ST_B 侧压B2左伺服预留
2095.04 BOOL  ; NC433_4_Z 4ST_B 侧压B2左伺服预留
2095.05 BOOL  ; NC433_4_Z 4ST_B 侧压B2左伺服预留
2095.06 BOOL  ; NC433_4_Z 4ST_B 侧压B2左伺服预留
2095.07 BOOL  ; NC433_4_Z 4ST_B 侧压B2左伺服预留
2095.08 BOOL  ; NC433_4_Z 4ST_B 侧压B2左伺服CW极限输入信号
2095.09 BOOL  ; NC433_4_Z 4ST_B 侧压B2左伺服CCW极限输入信号
2095.10 BOOL  ; NC433_4_Z 4ST_B 侧压B2左伺服原点接近输入信号
2095.11 BOOL  ; NC433_4_Z 4ST_B 侧压B2左伺服原点输入信号
2095.12 BOOL  ; NC433_4_Z 4ST_B 侧压B2左伺服中断输入信号
2095.13 BOOL  ; NC433_4_Z 4ST_B 侧压B2左伺服紧急输入信号
2095.14 BOOL  ; NC433_4_Z 4ST_B 侧压B2左伺服定位完成输入信号
2095.15 BOOL  ; NC433_4_Z 4ST_B 侧压B2左伺服偏差计数器复位输出/ 原点调整命令输出
2096 CHANNEL  ; DA08V_3 通道6DA 转换值
2096.00 BOOL  ; NC433_4_Z 4ST_B 侧压B2左伺服错误代码
2096.01 BOOL  ; NC433_4_Z 4ST_B 侧压B2左伺服错误代码
2096.02 BOOL  ; NC433_4_Z 4ST_B 侧压B2左伺服错误代码
2096.03 BOOL  ; NC433_4_Z 4ST_B 侧压B2左伺服错误代码
2096.04 BOOL  ; NC433_4_Z 4ST_B 侧压B2左伺服错误代码
2096.05 BOOL  ; NC433_4_Z 4ST_B 侧压B2左伺服错误代码
2096.06 BOOL  ; NC433_4_Z 4ST_B 侧压B2左伺服错误代码
2096.07 BOOL  ; NC433_4_Z 4ST_B 侧压B2左伺服错误代码
2096.08 BOOL  ; NC433_4_Z 4ST_B 侧压B2左伺服错误代码
2096.09 BOOL  ; NC433_4_Z 4ST_B 侧压B2左伺服错误代码
2096.10 BOOL  ; NC433_4_Z 4ST_B 侧压B2左伺服错误代码
2096.11 BOOL  ; NC433_4_Z 4ST_B 侧压B2左伺服错误代码
2096.12 BOOL  ; NC433_4_Z 4ST_B 侧压B2左伺服错误代码
2096.13 BOOL  ; NC433_4_Z 4ST_B 侧压B2左伺服错误代码
2096.14 BOOL  ; NC433_4_Z 4ST_B 侧压B2左伺服错误代码
2096.15 BOOL  ; NC433_4_Z 4ST_B 侧压B2左伺服错误代码
2097 CHANNEL  ; DA08V_3 通道7DA 转换值
2097.00 BOOL  ; NC433_4_U 4ST_B 侧压B2右伺服预留
2097.01 BOOL  ; NC433_4_U 4ST_B 侧压B2右伺服预留
2097.02 BOOL  ; NC433_4_U 4ST_B 侧压B2右伺服预留
2097.03 BOOL  ; NC433_4_U 4ST_B 侧压B2右伺服预留
2097.04 BOOL  ; NC433_4_U 4ST_B 侧压B2右伺服等待存储器操作
2097.05 BOOL  ; NC433_4_U 4ST_B 侧压B2右伺服定位完成标志位
2097.06 BOOL  ; NC433_4_U 4ST_B 侧压B2右伺服无原点标志位
2097.07 BOOL  ; NC433_4_U 4ST_B 侧压B2右伺服原点停止标志位
2097.08 BOOL  ; NC433_4_U 4ST_B 侧压B2右伺服0 区监测标志位
2097.09 BOOL  ; NC433_4_U 4ST_B 侧压B2右伺服1 区监测标志位
2097.10 BOOL  ; NC433_4_U 4ST_B 侧压B2右伺服2 区监测标志位
2097.11 BOOL  ; NC433_4_U 4ST_B 侧压B2右伺服示教完成
2097.12 BOOL  ; NC433_4_U 4ST_B 侧压B2右伺服错误标志
2097.13 BOOL  ; NC433_4_U 4ST_B 侧压B2右伺服忙标志
2097.14 BOOL  ; NC433_4_U 4ST_B 侧压B2右伺服数据传送标志位
2097.15 BOOL  ; NC433_4_U 4ST_B 侧压B2右伺服减速停止执行标志位
2098 CHANNEL  ; DA08V_3 通道8DA 转换值
2098.00 BOOL  ; NC433_4_U 4ST_B 侧压B2右伺服预留
2098.01 BOOL  ; NC433_4_U 4ST_B 侧压B2右伺服预留
2098.02 BOOL  ; NC433_4_U 4ST_B 侧压B2右伺服预留
2098.03 BOOL  ; NC433_4_U 4ST_B 侧压B2右伺服预留
2098.04 BOOL  ; NC433_4_U 4ST_B 侧压B2右伺服预留
2098.05 BOOL  ; NC433_4_U 4ST_B 侧压B2右伺服预留
2098.06 BOOL  ; NC433_4_U 4ST_B 侧压B2右伺服预留
2098.07 BOOL  ; NC433_4_U 4ST_B 侧压B2右伺服预留
2098.08 BOOL  ; NC433_4_U 4ST_B 侧压B2右伺服CW极限输入信号
2098.09 BOOL  ; NC433_4_U 4ST_B 侧压B2右伺服CCW极限输入信号
2098.10 BOOL  ; NC433_4_U 4ST_B 侧压B2右伺服原点接近输入信号
2098.11 BOOL  ; NC433_4_U 4ST_B 侧压B2右伺服原点输入信号
2098.12 BOOL  ; NC433_4_U 4ST_B 侧压B2右伺服中断输入信号
2098.13 BOOL  ; NC433_4_U 4ST_B 侧压B2右伺服紧急输入信号
2098.14 BOOL  ; NC433_4_U 4ST_B 侧压B2右伺服定位完成输入信号
2098.15 BOOL  ; NC433_4_U 4ST_B 侧压B2右伺服偏差计数器复位输出/ 原点调整命令输出
2099.00 BOOL  ; NC433_4_U 4ST_B 侧压B2右伺服错误代码
2099.01 BOOL  ; NC433_4_U 4ST_B 侧压B2右伺服错误代码
2099.02 BOOL  ; NC433_4_U 4ST_B 侧压B2右伺服错误代码
2099.03 BOOL  ; NC433_4_U 4ST_B 侧压B2右伺服错误代码
2099.04 BOOL  ; NC433_4_U 4ST_B 侧压B2右伺服错误代码
2099.05 BOOL  ; NC433_4_U 4ST_B 侧压B2右伺服错误代码
2099.06 BOOL  ; NC433_4_U 4ST_B 侧压B2右伺服错误代码
2099.07 BOOL  ; NC433_4_U 4ST_B 侧压B2右伺服错误代码
2099.08 BOOL  ; NC433_4_U 4ST_B 侧压B2右伺服错误代码
2099.09 BOOL  ; NC433_4_U 4ST_B 侧压B2右伺服错误代码
2099.10 BOOL  ; NC433_4_U 4ST_B 侧压B2右伺服错误代码
2099.11 BOOL  ; NC433_4_U 4ST_B 侧压B2右伺服错误代码
2099.12 BOOL  ; NC433_4_U 4ST_B 侧压B2右伺服错误代码
2099.13 BOOL  ; NC433_4_U 4ST_B 侧压B2右伺服错误代码
2099.14 BOOL  ; NC433_4_U 4ST_B 侧压B2右伺服错误代码
2099.15 BOOL  ; NC433_4_U 4ST_B 侧压B2右伺服错误代码
20.00 BOOL  ; 热压C上层上板左加热启动
20.01 BOOL  ; 热压C上层上板中加热启动
20.02 BOOL  ; 热压C上层上板右加热启动
20.03 BOOL  ; 热压C上层下板左加热启动
20.04 BOOL  ; 热压C上层下板中加热启动
20.05 BOOL  ; 热压C上层下板右加热启动
2100 CHANNEL  ; DA08V_4 通道使能
2100.00 BOOL  ; NC433_5_X 4ST_B 侧压B3左伺服存储器操作命令激活序列数
2100.01 BOOL  ; NC433_5_X 4ST_B 侧压B3左伺服存储器操作命令起动
2100.02 BOOL  ; NC433_5_X 4ST_B 侧压B3左伺服存储器操作命令独立起动
2100.03 BOOL  ; NC433_5_X 4ST_B 侧压B3左伺服直接操作命令绝对移动
2100.04 BOOL  ; NC433_5_X 4ST_B 侧压B3左伺服直接操作命令相对移动
2100.05 BOOL  ; NC433_5_X 4ST_B 侧压B3左伺服直接操作命令中断进给
2100.06 BOOL  ; NC433_5_X 4ST_B 侧压B3左伺服原点定位命令原点搜索
2100.07 BOOL  ; NC433_5_X 4ST_B 侧压B3左伺服原点定位命令原点返回
2100.08 BOOL  ; NC433_5_X 4ST_B 侧压B3左伺服原点定位命令当前位置预置
2100.09 BOOL  ; NC433_5_X 4ST_B 侧压B3左伺服点动
2100.10 BOOL  ; NC433_5_X 4ST_B 侧压B3左伺服点动方向(0=CW,1=CCW)
2100.11 BOOL  ; NC433_5_X 4ST_B 侧压B3左伺服示教
2100.12 BOOL  ; NC433_5_X 4ST_B 侧压B3左伺服错误清除
2100.13 BOOL  ; NC433_5_X 4ST_B 侧压B3左伺服偏差计数器复位输出/ 原点调整命令输出
2100.14 BOOL  ; NC433_5_X 4ST_B 侧压B3左伺服激活Override
2100.15 BOOL  ; NC433_5_X 4ST_B 侧压B3左伺服停止
2101 CHANNEL  ; DA08V_4 通道1DA 转换值
2101.00 BOOL  ; NC433_5_X 4ST_B 侧压B3左伺服预留
2101.01 BOOL  ; NC433_5_X 4ST_B 侧压B3左伺服预留
2101.02 BOOL  ; NC433_5_X 4ST_B 侧压B3左伺服预留
2101.03 BOOL  ; NC433_5_X 4ST_B 侧压B3左伺服预留
2101.04 BOOL  ; NC433_5_X 4ST_B 侧压B3左伺服预留
2101.05 BOOL  ; NC433_5_X 4ST_B 侧压B3左伺服预留
2101.06 BOOL  ; NC433_5_X 4ST_B 侧压B3左伺服预留
2101.07 BOOL  ; NC433_5_X 4ST_B 侧压B3左伺服预留
2101.08 BOOL  ; NC433_5_X 4ST_B 侧压B3左伺服强制中断
2101.09 BOOL  ; NC433_5_X 4ST_B 侧压B3左伺服预留
2101.10 BOOL  ; NC433_5_X 4ST_B 侧压B3左伺服预留
2101.11 BOOL  ; NC433_5_X 4ST_B 侧压B3左伺服预留
2101.12 BOOL  ; NC433_5_X 4ST_B 侧压B3左伺服数据写入
2101.13 BOOL  ; NC433_5_X 4ST_B 侧压B3左伺服数据读出
2101.14 BOOL  ; NC433_5_X 4ST_B 侧压B3左伺服数据保存
2101.15 BOOL  ; NC433_5_X 4ST_B 侧压B3左伺服预留
2102 CHANNEL  ; DA08V_4 通道2DA 转换值
2102.00 BOOL  ; NC433_5_Y 4ST_B 侧压B3右伺服存储器操作命令激活序列数
2102.01 BOOL  ; NC433_5_Y 4ST_B 侧压B3右伺服存储器操作命令起动
2102.02 BOOL  ; NC433_5_Y 4ST_B 侧压B3右伺服存储器操作命令独立起动
2102.03 BOOL  ; NC433_5_Y 4ST_B 侧压B3右伺服直接操作命令绝对移动
2102.04 BOOL  ; NC433_5_Y 4ST_B 侧压B3右伺服直接操作命令相对移动
2102.05 BOOL  ; NC433_5_Y 4ST_B 侧压B3右伺服直接操作命令中断进给
2102.06 BOOL  ; NC433_5_Y 4ST_B 侧压B3右伺服原点定位命令原点搜索
2102.07 BOOL  ; NC433_5_Y 4ST_B 侧压B3右伺服原点定位命令原点返回
2102.08 BOOL  ; NC433_5_Y 4ST_B 侧压B3右伺服原点定位命令当前位置预置
2102.09 BOOL  ; NC433_5_Y 4ST_B 侧压B3右伺服点动
2102.10 BOOL  ; NC433_5_Y 4ST_B 侧压B3右伺服点动方向(0=CW,1=CCW)
2102.11 BOOL  ; NC433_5_Y 4ST_B 侧压B3右伺服示教
2102.12 BOOL  ; NC433_5_Y 4ST_B 侧压B3右伺服错误清除
2102.13 BOOL  ; NC433_5_Y 4ST_B 侧压B3右伺服偏差计数器复位输出/ 原点调整命令输出
2102.14 BOOL  ; NC433_5_Y 4ST_B 侧压B3右伺服激活Override
2102.15 BOOL  ; NC433_5_Y 4ST_B 侧压B3右伺服停止
2103 CHANNEL  ; DA08V_4 通道3DA 转换值
2103.00 BOOL  ; NC433_5_Y 4ST_B 侧压B3右伺服预留
2103.01 BOOL  ; NC433_5_Y 4ST_B 侧压B3右伺服预留
2103.02 BOOL  ; NC433_5_Y 4ST_B 侧压B3右伺服预留
2103.03 BOOL  ; NC433_5_Y 4ST_B 侧压B3右伺服预留
2103.04 BOOL  ; NC433_5_Y 4ST_B 侧压B3右伺服预留
2103.05 BOOL  ; NC433_5_Y 4ST_B 侧压B3右伺服预留
2103.06 BOOL  ; NC433_5_Y 4ST_B 侧压B3右伺服预留
2103.07 BOOL  ; NC433_5_Y 4ST_B 侧压B3右伺服预留
2103.08 BOOL  ; NC433_5_Y 4ST_B 侧压B3右伺服强制中断
2103.09 BOOL  ; NC433_5_Y 4ST_B 侧压B3右伺服预留
2103.10 BOOL  ; NC433_5_Y 4ST_B 侧压B3右伺服预留
2103.11 BOOL  ; NC433_5_Y 4ST_B 侧压B3右伺服预留
2103.12 BOOL  ; NC433_5_Y 4ST_B 侧压B3右伺服数据写入
2103.13 BOOL  ; NC433_5_Y 4ST_B 侧压B3右伺服数据读出
2103.14 BOOL  ; NC433_5_Y 4ST_B 侧压B3右伺服数据保存
2103.15 BOOL  ; NC433_5_Y 4ST_B 侧压B3右伺服预留
2104 CHANNEL  ; DA08V_4 通道4DA 转换值
2104.00 BOOL  ; NC433_5_Z 4ST_B 侧压B4左伺服存储器操作命令激活序列数
2104.01 BOOL  ; NC433_5_Z 4ST_B 侧压B4左伺服存储器操作命令起动
2104.02 BOOL  ; NC433_5_Z 4ST_B 侧压B4左伺服存储器操作命令独立起动
2104.03 BOOL  ; NC433_5_Z 4ST_B 侧压B4左伺服直接操作命令绝对移动
2104.04 BOOL  ; NC433_5_Z 4ST_B 侧压B4左伺服直接操作命令相对移动
2104.05 BOOL  ; NC433_5_Z 4ST_B 侧压B4左伺服直接操作命令中断进给
2104.06 BOOL  ; NC433_5_Z 4ST_B 侧压B4左伺服原点定位命令原点搜索
2104.07 BOOL  ; NC433_5_Z 4ST_B 侧压B4左伺服原点定位命令原点返回
2104.08 BOOL  ; NC433_5_Z 4ST_B 侧压B4左伺服原点定位命令当前位置预置
2104.09 BOOL  ; NC433_5_Z 4ST_B 侧压B4左伺服点动
2104.10 BOOL  ; NC433_5_Z 4ST_B 侧压B4左伺服点动方向(0=CW,1=CCW)
2104.11 BOOL  ; NC433_5_Z 4ST_B 侧压B4左伺服示教
2104.12 BOOL  ; NC433_5_Z 4ST_B 侧压B4左伺服错误清除
2104.13 BOOL  ; NC433_5_Z 4ST_B 侧压B4左伺服偏差计数器复位输出/ 原点调整命令输出
2104.14 BOOL  ; NC433_5_Z 4ST_B 侧压B4左伺服激活Override
2104.15 BOOL  ; NC433_5_Z 4ST_B 侧压B4左伺服停止
2105 CHANNEL  ; DA08V_4 通道5DA 转换值
2105.00 BOOL  ; NC433_5_Z 4ST_B 侧压B4左伺服预留
2105.01 BOOL  ; NC433_5_Z 4ST_B 侧压B4左伺服预留
2105.02 BOOL  ; NC433_5_Z 4ST_B 侧压B4左伺服预留
2105.03 BOOL  ; NC433_5_Z 4ST_B 侧压B4左伺服预留
2105.04 BOOL  ; NC433_5_Z 4ST_B 侧压B4左伺服预留
2105.05 BOOL  ; NC433_5_Z 4ST_B 侧压B4左伺服预留
2105.06 BOOL  ; NC433_5_Z 4ST_B 侧压B4左伺服预留
2105.07 BOOL  ; NC433_5_Z 4ST_B 侧压B4左伺服预留
2105.08 BOOL  ; NC433_5_Z 4ST_B 侧压B4左伺服强制中断
2105.09 BOOL  ; NC433_5_Z 4ST_B 侧压B4左伺服预留
2105.10 BOOL  ; NC433_5_Z 4ST_B 侧压B4左伺服预留
2105.11 BOOL  ; NC433_5_Z 4ST_B 侧压B4左伺服预留
2105.12 BOOL  ; NC433_5_Z 4ST_B 侧压B4左伺服数据写入
2105.13 BOOL  ; NC433_5_Z 4ST_B 侧压B4左伺服数据读出
2105.14 BOOL  ; NC433_5_Z 4ST_B 侧压B4左伺服数据保存
2105.15 BOOL  ; NC433_5_Z 4ST_B 侧压B4左伺服预留
2106 CHANNEL  ; DA08V_4 通道6DA 转换值
2106.00 BOOL  ; NC433_5_U 4ST_B 侧压B4右伺服存储器操作命令激活序列数
2106.01 BOOL  ; NC433_5_U 4ST_B 侧压B4右伺服存储器操作命令起动
2106.02 BOOL  ; NC433_5_U 4ST_B 侧压B4右伺服存储器操作命令独立起动
2106.03 BOOL  ; NC433_5_U 4ST_B 侧压B4右伺服直接操作命令绝对移动
2106.04 BOOL  ; NC433_5_U 4ST_B 侧压B4右伺服直接操作命令相对移动
2106.05 BOOL  ; NC433_5_U 4ST_B 侧压B4右伺服直接操作命令中断进给
2106.06 BOOL  ; NC433_5_U 4ST_B 侧压B4右伺服原点定位命令原点搜索
2106.07 BOOL  ; NC433_5_U 4ST_B 侧压B4右伺服原点定位命令原点返回
2106.08 BOOL  ; NC433_5_U 4ST_B 侧压B4右伺服原点定位命令当前位置预置
2106.09 BOOL  ; NC433_5_U 4ST_B 侧压B4右伺服点动
2106.10 BOOL  ; NC433_5_U 4ST_B 侧压B4右伺服点动方向(0=CW,1=CCW)
2106.11 BOOL  ; NC433_5_U 4ST_B 侧压B4右伺服示教
2106.12 BOOL  ; NC433_5_U 4ST_B 侧压B4右伺服错误清除
2106.13 BOOL  ; NC433_5_U 4ST_B 侧压B4右伺服偏差计数器复位输出/ 原点调整命令输出
2106.14 BOOL  ; NC433_5_U 4ST_B 侧压B4右伺服激活Override
2106.15 BOOL  ; NC433_5_U 300-1ST 焊后移载机械手X轴停止
2107 CHANNEL  ; DA08V_4 通道7DA 转换值
2107.00 BOOL  ; NC433_5_U 4ST_B 侧压B4右伺服预留
2107.01 BOOL  ; NC433_5_U 4ST_B 侧压B4右伺服预留
2107.02 BOOL  ; NC433_5_U 4ST_B 侧压B4右伺服预留
2107.03 BOOL  ; NC433_5_U 4ST_B 侧压B4右伺服预留
2107.04 BOOL  ; NC433_5_U 4ST_B 侧压B4右伺服预留
2107.05 BOOL  ; NC433_5_U 4ST_B 侧压B4右伺服预留
2107.06 BOOL  ; NC433_5_U 4ST_B 侧压B4右伺服预留
2107.07 BOOL  ; NC433_5_U 4ST_B 侧压B4右伺服预留
2107.08 BOOL  ; NC433_5_U 4ST_B 侧压B4右伺服强制中断
2107.09 BOOL  ; NC433_5_U 4ST_B 侧压B4右伺服预留
2107.10 BOOL  ; NC433_5_U 4ST_B 侧压B4右伺服预留
2107.11 BOOL  ; NC433_5_U 4ST_B 侧压B4右伺服预留
2107.12 BOOL  ; NC433_5_U 4ST_B 侧压B4右伺服数据写入
2107.13 BOOL  ; NC433_5_U 4ST_B 侧压B4右伺服数据读出
2107.14 BOOL  ; NC433_5_U 4ST_B 侧压B4右伺服数据保存
2107.15 BOOL  ; NC433_5_U 4ST_B 侧压B4右伺服预留
2108 CHANNEL  ; DA08V_4 通道8DA 转换值
2108.00 BOOL  ; NC433_5_X 4ST_B 侧压B3左伺服预留
2108.01 BOOL  ; NC433_5_X 4ST_B 侧压B3左伺服预留
2108.02 BOOL  ; NC433_5_X 4ST_B 侧压B3左伺服预留
2108.03 BOOL  ; NC433_5_X 4ST_B 侧压B3左伺服预留
2108.04 BOOL  ; NC433_5_X 4ST_B 侧压B3左伺服等待存储器操作
2108.05 BOOL  ; NC433_5_X 4ST_B 侧压B3左伺服定位完成标志位
2108.06 BOOL  ; NC433_5_X 4ST_B 侧压B3左伺服无原点标志位
2108.07 BOOL  ; NC433_5_X 4ST_B 侧压B3左伺服原点停止标志位
2108.08 BOOL  ; NC433_5_X 4ST_B 侧压B3左伺服0 区监测标志位
2108.09 BOOL  ; NC433_5_X 4ST_B 侧压B3左伺服1 区监测标志位
2108.10 BOOL  ; NC433_5_X 4ST_B 侧压B3左伺服2 区监测标志位
2108.11 BOOL  ; NC433_5_X 4ST_B 侧压B3左伺服示教完成
2108.12 BOOL  ; NC433_5_X 4ST_B 侧压B3左伺服错误标志
2108.13 BOOL  ; NC433_5_X 4ST_B 侧压B3左伺服忙标志
2108.14 BOOL  ; NC433_5_X 4ST_B 侧压B3左伺服数据传送标志位
2108.15 BOOL  ; NC433_5_X 4ST_B 侧压B3左伺服减速停止执行标志位
2109.00 BOOL  ; NC433_5_X 4ST_B 侧压B3左伺服预留
2109.01 BOOL  ; NC433_5_X 4ST_B 侧压B3左伺服预留
2109.02 BOOL  ; NC433_5_X 4ST_B 侧压B3左伺服预留
2109.03 BOOL  ; NC433_5_X 4ST_B 侧压B3左伺服预留
2109.04 BOOL  ; NC433_5_X 4ST_B 侧压B3左伺服预留
2109.05 BOOL  ; NC433_5_X 4ST_B 侧压B3左伺服预留
2109.06 BOOL  ; NC433_5_X 4ST_B 侧压B3左伺服预留
2109.07 BOOL  ; NC433_5_X 4ST_B 侧压B3左伺服预留
2109.08 BOOL  ; NC433_5_X 4ST_B 侧压B3左伺服CW极限输入信号
2109.09 BOOL  ; NC433_5_X 4ST_B 侧压B3左伺服CCW极限输入信号
2109.10 BOOL  ; NC433_5_X 4ST_B 侧压B3左伺服原点接近输入信号
2109.11 BOOL  ; NC433_5_X 4ST_B 侧压B3左伺服原点输入信号
2109.12 BOOL  ; NC433_5_X 4ST_B 侧压B3左伺服中断输入信号
2109.13 BOOL  ; NC433_5_X 4ST_B 侧压B3左伺服紧急输入信号
2109.14 BOOL  ; NC433_5_X 4ST_B 侧压B3左伺服定位完成输入信号
2109.15 BOOL  ; NC433_5_X 4ST_B 侧压B3左伺服偏差计数器复位输出/ 原点调整命令输出
2110.00 BOOL  ; NC433_5_X 4ST_B 侧压B3左伺服错误代码
2110.01 BOOL  ; NC433_5_X 4ST_B 侧压B3左伺服错误代码
2110.02 BOOL  ; NC433_5_X 4ST_B 侧压B3左伺服错误代码
2110.03 BOOL  ; NC433_5_X 4ST_B 侧压B3左伺服错误代码
2110.04 BOOL  ; NC433_5_X 4ST_B 侧压B3左伺服错误代码
2110.05 BOOL  ; NC433_5_X 4ST_B 侧压B3左伺服错误代码
2110.06 BOOL  ; NC433_5_X 4ST_B 侧压B3左伺服错误代码
2110.07 BOOL  ; NC433_5_X 4ST_B 侧压B3左伺服错误代码
2110.08 BOOL  ; NC433_5_X 4ST_B 侧压B3左伺服错误代码
2110.09 BOOL  ; NC433_5_X 4ST_B 侧压B3左伺服错误代码
2110.10 BOOL  ; NC433_5_X 4ST_B 侧压B3左伺服错误代码
2110.11 BOOL  ; NC433_5_X 4ST_B 侧压B3左伺服错误代码
2110.12 BOOL  ; NC433_5_X 4ST_B 侧压B3左伺服错误代码
2110.13 BOOL  ; NC433_5_X 4ST_B 侧压B3左伺服错误代码
2110.14 BOOL  ; NC433_5_X 4ST_B 侧压B3左伺服错误代码
2110.15 BOOL  ; NC433_5_X 4ST_B 侧压B3左伺服错误代码
2111.00 BOOL  ; NC433_5_Y 4ST_B 侧压B3右伺服预留
2111.01 BOOL  ; NC433_5_Y 4ST_B 侧压B3右伺服预留
2111.02 BOOL  ; NC433_5_Y 4ST_B 侧压B3右伺服预留
2111.03 BOOL  ; NC433_5_Y 4ST_B 侧压B3右伺服预留
2111.04 BOOL  ; NC433_5_Y 4ST_B 侧压B3右伺服等待存储器操作
2111.05 BOOL  ; NC433_5_Y 4ST_B 侧压B3右伺服定位完成标志位
2111.06 BOOL  ; NC433_5_Y 4ST_B 侧压B3右伺服无原点标志位
2111.07 BOOL  ; NC433_5_Y 4ST_B 侧压B3右伺服原点停止标志位
2111.08 BOOL  ; NC433_5_Y 4ST_B 侧压B3右伺服0 区监测标志位
2111.09 BOOL  ; NC433_5_Y 4ST_B 侧压B3右伺服1 区监测标志位
2111.10 BOOL  ; NC433_5_Y 4ST_B 侧压B3右伺服2 区监测标志位
2111.11 BOOL  ; NC433_5_Y 4ST_B 侧压B3右伺服示教完成
2111.12 BOOL  ; NC433_5_Y 4ST_B 侧压B3右伺服错误标志
2111.13 BOOL  ; NC433_5_Y 4ST_B 侧压B3右伺服忙标志
2111.14 BOOL  ; NC433_5_Y 4ST_B 侧压B3右伺服数据传送标志位
2111.15 BOOL  ; NC433_5_Y 4ST_B 侧压B3右伺服减速停止执行标志位
2112.00 BOOL  ; NC433_5_Y 4ST_B 侧压B3右伺服预留
2112.01 BOOL  ; NC433_5_Y 4ST_B 侧压B3右伺服预留
2112.02 BOOL  ; NC433_5_Y 4ST_B 侧压B3右伺服预留
2112.03 BOOL  ; NC433_5_Y 4ST_B 侧压B3右伺服预留
2112.04 BOOL  ; NC433_5_Y 4ST_B 侧压B3右伺服预留
2112.05 BOOL  ; NC433_5_Y 4ST_B 侧压B3右伺服预留
2112.06 BOOL  ; NC433_5_Y 4ST_B 侧压B3右伺服预留
2112.07 BOOL  ; NC433_5_Y 4ST_B 侧压B3右伺服预留
2112.08 BOOL  ; NC433_5_Y 4ST_B 侧压B3右伺服CW极限输入信号
2112.09 BOOL  ; NC433_5_Y 4ST_B 侧压B3右伺服CCW极限输入信号
2112.10 BOOL  ; NC433_5_Y 4ST_B 侧压B3右伺服原点接近输入信号
2112.11 BOOL  ; NC433_5_Y 4ST_B 侧压B3右伺服原点输入信号
2112.12 BOOL  ; NC433_5_Y 4ST_B 侧压B3右伺服中断输入信号
2112.13 BOOL  ; NC433_5_Y 4ST_B 侧压B3右伺服紧急输入信号
2112.14 BOOL  ; NC433_5_Y 4ST_B 侧压B3右伺服定位完成输入信号
2112.15 BOOL  ; NC433_5_Y 4ST_B 侧压B3右伺服偏差计数器复位输出/ 原点调整命令输出
2113.00 BOOL  ; NC433_5_Y 4ST_B 侧压B3右伺服错误代码
2113.01 BOOL  ; NC433_5_Y 4ST_B 侧压B3右伺服错误代码
2113.02 BOOL  ; NC433_5_Y 4ST_B 侧压B3右伺服错误代码
2113.03 BOOL  ; NC433_5_Y 4ST_B 侧压B3右伺服错误代码
2113.04 BOOL  ; NC433_5_Y 4ST_B 侧压B3右伺服错误代码
2113.05 BOOL  ; NC433_5_Y 4ST_B 侧压B3右伺服错误代码
2113.06 BOOL  ; NC433_5_Y 4ST_B 侧压B3右伺服错误代码
2113.07 BOOL  ; NC433_5_Y 4ST_B 侧压B3右伺服错误代码
2113.08 BOOL  ; NC433_5_Y 4ST_B 侧压B3右伺服错误代码
2113.09 BOOL  ; NC433_5_Y 4ST_B 侧压B3右伺服错误代码
2113.10 BOOL  ; NC433_5_Y 4ST_B 侧压B3右伺服错误代码
2113.11 BOOL  ; NC433_5_Y 4ST_B 侧压B3右伺服错误代码
2113.12 BOOL  ; NC433_5_Y 4ST_B 侧压B3右伺服错误代码
2113.13 BOOL  ; NC433_5_Y 4ST_B 侧压B3右伺服错误代码
2113.14 BOOL  ; NC433_5_Y 4ST_B 侧压B3右伺服错误代码
2113.15 BOOL  ; NC433_5_Y 4ST_B 侧压B3右伺服错误代码
2114.00 BOOL  ; NC433_5_Z 4ST_B 侧压B4左伺服预留
2114.01 BOOL  ; NC433_5_Z 4ST_B 侧压B4左伺服预留
2114.02 BOOL  ; NC433_5_Z 4ST_B 侧压B4左伺服预留
2114.03 BOOL  ; NC433_5_Z 4ST_B 侧压B4左伺服预留
2114.04 BOOL  ; NC433_5_Z 4ST_B 侧压B4左伺服等待存储器操作
2114.05 BOOL  ; NC433_5_Z 4ST_B 侧压B4左伺服定位完成标志位
2114.06 BOOL  ; NC433_5_Z 4ST_B 侧压B4左伺服无原点标志位
2114.07 BOOL  ; NC433_5_Z 4ST_B 侧压B4左伺服原点停止标志位
2114.08 BOOL  ; NC433_5_Z 4ST_B 侧压B4左伺服0 区监测标志位
2114.09 BOOL  ; NC433_5_Z 4ST_B 侧压B4左伺服1 区监测标志位
2114.10 BOOL  ; NC433_5_Z 4ST_B 侧压B4左伺服2 区监测标志位
2114.11 BOOL  ; NC433_5_Z 4ST_B 侧压B4左伺服示教完成
2114.12 BOOL  ; NC433_5_Z 4ST_B 侧压B4左伺服错误标志
2114.13 BOOL  ; NC433_5_Z 4ST_B 侧压B4左伺服忙标志
2114.14 BOOL  ; NC433_5_Z 4ST_B 侧压B4左伺服数据传送标志位
2114.15 BOOL  ; NC433_5_Z 4ST_B 侧压B4左伺服减速停止执行标志位
2115.00 BOOL  ; NC433_5_Z 4ST_B 侧压B4左伺服预留
2115.01 BOOL  ; NC433_5_Z 4ST_B 侧压B4左伺服预留
2115.02 BOOL  ; NC433_5_Z 4ST_B 侧压B4左伺服预留
2115.03 BOOL  ; NC433_5_Z 4ST_B 侧压B4左伺服预留
2115.04 BOOL  ; NC433_5_Z 4ST_B 侧压B4左伺服预留
2115.05 BOOL  ; NC433_5_Z 4ST_B 侧压B4左伺服预留
2115.06 BOOL  ; NC433_5_Z 4ST_B 侧压B4左伺服预留
2115.07 BOOL  ; NC433_5_Z 4ST_B 侧压B4左伺服预留
2115.08 BOOL  ; NC433_5_Z 4ST_B 侧压B4左伺服CW极限输入信号
2115.09 BOOL  ; NC433_5_Z 4ST_B 侧压B4左伺服CCW极限输入信号
2115.10 BOOL  ; NC433_5_Z 4ST_B 侧压B4左伺服原点接近输入信号
2115.11 BOOL  ; NC433_5_Z 4ST_B 侧压B4左伺服原点输入信号
2115.12 BOOL  ; NC433_5_Z 4ST_B 侧压B4左伺服中断输入信号
2115.13 BOOL  ; NC433_5_Z 4ST_B 侧压B4左伺服紧急输入信号
2115.14 BOOL  ; NC433_5_Z 4ST_B 侧压B4左伺服定位完成输入信号
2115.15 BOOL  ; NC433_5_Z 4ST_B 侧压B4左伺服偏差计数器复位输出/ 原点调整命令输出
2116.00 BOOL  ; NC433_5_Z 4ST_B 侧压B4左伺服错误代码
2116.01 BOOL  ; NC433_5_Z 4ST_B 侧压B4左伺服错误代码
2116.02 BOOL  ; NC433_5_Z 4ST_B 侧压B4左伺服错误代码
2116.03 BOOL  ; NC433_5_Z 4ST_B 侧压B4左伺服错误代码
2116.04 BOOL  ; NC433_5_Z 4ST_B 侧压B4左伺服错误代码
2116.05 BOOL  ; NC433_5_Z 4ST_B 侧压B4左伺服错误代码
2116.06 BOOL  ; NC433_5_Z 4ST_B 侧压B4左伺服错误代码
2116.07 BOOL  ; NC433_5_Z 4ST_B 侧压B4左伺服错误代码
2116.08 BOOL  ; NC433_5_Z 4ST_B 侧压B4左伺服错误代码
2116.09 BOOL  ; NC433_5_Z 4ST_B 侧压B4左伺服错误代码
2116.10 BOOL  ; NC433_5_Z 4ST_B 侧压B4左伺服错误代码
2116.11 BOOL  ; NC433_5_Z 4ST_B 侧压B4左伺服错误代码
2116.12 BOOL  ; NC433_5_Z 4ST_B 侧压B4左伺服错误代码
2116.13 BOOL  ; NC433_5_Z 4ST_B 侧压B4左伺服错误代码
2116.14 BOOL  ; NC433_5_Z 4ST_B 侧压B4左伺服错误代码
2116.15 BOOL  ; NC433_5_Z 4ST_B 侧压B4左伺服错误代码
2117.00 BOOL  ; NC433_5_U 4ST_B 侧压B4右伺服预留
2117.01 BOOL  ; NC433_5_U 4ST_B 侧压B4右伺服预留
2117.02 BOOL  ; NC433_5_U 4ST_B 侧压B4右伺服预留
2117.03 BOOL  ; NC433_5_U 4ST_B 侧压B4右伺服预留
2117.04 BOOL  ; NC433_5_U 4ST_B 侧压B4右伺服等待存储器操作
2117.05 BOOL  ; NC433_5_U 4ST_B 侧压B4右伺服定位完成标志位
2117.06 BOOL  ; NC433_5_U 4ST_B 侧压B4右伺服无原点标志位
2117.07 BOOL  ; NC433_5_U 4ST_B 侧压B4右伺服原点停止标志位
2117.08 BOOL  ; NC433_5_U 4ST_B 侧压B4右伺服0 区监测标志位
2117.09 BOOL  ; NC433_5_U 4ST_B 侧压B4右伺服1 区监测标志位
2117.10 BOOL  ; NC433_5_U 4ST_B 侧压B4右伺服2 区监测标志位
2117.11 BOOL  ; NC433_5_U 4ST_B 侧压B4右伺服示教完成
2117.12 BOOL  ; NC433_5_U 4ST_B 侧压B4右伺服错误标志
2117.13 BOOL  ; NC433_5_U 4ST_B 侧压B4右伺服忙标志
2117.14 BOOL  ; NC433_5_U 4ST_B 侧压B4右伺服数据传送标志位
2117.15 BOOL  ; NC433_5_U 4ST_B 侧压B4右伺服减速停止执行标志位
2118.00 BOOL  ; NC433_5_U 4ST_B 侧压B4右伺服预留
2118.01 BOOL  ; NC433_5_U 4ST_B 侧压B4右伺服预留
2118.02 BOOL  ; NC433_5_U 4ST_B 侧压B4右伺服预留
2118.03 BOOL  ; NC433_5_U 4ST_B 侧压B4右伺服预留
2118.04 BOOL  ; NC433_5_U 4ST_B 侧压B4右伺服预留
2118.05 BOOL  ; NC433_5_U 4ST_B 侧压B4右伺服预留
2118.06 BOOL  ; NC433_5_U 4ST_B 侧压B4右伺服预留
2118.07 BOOL  ; NC433_5_U 4ST_B 侧压B4右伺服预留
2118.08 BOOL  ; NC433_5_U 4ST_B 侧压B4右伺服CW极限输入信号
2118.09 BOOL  ; NC433_5_U 4ST_B 侧压B4右伺服CCW极限输入信号
2118.10 BOOL  ; NC433_5_U 4ST_B 侧压B4右伺服原点接近输入信号
2118.11 BOOL  ; NC433_5_U 4ST_B 侧压B4右伺服原点输入信号
2118.12 BOOL  ; NC433_5_U 4ST_B 侧压B4右伺服中断输入信号
2118.13 BOOL  ; NC433_5_U 4ST_B 侧压B4右伺服紧急输入信号
2118.14 BOOL  ; NC433_5_U 4ST_B 侧压B4右伺服定位完成输入信号
2118.15 BOOL  ; NC433_5_U 4ST_B 侧压B4右伺服偏差计数器复位输出/ 原点调整命令输出
2119.00 BOOL  ; NC433_5_U 4ST_B 侧压B4右伺服错误代码
2119.01 BOOL  ; NC433_5_U 4ST_B 侧压B4右伺服错误代码
2119.02 BOOL  ; NC433_5_U 4ST_B 侧压B4右伺服错误代码
2119.03 BOOL  ; NC433_5_U 4ST_B 侧压B4右伺服错误代码
2119.04 BOOL  ; NC433_5_U 4ST_B 侧压B4右伺服错误代码
2119.05 BOOL  ; NC433_5_U 4ST_B 侧压B4右伺服错误代码
2119.06 BOOL  ; NC433_5_U 4ST_B 侧压B4右伺服错误代码
2119.07 BOOL  ; NC433_5_U 4ST_B 侧压B4右伺服错误代码
2119.08 BOOL  ; NC433_5_U 4ST_B 侧压B4右伺服错误代码
2119.09 BOOL  ; NC433_5_U 4ST_B 侧压B4右伺服错误代码
2119.10 BOOL  ; NC433_5_U 4ST_B 侧压B4右伺服错误代码
2119.11 BOOL  ; NC433_5_U 4ST_B 侧压B4右伺服错误代码
2119.12 BOOL  ; NC433_5_U 4ST_B 侧压B4右伺服错误代码
2119.13 BOOL  ; NC433_5_U 4ST_B 侧压B4右伺服错误代码
2119.14 BOOL  ; NC433_5_U 4ST_B 侧压B4右伺服错误代码
2119.15 BOOL  ; NC433_5_U 4ST_B 侧压B4右伺服错误代码
2120.00 BOOL  ; NC433_6_X1#存储器操作命令激活序列数
2120.01 BOOL  ; NC433_6_X1#存储器操作命令起动
2120.02 BOOL  ; NC433_6_X1#存储器操作命令独立起动
2120.03 BOOL  ; NC433_6_X1#直接操作命令绝对移动
2120.04 BOOL  ; NC433_6_X1#直接操作命令相对移动
2120.05 BOOL  ; NC433_6_X1#直接操作命令中断进给
2120.06 BOOL  ; NC433_6_X1#原点定位命令原点搜索
2120.07 BOOL  ; NC433_6_X1#原点定位命令原点返回
2120.08 BOOL  ; NC433_6_X1#原点定位命令当前位置预置
2120.09 BOOL  ; NC433_6_X1#点动
2120.10 BOOL  ; NC433_6_X1#点动方向(0=CW,1=CCW)
2120.11 BOOL  ; NC433_6_X1#示教
2120.12 BOOL  ; NC433_6_X1#错误清除
2120.13 BOOL  ; NC433_6_X1#偏差计数器复位输出/ 原点调整命令输出
2120.14 BOOL  ; NC433_6_X1#激活Override
2120.15 BOOL  ; NC433_6_X1#停止
2121.00 BOOL  ; NC433_6_X1#预留
2121.01 BOOL  ; NC433_6_X1#预留
2121.02 BOOL  ; NC433_6_X1#预留
2121.03 BOOL  ; NC433_6_X1#预留
2121.04 BOOL  ; NC433_6_X1#预留
2121.05 BOOL  ; NC433_6_X1#预留
2121.06 BOOL  ; NC433_6_X1#预留
2121.07 BOOL  ; NC433_6_X1#预留
2121.08 BOOL  ; NC433_6_X1#强制中断
2121.09 BOOL  ; NC433_6_X1#预留
2121.10 BOOL  ; NC433_6_X1#预留
2121.11 BOOL  ; NC433_6_X1#预留
2121.12 BOOL  ; NC433_6_X1#数据写入
2121.13 BOOL  ; NC433_6_X1#数据读出
2121.14 BOOL  ; NC433_6_X1#数据保存
2121.15 BOOL  ; NC433_6_X1#预留
2122.00 BOOL  ; NC433_6_Y 2#存储器操作命令激活序列数
2122.01 BOOL  ; NC433_6_Y 2#存储器操作命令起动
2122.02 BOOL  ; NC433_6_Y 2#存储器操作命令独立起动
2122.03 BOOL  ; NC433_6_Y 2#直接操作命令绝对移动
2122.04 BOOL  ; NC433_6_Y 2#直接操作命令相对移动
2122.05 BOOL  ; NC433_6_Y 2#直接操作命令中断进给
2122.06 BOOL  ; NC433_6_Y 2#原点定位命令原点搜索
2122.07 BOOL  ; NC433_6_Y 2#原点定位命令原点返回
2122.08 BOOL  ; NC433_6_Y 2#原点定位命令当前位置预置
2122.09 BOOL  ; NC433_6_Y 2#点动
2122.10 BOOL  ; NC433_6_Y 2#点动方向(0=CW,1=CCW)
2122.11 BOOL  ; NC433_6_Y 2#示教
2122.12 BOOL  ; NC433_6_Y 2#错误清除
2122.13 BOOL  ; NC433_6_Y 2#偏差计数器复位输出/ 原点调整命令输出
2122.14 BOOL  ; NC433_6_Y 2#激活Override
2122.15 BOOL  ; NC433_6_Y 2#停止
2123.00 BOOL  ; NC433_6_Y 2#预留
2123.01 BOOL  ; NC433_6_Y 2#预留
2123.02 BOOL  ; NC433_6_Y 2#预留
2123.03 BOOL  ; NC433_6_Y 2#预留
2123.04 BOOL  ; NC433_6_Y 2#预留
2123.05 BOOL  ; NC433_6_Y 2#预留
2123.06 BOOL  ; NC433_6_Y 2#预留
2123.07 BOOL  ; NC433_6_Y 2#预留
2123.08 BOOL  ; NC433_6_Y 2#强制中断
2123.09 BOOL  ; NC433_6_Y 2#预留
2123.10 BOOL  ; NC433_6_Y 2#预留
2123.11 BOOL  ; NC433_6_Y 2#预留
2123.12 BOOL  ; NC433_6_Y 2#数据写入
2123.13 BOOL  ; NC433_6_Y 2#数据读出
2123.14 BOOL  ; NC433_6_Y 2#数据保存
2123.15 BOOL  ; NC433_6_Y 2#预留
2124.00 BOOL  ; NC433_6_Z 3#存储器操作命令激活序列数
2124.01 BOOL  ; NC433_6_Z 3#存储器操作命令起动
2124.02 BOOL  ; NC433_6_Z 3#存储器操作命令独立起动
2124.03 BOOL  ; NC433_6_Z 3#直接操作命令绝对移动
2124.04 BOOL  ; NC433_6_Z 3#直接操作命令相对移动
2124.05 BOOL  ; NC433_6_Z 3#直接操作命令中断进给
2124.06 BOOL  ; NC433_6_Z 3#原点定位命令原点搜索
2124.07 BOOL  ; NC433_6_Z 3#原点定位命令原点返回
2124.08 BOOL  ; NC433_6_Z 3#原点定位命令当前位置预置
2124.09 BOOL  ; NC433_6_Z 3#点动
2124.10 BOOL  ; NC433_6_Z 3#点动方向(0=CW,1=CCW)
2124.11 BOOL  ; NC433_6_Z 3#示教
2124.12 BOOL  ; NC433_6_Z 3#错误清除
2124.13 BOOL  ; NC433_6_Z 3#偏差计数器复位输出/ 原点调整命令输出
2124.14 BOOL  ; NC433_6_Z 3#激活Override
2124.15 BOOL  ; NC433_6_Z 3#停止
2125.00 BOOL  ; NC433_6_Z 3#预留
2125.01 BOOL  ; NC433_6_Z 3#预留
2125.02 BOOL  ; NC433_6_Z 3#预留
2125.03 BOOL  ; NC433_6_Z 3#预留
2125.04 BOOL  ; NC433_6_Z 3#预留
2125.05 BOOL  ; NC433_6_Z 3#预留
2125.06 BOOL  ; NC433_6_Z 3#预留
2125.07 BOOL  ; NC433_6_Z 3#预留
2125.08 BOOL  ; NC433_6_Z 3#强制中断
2125.09 BOOL  ; NC433_6_Z 3#预留
2125.10 BOOL  ; NC433_6_Z 3#预留
2125.11 BOOL  ; NC433_6_Z 3#预留
2125.12 BOOL  ; NC433_6_Z 3#数据写入
2125.13 BOOL  ; NC433_6_Z 3#数据读出
2125.14 BOOL  ; NC433_6_Z 3#数据保存
2125.15 BOOL  ; NC433_6_Z 3#预留
2126.00 BOOL  ; NC433_6_U 7ST接料伺服存储器操作命令激活序列数
2126.01 BOOL  ; NC433_6_U 7ST接料伺服存储器操作命令起动
2126.02 BOOL  ; NC433_6_U 7ST接料伺服存储器操作命令独立起动
2126.03 BOOL  ; NC433_6_U 7ST接料伺服直接操作命令绝对移动
2126.04 BOOL  ; NC433_6_U 7ST接料伺服直接操作命令相对移动
2126.05 BOOL  ; NC433_6_U 7ST接料伺服直接操作命令中断进给
2126.06 BOOL  ; NC433_6_U 7ST接料伺服原点定位命令原点搜索
2126.07 BOOL  ; NC433_6_U 7ST接料伺服原点定位命令原点返回
2126.08 BOOL  ; NC433_6_U 7ST接料伺服原点定位命令当前位置预置
2126.09 BOOL  ; NC433_6_U 7ST接料伺服点动
2126.10 BOOL  ; NC433_6_U 7ST接料伺服点动方向(0=CW,1=CCW)
2126.11 BOOL  ; NC433_6_U 7ST接料伺服示教
2126.12 BOOL  ; NC433_6_U 7ST接料伺服错误清除
